# B&R Automation Studio project A2019059_Linka_Power_CP (part 2)

### Cpu.per - 5PC900_TS17_00/Cpu.per
```iecst
VAR_CONFIG
	Paletka AT %M0; (* *)
	P1_Skrutk_4F_DPS_M4_Vysunutie AT %MD5944; (* *)
	P1_Skrutk_4F_LavaK30_Vysunutie AT %MD5948; (* *)
	P1_Skrutk_4F_PravaK30_Vysunutie AT %MD5952; (* *)
	P1_Skrutk_4F_PrednaM4_Vysunutie AT %MD5956; (* *)
	P1_Skrutk_4F_ZadnaM4_Vysunutie AT %MD5960; (* *)
	P1_Skrutk_5F_DPS_M4_Vysunutie AT %MD5964; (* *)
	P1_Skrutk_5F_LavaK30_Vysunutie AT %MD5968; (* *)
	P1_Skrutk_5F_PravaK30_Vysunutie AT %MD5972; (* *)
	P1_Skrutk_5F_PrednaM4_Vysunutie AT %MD5976; (* *)
	P1_Skrutk_5F_ZadnaM4_Vysunutie AT %MD5980; (* *)
	P1_Skrutk_5H_LavaK30_Vysunutie AT %MD5984; (* *)
	P1_Skrutk_5H_LavaM5_Vysunutie AT %MD5988; (* *)
	P1_Skrutk_5H_PravaK30_Vysunutie AT %MD5992; (* *)
	P1_Skrutk_5H_PravaM5_Vysunutie AT %MD5996; (* *)
	P1_Skrutk_5H_StrednaM5_Vysunutie AT %MD6000; (* *)
	P2_Maticovacka_5H_Vysunutie AT %MD6004; (* *)
	P2_Skrutk_4F_LavaM4_Vysunutie AT %MD6008; (* *)
	P2_Skrutk_4F_LavaM6_Vysunutie AT %MD6012; (* *)
	P2_Skrutk_4F_PravaM4_Vysunutie AT %MD6016; (* *)
	P2_Skrutk_4F_PravaM6_Vysunutie AT %MD6020; (* *)
	P2_Skrutk_5F_LavaM4_Vysunutie AT %MD6024; (* *)
	P2_Skrutk_5F_LavaM6_Vysunutie AT %MD6028; (* *)
	P2_Skrutk_5F_PravaM4_Vysunutie AT %MD6032; (* *)
	P2_Skrutk_5F_PravaM6_Vysunutie AT %MD6036; (* *)
	P2_Skrutk_5H_LavaM5_Vysunutie AT %MD6040; (* *)
	P2_Skrutk_5H_PravaM5_Vysunutie AT %MD6044; (* *)
	P2_Skrutk_5H_StrednaM4_Vysunutie AT %MD6048; (* *)
	P3_Skrutk_4F_StredK40_Vysunutie AT %MD6052; (* *)
	P3_Skrutk_4F_StredM5_Vysunutie AT %MD6056; (* *)
	P3_Skrutk_5F_StredK40_Vysunutie AT %MD6060; (* *)
	P3_Skrutk_5F_StredM5_Vysunutie AT %MD6064; (* *)
	P3_Skrutk_5H_StredM5_Vysunutie AT %MD6068; (* *)
	Buffer_1 AT %M6072; (* *)
	Buffer_2 AT %M6280; (* *)
	Buffer_3 AT %M6488; (* *)
	Buffer_4 AT %M6696; (* *)
	Buffer_5 AT %M6904; (* *)
	Buffer_6 AT %M7112; (* *)
	Buffer_7 AT %M7320; (* *)
	Buffer_8 AT %M7528; (* *)
	Buffer_9 AT %M7736; (* *)
	Buffer_10 AT %M7944; (* *)
	Buffer_11 AT %M8152; (* *)
	Buffer_12 AT %M8360; (* *)
	Buffer_13 AT %M8568; (* *)
	Buffer_14 AT %M8776; (* *)
	Buffer_15 AT %M8984; (* *)
	Buffer_16 AT %M9192; (* *)
	Buffer_17 AT %M9400; (* *)
	Buffer_18 AT %M9608; (* *)
	Buffer_19 AT %M9816; (* *)
	Buffer_20 AT %M10024; (* *)
END_VAR
```

### IoMap.iom - 5PC900_TS17_00/IoMap.iom
```iecst
VAR_CONFIG
	Cyclic#1.Safety.IN.P2_Robot_TlacitkoCS_CH1_CS4 AT %IX."AB2.4_20xSI".SafeDigitalInput01;
	Cyclic#1.Safety.IN.P2_Robot_TlacitkoCS_CH2_CS4 AT %IX."AB2.4_20xSI".SafeDigitalInput02;
	Cyclic#1.Safety.IN.P2_Panel_TlacitkoCS_CH1_CS2 AT %IX."AB2.4_20xSI".SafeDigitalInput03;
	Cyclic#1.Safety.IN.P2_Panel_TlacitkoCS_CH2_CS2 AT %IX."AB2.4_20xSI".SafeDigitalInput04;
	Cyclic#1.Safety.IN.P2_VyblokovanieSafety_CH1_SA1 AT %IX."AB2.4_20xSI".SafeDigitalInput05;
	Cyclic#1.Safety.IN.P2_VyblokovanieSafety_CH2_SA1 AT %IX."AB2.4_20xSI".SafeDigitalInput06;
	Cyclic#1.Safety.IN.P2_Skrina_TlacitkoCS_CH1_CS3 AT %IX."AB2.4_20xSI".SafeDigitalInput07;
	Cyclic#1.Safety.IN.P2_Skrina_TlacitkoCS_CH2_CS3 AT %IX."AB2.4_20xSI".SafeDigitalInput08;
	Cyclic#1.Safety.IN.P2_ZaklTesn_PojazdSnim_CH1_B2 AT %IX."AB2.4_20xSI".SafeDigitalInput09;
	Cyclic#1.Safety.IN.P2_ZaklTesn_PojazdSnim_CH2_B2 AT %IX."AB2.4_20xSI".SafeDigitalInput10;
	Cyclic#1.P2_Dopravniky.IN.HornyDoprav_TeplotaMotora_OK AT %IX."AB2.4_20xSI".SafeDigitalInput11;
	Cyclic#1.P2_Dopravniky.IN.SpodnyDoprav_TeplotaMotora_OK AT %IX."AB2.4_20xSI".SafeDigitalInput12;
	Cyclic#1.Safety.IN.P2_ZaklTesn_Bumper_CH1_B1 AT %IX."AB2.4_20xSI".SafeDigitalInput13;
	Cyclic#1.Safety.IN.P2_ZaklTesn_Bumper_CH2_B1 AT %IX."AB2.4_20xSI".SafeDigitalInput14;
	Cyclic#1.P2_Pracovisko.IN.PrepatovaOchrana_OK AT %IX."AB2.7_16xDI".DigitalInput01;
	Cyclic#1.P2_Pracovisko.IN.NapajaniaRobota_OK AT %IX."AB2.7_16xDI".DigitalInput02;
	Cyclic#1.P2_SkrutkovacMatic.IN.NapajanieSkrutkovackyMatic_OK AT %IX."AB2.7_16xDI".DigitalInput03;
	Cyclic#1.P2_Srobovanie.IN.NapajanieSkrutkovackyM6_OK AT %IX."AB2.7_16xDI".DigitalInput04;
	Cyclic#1.P2_Srobovanie.IN.NapajanieSkrutkovackyM4_OK AT %IX."AB2.7_16xDI".DigitalInput05;
	Cyclic#1.P2_Srobovanie.IN.NapajanieSkrutkovackyM5_OK AT %IX."AB2.7_16xDI".DigitalInput06;
	Cyclic#1.P2_Srobovanie.IN.NapajanieVibroZasobnikaM5_OK AT %IX."AB2.7_16xDI".DigitalInput07;
	Cyclic#1.P2_Srobovanie.IN.NapajanieVibroZasobnikaM4_OK AT %IX."AB2.7_16xDI".DigitalInput08;
	Cyclic#1.P2_Srobovanie.IN.NapajanieVibroZasobnikaM6_OK AT %IX."AB2.7_16xDI".DigitalInput09;
	Cyclic#1.P2_SkrutkovacMatic.IN.NapajanieVibroZasobnikaMatic_OK AT %IX."AB2.7_16xDI".DigitalInput10;
	Cyclic#1.P2_Dopravniky.IN.HornyDoprav_READY AT %IX."AB2.7_16xDI".DigitalInput11;
	Cyclic#1.P2_Dopravniky.IN.SpodnyDoprav_READY AT %IX."AB2.7_16xDI".DigitalInput12;
	Cyclic#1.P2_Zvaranie.IN.NapajanieZvaracky_OK AT %IX."AB2.7_16xDI".DigitalInput13;
	Cyclic#1.P2_Cistenie.IN.Ionizator_Alarm1 AT %IX."AB2.7_16xDI".DigitalInput14;
	Cyclic#1.P2_Cistenie.IN.Ionizator_Alarm2 AT %IX."AB2.7_16xDI".DigitalInput15;
	Cyclic#1.P2_Cistenie.IN.Ionizator_Alarm3 AT %IX."AB2.7_16xDI".DigitalInput16;
	Cyclic#1.P2_Pracovisko.STAV.KartaAB24_OK AT %IX."AB2.4_20xSI".ModuleOk;
	Cyclic#1.P2_Pracovisko.STAV.KartaAB25_OK AT %IX."AB2.5_4xSO".ModuleOk;
	Cyclic#1.P2_Pracovisko.STAV.KartaAB26_OK AT %IX."AB2.6_4xSO".ModuleOk;
	Cyclic#1.P2_Pracovisko.STAV.KartaAB27_OK AT %IX."AB2.7_16xDI".ModuleOk;
	Cyclic#1.P2_Pracovisko.STAV.KartaAB28_OK AT %IX."AB2.8_16xDI".ModuleOk;
	Cyclic#1.P2_Pracovisko.STAV.KartaAB29_OK AT %IX."AB2.9_16xDO".ModuleOk;
	Cyclic#1.P2_Pracovisko.STAV.KartaAB210_OK AT %IX."AB2.10_16xDO".ModuleOk;
	Cyclic#1.P2_Pracovisko.STAV.KartaAB211_OK AT %IX."AB2.11_X2X".ModuleOk;
	Cyclic#1.P2_Pracovisko.STAV.ModulDM21_OK AT %IX."DM2.1_16DI/DO".ModuleOk;
	Cyclic#1.P2_Pracovisko.STAV.ModulDI21_OK AT %IX."DI2.1_8DI".ModuleOk;
	Cyclic#1.P2_Pracovisko.STAV.ModulDI22_OK AT %IX."DI2.2_16DI".ModuleOk;
	Cyclic#1.P2_Pracovisko.STAV.ModulDI23_OK AT %IX."DI2.3_16DI".ModuleOk;
	Cyclic#1.P2_Pracovisko.STAV.ModulDI24_OK AT %IX."DI2.4_16DI".ModuleOk;
	Cyclic#1.P2_Pracovisko.STAV.ModulDI25_OK AT %IX."DI2.5_16DI".ModuleOk;
	Cyclic#1.P2_Pracovisko.STAV.ModulSI21_OK AT %IX."SI2.1".ModuleOk;
	Cyclic#1.P2_Pracovisko.STAV.ModulSI22_OK AT %IX."SI2.2".ModuleOk;
	Cyclic#1.P2_Zvaranie.IN.ZvarackaStav_RUN AT %IX."AB2.8_16xDI".DigitalInput01;
	Cyclic#1.P2_Zvaranie.IN.ZvarackaStav_READY AT %IX."AB2.8_16xDI".DigitalInput02;
	Cyclic#1.Safety.IN.P2_SV_Ventil1_ZonaBunka AT %IX."AB2.8_16xDI".DigitalInput04;
	Cyclic#1.Safety.IN.P2_SV_Ventil2_ZonaBunka AT %IX."AB2.8_16xDI".DigitalInput05;
	Cyclic#1.Safety.IN.P2_SV_Ventil_ZonaMaticov AT %IX."AB2.8_16xDI".DigitalInput06;
	Cyclic#1.Safety.IN.P2_SV_ZonaCS AT %IX."AB2.8_16xDI".DigitalInput07;
	Cyclic#1.Safety.IN.P2_SV_ZonaBunka AT %IX."AB2.8_16xDI".DigitalInput08;
	Cyclic#1.Safety.IN.P2_SV_ZonaZaklTesneniaPojazd AT %IX."AB2.8_16xDI".DigitalInput09;
	Cyclic#1.Safety.IN.P2_SV_ZonaZaklTesneniaZdvih AT %IX."AB2.8_16xDI".DigitalInput10;
	Cyclic#1.P2_Pracovisko.OUT.Majak_ZeleneSvetlo AT %QX."AB2.9_16xDO".DigitalOutput01;
	Cyclic#1.P2_Pracovisko.OUT.Majak_ZlteSvetlo AT %QX."AB2.9_16xDO".DigitalOutput02;
	Cyclic#1.P2_Pracovisko.OUT.Majak_CerveneSvetlo AT %QX."AB2.9_16xDO".DigitalOutput03;
	Cyclic#1.P2_Pracovisko.OUT.Majak_Hukacka AT %QX."AB2.9_16xDO".DigitalOutput04;
	Cyclic#1.P2_Cistenie.OUT.Ionizator_RUN_ZX2 AT %QX."AB2.9_16xDO".DigitalOutput09;
	Cyclic#1.P2_Zvaranie.OUT.Zvaracka_START AT %QX."AB2.9_16xDO".DigitalOutput10;
	Cyclic#1.P2_Zvaranie.OUT.Zvaracka_RESET AT %QX."AB2.9_16xDO".DigitalOutput11;
	Cyclic#1.P2_SkrutkovacMatic.OUT.SkrutkMatic_VYSUN_YV62 AT %QX."AB2.10_16xDO".DigitalOutput01;
	Cyclic#1.P2_SkrutkovacMatic.OUT.SkrutkMatic_ZASUN_YV75 AT %QX."AB2.10_16xDO".DigitalOutput02;
	Cyclic#1.P2_Pracovisko.OUT.OsvetlenieBunky AT %QX."AB2.10_16xDO".DigitalOutput03;
	Cyclic#1.P2_Srobovanie.OUT.ZasobSrobM6_Banner_CervenaLED AT %QX."DM2.1_16DI/DO".DigitalOutput09;
	Cyclic#1.P2_Srobovanie.IN.ZasobSrobM6_Banner_SB3 AT %IX."DM2.1_16DI/DO".DigitalInput10;
	Cyclic#1.P2_SkrutkovacMatic.IN.ZasobMatic_Banner_SB4 AT %IX."DM2.1_16DI/DO".DigitalInput12;
	Cyclic#1.P2_Srobovanie.OUT.ZasobSrobM4_Banner_CervenaLED AT %QX."DM2.1_16DI/DO".DigitalOutput13;
	Cyclic#1.P2_Srobovanie.IN.ZasobSrobM4_Banner_SB5 AT %IX."DM2.1_16DI/DO".DigitalInput14;
	Cyclic#1.P2_Srobovanie.OUT.ZasobSrobM5_Banner_CervenaLED AT %QX."DM2.1_16DI/DO".DigitalOutput15;
	Cyclic#1.P2_Srobovanie.IN.ZasobSrobM5_Banner_SB6 AT %IX."DM2.1_16DI/DO".DigitalInput16;
	Cyclic#1.P2_SkrutkovacMatic.OUT.ZasobMatic_Banner_CervenaLED AT %QX."DM2.1_16DI/DO".DigitalOutput11;
	Cyclic#1.P2_Srobovanie.IN.ManipulOsY_LimSnimacPOS_IS19 AT %IX."DI2.1_8DI".DigitalInput01;
	Cyclic#1.P2_Srobovanie.IN.ManipulOsY_LimSnimacNEG_IS20 AT %IX."DI2.1_8DI".DigitalInput02;
	Cyclic#1.P2_Srobovanie.IN.ManipulOsX_LimSnimacPOS_IS21 AT %IX."DI2.1_8DI".DigitalInput03;
	Cyclic#1.P2_Srobovanie.IN.ManipulOsX_LimSnimacNEG_IS22 AT %IX."DI2.1_8DI".DigitalInput04;
	Cyclic#1.P2_Zvaranie.IN.ZdvihZvarania_RefSnimac_IS9 AT %IX."DI2.2_16DI".DigitalInput01;
	Cyclic#1.P2_Zvaranie.IN.PojazdZvarania_PozVPRAVO_IS10 AT %IX."DI2.2_16DI".DigitalInput02;
	Cyclic#1.P2_Zvaranie.IN.PojazdZvarania_PozVLAVO_IS11 AT %IX."DI2.2_16DI".DigitalInput03;
	Cyclic#1.P2_Cistenie.IN.Dvere_OTVORENE_MS7 AT %IX."DI2.2_16DI".DigitalInput09;
	Cyclic#1.P2_Cistenie.IN.Dvere_ZATVORENE_MS8 AT %IX."DI2.2_16DI".DigitalInput10;
	Cyclic#1.P2_Cistenie.IN.VakumDosiahnute_S5 AT %IX."DI2.2_16DI".DigitalInput11;
	Cyclic#1.P2_Robot.IN.DokStanPritGripra_MVcase_IS1 AT %IX."DI2.2_16DI".DigitalInput12;
	Cyclic#1.P2_Robot.IN.DokStanPritGripra_BusBary45F_IS2 AT %IX."DI2.2_16DI".DigitalInput13;
	Cyclic#1.P2_Robot.IN.DokStanPritGripra_BusBary5H_IS3 AT %IX."DI2.2_16DI".DigitalInput14;
	Cyclic#1.P2_Robot.IN.SnimacVakua_45F_S1 AT %IX."DI2.2_16DI".DigitalInput15;
	Cyclic#1.P2_Robot.IN.SnimacVakua_5H_S2 AT %IX."DI2.2_16DI".DigitalInput16;
	Cyclic#1.P2_StoperMaticovacky.IN.Centrovanie_VYSUNUTE_IS12 AT %IX."DI2.3_16DI".DigitalInput01;
	Cyclic#1.P2_StoperMaticovacky.IN.Centrovanie_ZASUNUTE_IS13 AT %IX."DI2.3_16DI".DigitalInput02;
	Cyclic#1.P2_StoperSrobovania.IN.Centrovanie_VYSUNUTE_IS14 AT %IX."DI2.3_16DI".DigitalInput03;
	Cyclic#1.P2_StoperSrobovania.IN.Centrovanie_ZASUNUTE_IS15 AT %IX."DI2.3_16DI".DigitalInput04;
	Cyclic#1.P2_StoperZvarania.IN.Centrovanie_VYSUNUTE_IS16 AT %IX."DI2.3_16DI".DigitalInput05;
	Cyclic#1.P2_StoperZvarania.IN.Centrovanie_ZASUNUTE_IS17 AT %IX."DI2.3_16DI".DigitalInput06;
	Cyclic#1.P2_Dopravniky.IN.SpodnyDoprav_Zaplnenie_IS18 AT %IX."DI2.3_16DI".DigitalInput07;
	Cyclic#1.P2_Srobovanie.IN.SkrutkM5_SrobaPresla_IS32 AT %IX."DI2.3_16DI".DigitalInput15;
	Cyclic#1.P2_Srobovanie.IN.SkrutkM5_Cist_SrobaPresla_IS31 AT %IX."DI2.3_16DI".DigitalInput14;
	Cyclic#1.P2_Srobovanie.IN.SkrutkM5_Cist_BrzdaZatvorena_MS2 AT %IX."DI2.3_16DI".DigitalInput13;
	Cyclic#1.P2_Srobovanie.IN.SkrutkM5_Cist_BrzdaOtvorena_MS1 AT %IX."DI2.3_16DI".DigitalInput12;
	Cyclic#1.P2_Srobovanie.IN.NastrelSrobM5_SrobaPresla_IS29 AT %IX."DI2.3_16DI".DigitalInput11;
	Cyclic#1.P2_Srobovanie.IN.ZasobSrobM5_ListaPLNA_OS3 AT %IX."DI2.3_16DI".DigitalInput10;
	Cyclic#1.P2_Srobovanie.IN.ZasobSrobM5_PRAZDNY_IS28 AT %IX."DI2.3_16DI".DigitalInput09;
	Cyclic#1.P2_SkrutkovacMatic.IN.ZasobMatic_PRAZDNY_IS23 AT %IX."DI2.4_16DI".DigitalInput01;
	Cyclic#1.P2_SkrutkovacMatic.IN.ZasobMatic_ListaPLNA_OS1 AT %IX."DI2.4_16DI".DigitalInput02;
	Cyclic#1.P2_SkrutkovacMatic.IN.OddelMatic_MaticaPresla_IS24 AT %IX."DI2.4_16DI".DigitalInput03;
	Cyclic#1.P2_SkrutkovacMatic.IN.DavkMatic_PritomnostMatice_OS2 AT %IX."DI2.4_16DI".DigitalInput04;
	Cyclic#1.P2_SkrutkovacMatic.IN.DavkMatic_ZASUNUTY_IS25 AT %IX."DI2.4_16DI".DigitalInput05;
	Cyclic#1.P2_SkrutkovacMatic.IN.DavkMatic_VYSUNUTY_IS26 AT %IX."DI2.4_16DI".DigitalInput06;
	Cyclic#1.P2_SkrutkovacMatic.IN.DavkMatic_MaticaPresla_IS27 AT %IX."DI2.4_16DI".DigitalInput07;
	Cyclic#1.P2_SkrutkovacMatic.IN.SkrutkMatic_ZASUNUTY_MS9 AT %IX."DI2.4_16DI".DigitalInput08;
	Cyclic#1.P2_Srobovanie.IN.ZasobSrobM4_PRAZDNY_IS33 AT %IX."DI2.4_16DI".DigitalInput09;
	Cyclic#1.P2_Srobovanie.IN.ZasobSrobM4_ListaPLNA_OS4 AT %IX."DI2.4_16DI".DigitalInput10;
	Cyclic#1.P2_Srobovanie.IN.NastrelSrobM4_SrobaPresla_IS34 AT %IX."DI2.4_16DI".DigitalInput11;
	Cyclic#1.P2_Srobovanie.IN.SkrutkM4_Cist_BrzdaOtvorena_MS12 AT %IX."DI2.4_16DI".DigitalInput12;
	Cyclic#1.P2_Srobovanie.IN.SkrutkM4_Cist_BrzdaZatvoren_MS13 AT %IX."DI2.4_16DI".DigitalInput13;
	Cyclic#1.P2_Srobovanie.IN.SkrutkM4_Cist_SrobaPresla_IS35 AT %IX."DI2.4_16DI".DigitalInput14;
	Cyclic#1.P2_Srobovanie.IN.SkrutkM4_SrobaPresla_IS30 AT %IX."DI2.4_16DI".DigitalInput15;
	Cyclic#1.P2_Srobovanie.IN.ZasobSrobM6_PRAZDNY_IS36 AT %IX."DI2.5_16DI".DigitalInput01;
	Cyclic#1.P2_Srobovanie.IN.ZasobSrobM6_ListaPLNA_OS5 AT %IX."DI2.5_16DI".DigitalInput02;
	Cyclic#1.P2_Srobovanie.IN.NastrelSrobM6_SrobaPresla_IS37 AT %IX."DI2.5_16DI".DigitalInput03;
	Cyclic#1.P2_Srobovanie.IN.SkrutkM6_Cist_BrzdaOtvorena_MS15 AT %IX."DI2.5_16DI".DigitalInput04;
	Cyclic#1.P2_Srobovanie.IN.SkrutkM6_Cist_BrzdaZatvoren_MS16 AT %IX."DI2.5_16DI".DigitalInput05;
	Cyclic#1.P2_Srobovanie.IN.SkrutkM6_Cist_SrobaPresla_IS39 AT %IX."DI2.5_16DI".DigitalInput06;
	Cyclic#1.P2_Srobovanie.IN.SkrutkM6_SrobaPresla_IS38 AT %IX."DI2.5_16DI".DigitalInput07;
	Cyclic#1.P2_ZakladacTesnenia.IN.ZdvihZaklad_RefSnimac_IS8 AT %IX."DI2.5_16DI".DigitalInput09;
	Cyclic#1.P2_ZakladacTesnenia.IN.Vozik_Zaklad_PritomPowerCP_IOS6 AT %IX."DI2.5_16DI".DigitalInput14;
	Cyclic#1.P2_ZakladacTesnenia.IN.Kopito_ZakladPoloha_IS7 AT %IX."DI2.5_16DI".DigitalInput15;
	Cyclic#1.P2_Pracovisko.IN.PrivodVzduchu_SnimacTlaku_S3 AT %IX."DI2.5_16DI".DigitalInput16;
	Cyclic#1.Safety.IN.P2_ZamkyBunky_CH1 AT %IX."SI2.1".SafeDigitalInput01;
	Cyclic#1.Safety.IN.P2_ZamkyBunky_CH2 AT %IX."SI2.1".SafeDigitalInput02;
	Cyclic#1.Safety.OUT.P2_ZamkniZamok_PredneDvereLS AT %QX."DM2.1_16DI/DO".DigitalOutput01;
	Cyclic#1.Safety.IN.P2_PredneDvereLS_PritomPetlice AT %IX."DM2.1_16DI/DO".DigitalInput02;
	Cyclic#1.Safety.OUT.P2_ZamkniZamok_PredneDverePS AT %QX."DM2.1_16DI/DO".DigitalOutput03;
	Cyclic#1.Safety.IN.P2_PredneDverePS_PritomPetlice AT %IX."DM2.1_16DI/DO".DigitalInput04;
	Cyclic#1.Safety.IN.P2_ZaklTesn_Bariera_CH1_BC1 AT %IX."SI2.1".SafeDigitalInput03;
	Cyclic#1.Safety.IN.P2_ZaklTesn_Bariera_CH2_BC1 AT %IX."SI2.1".SafeDigitalInput04;
	Cyclic#1.Safety.IN.P2_TlacitkoCS_CH1_CS1 AT %IX."SI2.1".SafeDigitalInput05;
	Cyclic#1.Safety.IN.P2_TlacitkoCS_CH2_CS1 AT %IX."SI2.1".SafeDigitalInput06;
	Cyclic#1.Safety.IN.P2_VstupBunky_Bariera_CH1_BC2 AT %IX."SI2.2".SafeDigitalInput01;
	Cyclic#1.Safety.IN.P2_VstupBunky_Bariera_CH2_BC2 AT %IX."SI2.2".SafeDigitalInput02;
	Cyclic#1.Safety.IN.P2_ZaklTesn_DvojrOvladLS_CH1_SB1 AT %IX."SI2.2".SafeDigitalInput05;
	Cyclic#1.Safety.IN.P2_ZaklTesn_DvojrOvladLS_CH2_SB1 AT %IX."SI2.2".SafeDigitalInput06;
	Cyclic#1.Safety.IN.P2_ZaklTesn_DvojrOvladPS_CH1_SB2 AT %IX."SI2.2".SafeDigitalInput07;
	Cyclic#1.Safety.IN.P2_ZaklTesn_DvojrOvladPS_CH2_SB2 AT %IX."SI2.2".SafeDigitalInput08;
	Cyclic#1.P2_Pracovisko.OUT.VT1_OUT1 AT %QB."VentilovyTerminal_VT1".OUT1_I2200_S01Out;
	Cyclic#1.P2_Pracovisko.OUT.VT1_OUT2 AT %QB."VentilovyTerminal_VT1".OUT2_I2200_S02Out;
	Cyclic#1.P2_Pracovisko.OUT.VT1_OUT3 AT %QB."VentilovyTerminal_VT1".OUT3_I2200_S03Out;
	Cyclic#1.P2_Pracovisko.OUT.VT1_OUT4 AT %QB."VentilovyTerminal_VT1".OUT4_I2200_S04Out;
	Cyclic#1.P2_Pracovisko.OUT.VT2_OUT1 AT %QB."VentilovyTerminal_VT2".OUT1_I2200_S01Out;
	Cyclic#1.P2_Pracovisko.OUT.VT2_OUT2 AT %QB."VentilovyTerminal_VT2".OUT2_I2200_S02Out;
	Cyclic#1.P2_Pracovisko.OUT.VT2_OUT3 AT %QB."VentilovyTerminal_VT2".OUT3_I2200_S03Out;
	Cyclic#1.P2_Pracovisko.OUT.VT2_OUT4 AT %QB."VentilovyTerminal_VT2".OUT4_I2200_S04Out;
	Cyclic#1.P2_Pracovisko.OUT.VT3_OUT1 AT %QB."VentilovyTerminal_VT3".OUT1_I2200_S01Out;
	Cyclic#1.P2_Pracovisko.OUT.VT3_OUT2 AT %QB."VentilovyTerminal_VT3".OUT2_I2200_S02Out;
	Cyclic#1.P2_Pracovisko.OUT.VT3_OUT3 AT %QB."VentilovyTerminal_VT3".OUT3_I2200_S03Out;
	Cyclic#1.P2_Pracovisko.OUT.VT3_OUT4 AT %QB."VentilovyTerminal_VT3".OUT4_I2200_S04Out;
	Cyclic#1.Safety.IN.ZonaCS_RESET AT %QX."SL1_SafetyMaster".BOOL101;
	Cyclic#1.Safety.IN.P2_ZonaZaklTesneniaPojazd_RESET AT %QX."SL1_SafetyMaster".BOOL102;
	Cyclic#1.Safety.IN.P2_ZonaZaklTesneniaZdvih_RESET AT %QX."SL1_SafetyMaster".BOOL103;
	Cyclic#1.Safety.IN.P2_ZonaMaticovacky_RESET AT %QX."SL1_SafetyMaster".BOOL104;
	Cyclic#1.Safety.IN.P2_ZonaBunky_RESET AT %QX."SL1_SafetyMaster".BOOL105;
	Cyclic#1.P2_Pracovisko.IN.PrivodVzduchu_SnimacTlaku_S3 AT %QX."SL1_SafetyMaster".BOOL106;
	Cyclic#1.Safety.IN.P2_SV_Ventil_ZonaMaticov AT %QX."SL1_SafetyMaster".BOOL107;
	Cyclic#1.Safety.IN.P2_SV_Ventil1_ZonaBunka AT %QX."SL1_SafetyMaster".BOOL108;
	Cyclic#1.Safety.IN.P2_SV_Ventil2_ZonaBunka AT %QX."SL1_SafetyMaster".BOOL109;
	Cyclic#1.Safety.IN.P2_SV_ZonaBunka AT %QX."SL1_SafetyMaster".BOOL110;
	Cyclic#1.Safety.IN.P2_SV_ZonaCS AT %QX."SL1_SafetyMaster".BOOL111;
	Cyclic#1.Safety.IN.P2_SV_ZonaZaklTesneniaPojazd AT %QX."SL1_SafetyMaster".BOOL112;
	Cyclic#1.Safety.IN.P2_SV_ZonaZaklTesneniaZdvih AT %QX."SL1_SafetyMaster".BOOL113;
	Cyclic#1.Safety.STAV.SafetyPLC_Nabehlo AT %IX."SL1_SafetyMaster".BOOL001;
	Cyclic#1.Safety.STAV.P2_TlacitkoCS_AKTIVNE AT %IX."SL1_SafetyMaster".BOOL002;
	Cyclic#1.Safety.STAV.P2_Panel_TlacitkoCS_AKTIVNE AT %IX."SL1_SafetyMaster".BOOL003;
	Cyclic#1.Safety.STAV.P2_Robot_TlacitkoCS_AKTIVNE AT %IX."SL1_SafetyMaster".BOOL004;
	Cyclic#1.Safety.STAV.P2_Skrina_TlacitkoCS_AKTIVNE AT %IX."SL1_SafetyMaster".BOOL005;
	Cyclic#1.Safety.STAV.P2_VstupBunky_Bariera_AKTIVNA AT %IX."SL1_SafetyMaster".BOOL006;
	Cyclic#1.Safety.STAV.P2_ZaklTesnenia_Bariera_AKTIVNA AT %IX."SL1_SafetyMaster".BOOL007;
	Cyclic#1.Safety.STAV.P2_ZaklTesnenia_Bumper_AKTIVNY AT %IX."SL1_SafetyMaster".BOOL008;
	Cyclic#1.Safety.STAV.P2_DvojrucneOvladanie_AKTIVNE AT %IX."SL1_SafetyMaster".BOOL009;
	Cyclic#1.Safety.STAV.P2_ZamkyBunky_AKTIVNE AT %IX."SL1_SafetyMaster".BOOL010;
	Cyclic#1.Safety.STAV.P2_ZonaMaticovacky_AKTIVNA AT %IX."SL1_SafetyMaster".BOOL011;
	Cyclic#1.Safety.STAV.P2_ZonaZaklTesnenPojazd_AKTIVNA AT %IX."SL1_SafetyMaster".BOOL012;
	Cyclic#1.Safety.STAV.P2_ZonaZaklTesnenZdvih_AKTIVNA AT %IX."SL1_SafetyMaster".BOOL013;
	Cyclic#1.Safety.STAV.ZonaCS_AKTIVNA AT %IX."SL1_SafetyMaster".BOOL014;
	Cyclic#1.Safety.STAV.P2_ZonaBunky_AKTIVNA AT %IX."SL1_SafetyMaster".BOOL015;
	Cyclic#1.Safety.STAV.P2_VyblokovanieSafety_AKTIVNE AT %IX."SL1_SafetyMaster".BOOL016;
	Cyclic#1.Safety.STAV.P2_ZaklTesnenia_Pojazd_ZASUNUTY AT %IX."SL1_SafetyMaster".BOOL017;
	Cyclic#1.Safety.IN.P2_StavKartySO_AB25 AT %QD."SL1_SafetyMaster".UDINT101;
	Cyclic#1.Safety.IN.P2_StavKartySO_AB26 AT %QD."SL1_SafetyMaster".UDINT102;
	Cyclic#1.Safety.IN.P2_ReleaseKartySO_AB25 AT %QX."SL1_SafetyMaster".BOOL114;
	Cyclic#1.Safety.IN.P2_ReleaseKartySO_AB26 AT %QX."SL1_SafetyMaster".BOOL115;
	Cyclic#1.P2_ZakladacTesnenia.OUT.LED_DvojrucneOvladanie_H1 AT %QX."AB2.10_16xDO".DigitalOutput10;
	Cyclic#1.P2_StoperZaklTesnenia.PAR.SnimacPaletky_IOLinkInputs AT %IO."DS2_2".InputData01;
	Cyclic#1.P2_StoperMaticovacky.PAR.SnimacPaletky_IOLinkInputs AT %IO."DS2_2".InputData02;
	Cyclic#1.P2_StoperSrobovania.PAR.SnimacPaletky_IOLinkInputs AT %IO."DS2_2".InputData03;
	Cyclic#1.P2_StoperZvarania.PAR.SnimacPaletky_IOLinkInputs AT %IO."DS2_2".InputData04;
	Cyclic#1.P2_Robot.PAR.Modul_IOLink_Inputs AT %IB."DS2_1".InputData01_1;
	Cyclic#1.P2_StoperZaklTesnenia.PAR.Banner_IOLinkInputs AT %IB."DS2_1".InputData02_1;
	Cyclic#1.P2_StoperZaklTesnenia.PAR.Banner_IOLinkOutputs AT %QB."DS2_1".OutputData02_1;
	Cyclic#1.P2_Robot.PAR.Griper_4F_5F_5H_IOLink_Inputs AT %IW."DS2_1".InputData04_1;
	Cyclic#1.P2_StoperZaklTesnenia.PAR.Banner_IOLinkInputs AT %IO."DS2_1".InputData02;
	Cyclic#1.P2_StoperZaklTesnenia.PAR.Banner_IOLinkOutputs AT %QO."DS2_1".OutputData02;
	Cyclic#1.P2_Pracovisko.OUT.Osvetlenie_CAM7_CAM17 AT %QX."AB2.10_16xDO".DigitalOutput06;
	Cyclic#1.P2_Pracovisko.OUT.Osvetlenie_CAM1 AT %QX."AB2.10_16xDO".DigitalOutput07;
	Cyclic#1.P2_Pracovisko.OUT.Osvetlenie_CAM10 AT %QX."AB2.10_16xDO".DigitalOutput08;
	Cyclic#1.P2_Pracovisko.OUT.Osvetlenie_CAM11 AT %QX."AB2.10_16xDO".DigitalOutput09;
	Cyclic#1.P2_Srobovanie.IN.SkrutkM6_ZASUNUTY_MS14 AT %IX."DI2.1_8DI".DigitalInput05;
	Cyclic#1.P2_Srobovanie.IN.SkrutkM4_ZASUNUTY_MS10 AT %IX."DI2.1_8DI".DigitalInput06;
	Cyclic#1.P2_Srobovanie.IN.SkrutkM5_ZASUNUTY_MS11 AT %IX."DI2.1_8DI".DigitalInput07;
	Cyclic#1.P2_SkrutkovacMatic.IN.OddelMatic_Otoceny_VZAD_MS58 AT %IX."DI2.2_16DI".DigitalInput04;
	Cyclic#1.P2_SkrutkovacMatic.IN.OddelMatic_Otoceny_VPRED_MS59 AT %IX."DI2.2_16DI".DigitalInput05;
	Cyclic#1.P2_SkrutkovacMatic.OUT.ZasobMatic_Vibrovanie_RUN_FM1 AT %QX."AB2.9_16xDO".DigitalOutput05;
	Cyclic#1.P2_Srobovanie.OUT.ZasobSrobM6_Vibrovanie_RUN_FM2 AT %QX."AB2.9_16xDO".DigitalOutput06;
	Cyclic#1.P2_Srobovanie.OUT.ZasobSrobM4_Vibrovanie_RUN_FM3 AT %QX."AB2.9_16xDO".DigitalOutput07;
	Cyclic#1.P2_Srobovanie.OUT.ZasobSrobM5_Vibrovanie_RUN_FM4 AT %QX."AB2.9_16xDO".DigitalOutput08;
	Cyclic#1.Safety.IN.P1_Robot_TlacitkoCS_CH1_CS10 AT %IX."AB1.4_20xSI".SafeDigitalInput01;
	Cyclic#1.Safety.IN.P1_Robot_TlacitkoCS_CH2_CS10 AT %IX."AB1.4_20xSI".SafeDigitalInput02;
	Cyclic#1.Safety.IN.P1_Panel_TlacitkoCS_CH1_CS8 AT %IX."AB1.4_20xSI".SafeDigitalInput03;
	Cyclic#1.Safety.IN.P1_Panel_TlacitkoCS_CH2_CS8 AT %IX."AB1.4_20xSI".SafeDigitalInput04;
	Cyclic#1.Safety.IN.P1_VyblokovanieSafety_CH1_SA1 AT %IX."AB1.4_20xSI".SafeDigitalInput05;
	Cyclic#1.Safety.IN.P1_VyblokovanieSafety_CH2_SA1 AT %IX."AB1.4_20xSI".SafeDigitalInput06;
	Cyclic#1.Safety.IN.P1_Skrina_TlacitkoCS_CH1_CS5 AT %IX."AB1.4_20xSI".SafeDigitalInput07;
	Cyclic#1.Safety.IN.P1_Skrina_TlacitkoCS_CH2_CS5 AT %IX."AB1.4_20xSI".SafeDigitalInput08;
	Cyclic#1.Safety.IN.P1_Vytah_SnimHornaPoz_CH1_B8 AT %IX."AB1.4_20xSI".SafeDigitalInput09;
	Cyclic#1.Safety.IN.P1_Vytah_SnimHornaPoz_CH2_B8 AT %IX."AB1.4_20xSI".SafeDigitalInput10;
	Cyclic#1.P1_Dopravniky.IN.HornyDoprav_TeplotaMotora_OK AT %IX."AB1.4_20xSI".SafeDigitalInput12;
	Cyclic#1.P1_Dopravniky.IN.SpodnyDoprav_TeplotaMotora_OK AT %IX."AB1.4_20xSI".SafeDigitalInput13;
	Cyclic#1.P1_Vytah.IN.Dopravnik_TeplotaMotora_OK AT %IX."AB1.4_20xSI".SafeDigitalInput11;
	Cyclic#1.P1_Pracovisko.STAV.KartaAB14_OK AT %IX."AB1.4_20xSI".ModuleOk;
	Cyclic#1.P1_Pracovisko.STAV.KartaAB15_OK AT %IX."AB1.5_4xSO".ModuleOk;
	Cyclic#1.P1_Pracovisko.STAV.KartaAB16_OK AT %IX."AB1.6_16xDI".ModuleOk;
	Cyclic#1.P1_Pracovisko.IN.PrepatovaOchrana_OK AT %IX."AB1.6_16xDI".DigitalInput01;
	Cyclic#1.P1_Pracovisko.IN.NapajaniaRobota_OK AT %IX."AB1.6_16xDI".DigitalInput02;
	Cyclic#1.P1_Srobovanie.IN.NapajanieSkrutkovackyK30_OK AT %IX."AB1.6_16xDI".DigitalInput03;
	Cyclic#1.P1_Srobovanie.IN.NapajanieSkrutkovackyM5_OK AT %IX."AB1.6_16xDI".DigitalInput04;
	Cyclic#1.P1_Srobovanie.IN.NapajanieSkrutkovackyM4_OK AT %IX."AB1.6_16xDI".DigitalInput05;
	Cyclic#1.P1_Srobovanie.IN.NapajanieVibroZasobnikaK30_OK AT %IX."AB1.6_16xDI".DigitalInput06;
	Cyclic#1.P1_Srobovanie.IN.NapajanieVibroZasobnikaM4_OK AT %IX."AB1.6_16xDI".DigitalInput07;
	Cyclic#1.P1_Pracovisko.STAV.ModulSI11_OK AT %IX."SI1.1".ModuleOk;
	Cyclic#1.Safety.IN.P1_ZamkyBunky_CH1 AT %IX."SI1.1".SafeDigitalInput01;
	Cyclic#1.Safety.IN.P1_ZamkyBunky_CH2 AT %IX."SI1.1".SafeDigitalInput02;
	Cyclic#1.Safety.IN.P1_Vytah_Bariera_CH1_BC6 AT %IX."SI1.1".SafeDigitalInput03;
	Cyclic#1.Safety.IN.P1_Vytah_Bariera_CH2_BC6 AT %IX."SI1.1".SafeDigitalInput04;
	Cyclic#1.P1_Pracovisko.STAV.ModulSI12_OK AT %IX."SI1.2".ModuleOk;
	Cyclic#1.Safety.IN.P1_VstupBunky_Bariera_CH1_BC7 AT %IX."SI1.2".SafeDigitalInput01;
	Cyclic#1.Safety.IN.P1_VstupBunky_Bariera_CH2_BC7 AT %IX."SI1.2".SafeDigitalInput02;
	Cyclic#1.Safety.IN.P1_VystupTunela_Bariera_CH1_BC8 AT %IX."SI1.2".SafeDigitalInput03;
	Cyclic#1.Safety.IN.P1_VystupTunela_Bariera_CH2_BC8 AT %IX."SI1.2".SafeDigitalInput04;
	Cyclic#1.P1_Srobovanie.IN.NapajanieVibroZasobnikaM5_OK AT %IX."AB1.6_16xDI".DigitalInput08;
	Cyclic#1.P1_Srobovanie.IN.NapajanieVibroListyM5_OK AT %IX."AB1.6_16xDI".DigitalInput09;
	Cyclic#1.P1_Vytah.IN.Dopravnik_READY AT %IX."AB1.6_16xDI".DigitalInput10;
	Cyclic#1.P1_Dopravniky.IN.HornyDoprav_READY AT %IX."AB1.6_16xDI".DigitalInput11;
	Cyclic#1.P1_Dopravniky.IN.SpodnyDoprav_READY AT %IX."AB1.6_16xDI".DigitalInput12;
	Cyclic#1.Safety.IN.P1_SV_Ventil1_ZonaBunka_B9 AT %IX."AB1.6_16xDI".DigitalInput13;
	Cyclic#1.Safety.IN.P1_SV_Ventil2_ZonaBunka_B10 AT %IX."AB1.6_16xDI".DigitalInput14;
	Cyclic#1.P1_Pracovisko.STAV.KartaAB17_OK AT %IX."AB1.7_16xDI".ModuleOk;
	Cyclic#1.Safety.IN.P1_SV_ZonaCS AT %IX."AB1.7_16xDI".DigitalInput09;
	Cyclic#1.Safety.IN.P1_SV_ZonaBunka AT %IX."AB1.7_16xDI".DigitalInput10;
	Cyclic#1.Safety.IN.P1_SV_ZonaVytah AT %IX."AB1.7_16xDI".DigitalInput11;
	Cyclic#1.P1_Pracovisko.STAV.KartaAB18_OK AT %IX."AB1.8_16xDO".ModuleOk;
	Cyclic#1.P1_Pracovisko.OUT.Majak_ZeleneSvetlo AT %QX."AB1.8_16xDO".DigitalOutput01;
	Cyclic#1.P1_Pracovisko.OUT.Majak_ZlteSvetlo AT %QX."AB1.8_16xDO".DigitalOutput02;
	Cyclic#1.P1_Pracovisko.OUT.Majak_CerveneSvetlo AT %QX."AB1.8_16xDO".DigitalOutput03;
	Cyclic#1.P1_Pracovisko.OUT.Majak_Hukacka AT %QX."AB1.8_16xDO".DigitalOutput04;
	Cyclic#1.P1_Srobovanie.OUT.ZasobSrobK30_Vibrovanie_RUN_FM8 AT %QX."AB1.8_16xDO".DigitalOutput05;
	Cyclic#1.P1_Srobovanie.OUT.ZasobSrobM4_Vibrovanie_RUN_FM9 AT %QX."AB1.8_16xDO".DigitalOutput06;
	Cyclic#1.P1_Srobovanie.OUT.ZasobSrobM5_Vibrov_RUN_FM10 AT %QX."AB1.8_16xDO".DigitalOutput07;
	Cyclic#1.P1_Srobovanie.OUT.VibrolistaSrobM5_Vibrov_RUN_FM11 AT %QX."AB1.8_16xDO".DigitalOutput08;
	Cyclic#1.P1_Pracovisko.OUT.OsvetlenieBunky AT %QX."AB1.8_16xDO".DigitalOutput09;
	Cyclic#1.P1_Dopravniky.OUT.HornyDoprav_ChodVPRED_M32 AT %QX."AB1.8_16xDO".DigitalOutput11;
	Cyclic#1.P1_Dopravniky.OUT.SpodnyDoprav_ChodVPRED_M29 AT %QX."AB1.8_16xDO".DigitalOutput12;
	Cyclic#1.P1_Pracovisko.STAV.KartaAB19_OK AT %IX."AB1.9_16xDO".ModuleOk;
	Cyclic#1.P1_Pracovisko.OUT.Osvetlenie_CAM2 AT %QX."AB1.9_16xDO".DigitalOutput05;
	Cyclic#1.P1_Pracovisko.OUT.Osvetlenie_CAM4 AT %QX."AB1.9_16xDO".DigitalOutput06;
	Cyclic#1.P1_Pracovisko.OUT.Osvetlenie_CAM6 AT %QX."AB1.9_16xDO".DigitalOutput07;
	Cyclic#1.P1_Pracovisko.STAV.ModulDI13_OK AT %IX."DI1.3_8DI".ModuleOk;
	Cyclic#1.P1_Pracovisko.STAV.ModulDM11_OK AT %IX."DM1.1_16DI/DO".ModuleOk;
	Cyclic#1.P1_Pracovisko.STAV.ModulDI12_OK AT %IX."DI1.2_16DI".ModuleOk;
	Cyclic#1.P1_Pracovisko.STAV.ModulDS11_OK AT %IX."DS1_1".ModuleOk;
	Cyclic#1.P1_Pracovisko.STAV.ModulDI11_OK AT %IX."DI1.1_16DI".ModuleOk;
	Cyclic#1.P1_Pracovisko.STAV.ModulDI14_OK AT %IX."DI1.4_8DI".ModuleOk;
	Cyclic#1.P1_Pracovisko.STAV.ModulDS12_OK AT %IX."DS1_2".ModuleOk;
	Cyclic#1.P1_Robot.OUT.OtvorGriper_YV97 AT %QX."DM1.1_16DI/DO".DigitalOutput07;
	Cyclic#1.P1_Robot.OUT.ZatvorGriper_YV98 AT %QX."DM1.1_16DI/DO".DigitalOutput08;
	Cyclic#1.P1_Srobovanie.OUT.ZasobSrobK30_Banner_CervenaLED AT %QX."DM1.1_16DI/DO".DigitalOutput09;
	Cyclic#1.P1_Srobovanie.IN.ZasobSrobK30_Banner_SB9 AT %IX."DM1.1_16DI/DO".DigitalInput10;
	Cyclic#1.P1_Srobovanie.OUT.ZasobSrobM5_Banner_CervenaLED AT %QX."DM1.1_16DI/DO".DigitalOutput11;
	Cyclic#1.P1_Srobovanie.IN.ZasobSrobM5_Banner_SB10 AT %IX."DM1.1_16DI/DO".DigitalInput12;
	Cyclic#1.P1_Srobovanie.OUT.ZasobSrobM4_Banner_CervenaLED AT %QX."DM1.1_16DI/DO".DigitalOutput13;
	Cyclic#1.P1_Srobovanie.IN.ZasobSrobM4_Banner_SB8 AT %IX."DM1.1_16DI/DO".DigitalInput14;
	Cyclic#1.P1_StoperSrobovania.IN.Centrovanie_VYSUNUTE_IS62 AT %IX."DI1.1_16DI".DigitalInput01;
	Cyclic#1.P1_StoperSrobovania.IN.Centrovanie_ZASUNUTE_IS63 AT %IX."DI1.1_16DI".DigitalInput02;
	Cyclic#1.P1_AkumulacnyStoper.IN.PritomnPaletky_IS45 AT %IX."DI1.1_16DI".DigitalInput03;
	Cyclic#1.P1_SpodnyStoper.IN.PritomnPaletky_IS64 AT %IX."DI1.1_16DI".DigitalInput04;
	Cyclic#1.P1_Robot.IN.SnimacVakua_S20 AT %IX."DI1.1_16DI".DigitalInput05;
	Cyclic#1.P1_Robot.IN.DokStanPritGrip_BusBary5H_IS77 AT %IX."DI1.1_16DI".DigitalInput06;
	Cyclic#1.P1_Robot.IN.DokStanPritGrip_BusBary45F_IS78 AT %IX."DI1.1_16DI".DigitalInput07;
	Cyclic#1.P1_Srobovanie.IN.SkrutkM4_Cist_BrzdaZatvoren_MS19 AT %IX."DI1.1_16DI".DigitalInput14;
	Cyclic#1.P1_Srobovanie.IN.SkrutkM4_Cist_BrzdaOtvorena_MS18 AT %IX."DI1.1_16DI".DigitalInput13;
	Cyclic#1.P1_Srobovanie.IN.SkrutkM4_Cist_SrobaPresla_IS48 AT %IX."DI1.1_16DI".DigitalInput12;
	Cyclic#1.P1_Srobovanie.IN.NastrelSrobM4_SrobaPresla_IS46 AT %IX."DI1.1_16DI".DigitalInput11;
	Cyclic#1.P1_Srobovanie.IN.ZasobSrobM4_ListaPLNA_OS6 AT %IX."DI1.1_16DI".DigitalInput10;
	Cyclic#1.P1_Srobovanie.IN.ZasobSrobM4_PRAZDNY_IS44 AT %IX."DI1.1_16DI".DigitalInput09;
	Cyclic#1.P1_Srobovanie.IN.SkrutkM4_SrobaPresla_IS47 AT %IX."DI1.1_16DI".DigitalInput15;
	Cyclic#1.P1_Srobovanie.IN.ZasobSrobK30_PRAZDNY_IS49 AT %IX."DI1.2_16DI".DigitalInput01;
	Cyclic#1.P1_Srobovanie.IN.ZasobSrobK30_ListaPLNA_OS7 AT %IX."DI1.2_16DI".DigitalInput02;
	Cyclic#1.P1_Srobovanie.IN.NastrelSrobK30_SrobaPresla_IS50 AT %IX."DI1.2_16DI".DigitalInput03;
	Cyclic#1.P1_Srobovanie.IN.SkrutkK30_Cist_SrobaPresla_IS52 AT %IX."DI1.2_16DI".DigitalInput04;
	Cyclic#1.P1_Srobovanie.IN.SkrutkK30_Cist_BrzdaOtvoren_MS21 AT %IX."DI1.2_16DI".DigitalInput05;
	Cyclic#1.P1_Srobovanie.IN.SkrutkK30_Cist_BrzdaZatvor_MS22 AT %IX."DI1.2_16DI".DigitalInput06;
	Cyclic#1.P1_Srobovanie.IN.SkrutkK30_SrobaPresla_IS51 AT %IX."DI1.2_16DI".DigitalInput07;
	Cyclic#1.P1_Srobovanie.IN.ZasobSrobM5_PRAZDNY_IS53 AT %IX."DI1.2_16DI".DigitalInput09;
	Cyclic#1.P1_Srobovanie.IN.ZasobSrobM5_ListaPLNA_OS8 AT %IX."DI1.2_16DI".DigitalInput10;
	Cyclic#1.P1_Srobovanie.IN.VibrolistaSrobM5_KONIEC_OS9 AT %IX."DI1.2_16DI".DigitalInput11;
	Cyclic#1.P1_Srobovanie.IN.VibrolistaSrobM5_ZACIATOK_OS10 AT %IX."DI1.2_16DI".DigitalInput12;
	Cyclic#1.P1_Srobovanie.IN.OddelSrobM5_SrobaNaVstupe_OS13 AT %IX."DI1.2_16DI".DigitalInput13;
	Cyclic#1.P1_Srobovanie.IN.OddelSrobM5_SrobaNaVystupe_OS14 AT %IX."DI1.2_16DI".DigitalInput14;
	Cyclic#1.P1_Srobovanie.IN.OddelSrobM5_OtocenyVPRED_MS37 AT %IX."DI1.2_16DI".DigitalInput15;
	Cyclic#1.P1_Srobovanie.IN.OddelSrobM5_OtocenyVZAD_MS38 AT %IX."DI1.2_16DI".DigitalInput16;
	Cyclic#1.P1_Srobovanie.IN.ManipulOsY_LimSnimacNEG_IS40 AT %IX."DI1.4_8DI".DigitalInput01;
	Cyclic#1.P1_Srobovanie.IN.ManipulOsY_LimSnimacPOS_IS41 AT %IX."DI1.4_8DI".DigitalInput02;
	Cyclic#1.P1_Srobovanie.IN.ManipulOsX_LimSnimacNEG_IS42 AT %IX."DI1.4_8DI".DigitalInput03;
	Cyclic#1.P1_Srobovanie.IN.ManipulOsX_LimSnimacPOS_IS43 AT %IX."DI1.4_8DI".DigitalInput04;
	Cyclic#1.P1_Srobovanie.IN.SkrutkK30_ZASUNUTY_MS20 AT %IX."DI1.4_8DI".DigitalInput05;
	Cyclic#1.P1_Srobovanie.IN.SkrutkM5_ZASUNUTY_MS39 AT %IX."DI1.4_8DI".DigitalInput06;
	Cyclic#1.P1_Srobovanie.IN.SkrutkM4_ZASUNUTY_MS17 AT %IX."DI1.4_8DI".DigitalInput07;
	Cyclic#1.Safety.OUT.P1_ZamkniZamok_PredneDvere AT %QX."DM1.1_16DI/DO".DigitalOutput01;
	Cyclic#1.Safety.IN.P1_PredneDvere_PritomPetlice AT %IX."DM1.1_16DI/DO".DigitalInput02;
	Cyclic#1.Safety.OUT.P1_ZamkniZamok_ZadneDverePS AT %QX."DM1.1_16DI/DO".DigitalOutput03;
	Cyclic#1.Safety.IN.P1_ZadneDverePS_PritomPetlice AT %IX."DM1.1_16DI/DO".DigitalInput04;
	Cyclic#1.Safety.OUT.P1_ZamkniZamok_ZadneDvereLS AT %QX."DM1.1_16DI/DO".DigitalOutput05;
	Cyclic#1.Safety.IN.P1_ZadneDvereLS_PritomPetlice AT %IX."DM1.1_16DI/DO".DigitalInput06;
	Cyclic#1.P2_Pracovisko.STAV.ModulDS22_OK AT %IX."DS2_2".ModuleOk;
	Cyclic#1.P2_Pracovisko.STAV.ModulDS21_OK AT %IX."DS2_1".ModuleOk;
	Cyclic#1.P1_Pracovisko.IN.PrivodVzduchu_SnimacTlaku_S18 AT %QX."SL1_SafetyMaster".BOOL116;
	Cyclic#1.Safety.IN.P1_ZonaBunky_RESET AT %QX."SL1_SafetyMaster".BOOL117;
	Cyclic#1.Safety.IN.P1_ZonaVytahu_RESET AT %QX."SL1_SafetyMaster".BOOL118;
	Cyclic#1.Safety.IN.P1_SV_Ventil1_ZonaBunka_B9 AT %QX."SL1_SafetyMaster".BOOL119;
	Cyclic#1.Safety.IN.P1_SV_Ventil2_ZonaBunka_B10 AT %QX."SL1_SafetyMaster".BOOL120;
	Cyclic#1.Safety.IN.P1_SV_ZonaBunka AT %QX."SL1_SafetyMaster".BOOL121;
	Cyclic#1.Safety.IN.P1_SV_ZonaCS AT %QX."SL1_SafetyMaster".BOOL122;
	Cyclic#1.Safety.IN.P1_SV_ZonaVytah AT %QX."SL1_SafetyMaster".BOOL123;
	Cyclic#1.Safety.IN.P1_ReleaseKartySO_AB15 AT %QX."SL1_SafetyMaster".BOOL124;
	Cyclic#1.Safety.STAV.P1_Panel_TlacitkoCS_AKTIVNE AT %IX."SL1_SafetyMaster".BOOL018;
	Cyclic#1.Safety.STAV.P1_Robot_TlacitkoCS_AKTIVNE AT %IX."SL1_SafetyMaster".BOOL019;
	Cyclic#1.Safety.STAV.P1_Skrina_TlacitkoCS_AKTIVNE AT %IX."SL1_SafetyMaster".BOOL020;
	Cyclic#1.Safety.STAV.P1_VstupBunky_Bariera_AKTIVNA AT %IX."SL1_SafetyMaster".BOOL021;
	Cyclic#1.Safety.STAV.P1_VystupTunela_Bariera_AKTIVNA AT %IX."SL1_SafetyMaster".BOOL022;
	Cyclic#1.Safety.STAV.P1_Vytah_Bariera_AKTIVNA AT %IX."SL1_SafetyMaster".BOOL023;
	Cyclic#1.Safety.STAV.P1_VyblokovanieSafety_AKTIVNE AT %IX."SL1_SafetyMaster".BOOL024;
	Cyclic#1.Safety.STAV.P1_ZamkyBunky_AKTIVNE AT %IX."SL1_SafetyMaster".BOOL025;
	Cyclic#1.Safety.STAV.P1_ZonaBunky_AKTIVNA AT %IX."SL1_SafetyMaster".BOOL026;
	Cyclic#1.Safety.STAV.P1_ZonaVytahu_AKTIVNA AT %IX."SL1_SafetyMaster".BOOL027;
	Cyclic#1.Safety.STAV.P1_SnimacVytahu_AKTIVNY AT %IX."SL1_SafetyMaster".BOOL028;
	Cyclic#1.P1_Pracovisko.OUT.VT4_OUT1 AT %QB."VentilovyTerminal_VT4".OUT1_I2200_S01Out;
	Cyclic#1.P1_Pracovisko.OUT.VT4_OUT2 AT %QB."VentilovyTerminal_VT4".OUT2_I2200_S02Out;
	Cyclic#1.P1_Pracovisko.OUT.VT4_OUT3 AT %QB."VentilovyTerminal_VT4".OUT3_I2200_S03Out;
	Cyclic#1.P1_Pracovisko.OUT.VT4_OUT4 AT %QB."VentilovyTerminal_VT4".OUT4_I2200_S04Out;
	Cyclic#1.P1_Pracovisko.OUT.VT5_OUT1 AT %QB."VentilovyTerminal_VT5".OUT1_I2200_S01Out;
	Cyclic#1.P1_Pracovisko.OUT.VT5_OUT2 AT %QB."VentilovyTerminal_VT5".OUT2_I2200_S02Out;
	Cyclic#1.P1_Pracovisko.OUT.VT5_OUT3 AT %QB."VentilovyTerminal_VT5".OUT3_I2200_S03Out;
	Cyclic#1.P1_Pracovisko.OUT.VT5_OUT4 AT %QB."VentilovyTerminal_VT5".OUT4_I2200_S04Out;
	Cyclic#1.Safety.IN.P1_Vytah_Zdvih_BUSY AT %QX."SL1_SafetyMaster".BOOL125;
	Cyclic#1.Safety.IN.P2_ZaklTesnenia_Vysuvanie_BUSY AT %QX."SL1_SafetyMaster".BOOL126;
	Cyclic#1.Safety.IN.P2_ZaklTesnenia_Zasuvanie_BUSY AT %QX."SL1_SafetyMaster".BOOL127;
	Cyclic#1.Safety.IN.P2_ZaklTesnenia_Zdvih_BUSY AT %QX."SL1_SafetyMaster".BOOL128;
	Cyclic#1.::P2_Pracovisko.STAV.ModulDS23_OK AT %IX."DS2_3".ModuleOk;
	Cyclic#1.P1_Srobovanie.IN.SkrutkK30_VysunutieHrotu_IOlink AT %IW."DS1_2".InputData01_1;
	Cyclic#1.P1_Srobovanie.IN.SkrutkM4_VysunutieHrotu_IOlink AT %IW."DS1_2".InputData02_1;
	Cyclic#1.P1_Pracovisko.STAV.KOM_Robot_OK AT %IX."R1_IRB120".ModuleOk;
	Cyclic#1.P1_Robot.KOM_IN.Profinet_PLC_INPUTS[0] AT %IB."R1_IRB120".Module001_Input_0;
	Cyclic#1.P1_Robot.KOM_IN.Profinet_PLC_INPUTS[1] AT %IB."R1_IRB120".Module001_Input_1;
	Cyclic#1.P1_Robot.KOM_IN.Profinet_PLC_INPUTS[2] AT %IB."R1_IRB120".Module001_Input_2;
	Cyclic#1.P1_Robot.KOM_IN.Profinet_PLC_INPUTS[3] AT %IB."R1_IRB120".Module001_Input_3;
	Cyclic#1.P1_Robot.KOM_IN.Profinet_PLC_INPUTS[4] AT %IB."R1_IRB120".Module001_Input_4;
	Cyclic#1.P1_Robot.KOM_IN.Profinet_PLC_INPUTS[5] AT %IB."R1_IRB120".Module001_Input_5;
	Cyclic#1.P1_Robot.KOM_IN.Profinet_PLC_INPUTS[6] AT %IB."R1_IRB120".Module001_Input_6;
	Cyclic#1.P1_Robot.KOM_IN.Profinet_PLC_INPUTS[7] AT %IB."R1_IRB120".Module001_Input_7;
	Cyclic#1.P1_Robot.KOM_IN.Profinet_PLC_INPUTS[8] AT %IB."R1_IRB120".Module001_Input_8;
	Cyclic#1.P1_Robot.KOM_IN.Profinet_PLC_INPUTS[9] AT %IB."R1_IRB120".Module001_Input_9;
	Cyclic#1.P1_Robot.KOM_IN.Profinet_PLC_INPUTS[10] AT %IB."R1_IRB120".Module001_Input_10;
	Cyclic#1.P1_Robot.KOM_IN.Profinet_PLC_INPUTS[11] AT %IB."R1_IRB120".Module001_Input_11;
	Cyclic#1.P1_Robot.KOM_IN.Profinet_PLC_INPUTS[12] AT %IB."R1_IRB120".Module001_Input_12;
	Cyclic#1.P1_Robot.KOM_IN.Profinet_PLC_INPUTS[13] AT %IB."R1_IRB120".Module001_Input_13;
	Cyclic#1.P1_Robot.KOM_IN.Profinet_PLC_INPUTS[14] AT %IB."R1_IRB120".Module001_Input_14;
	Cyclic#1.P1_Robot.KOM_IN.Profinet_PLC_INPUTS[15] AT %IB."R1_IRB120".Module001_Input_15;
	Cyclic#1.P1_Robot.KOM_IN.Profinet_PLC_INPUTS[16] AT %IB."R1_IRB120".Module001_Input_16;
	Cyclic#1.P1_Robot.KOM_IN.Profinet_PLC_INPUTS[17] AT %IB."R1_IRB120".Module001_Input_17;
	Cyclic#1.P1_Robot.KOM_IN.Profinet_PLC_INPUTS[18] AT %IB."R1_IRB120".Module001_Input_18;
	Cyclic#1.P1_Robot.KOM_IN.Profinet_PLC_INPUTS[19] AT %IB."R1_IRB120".Module001_Input_19;
	Cyclic#1.P1_Robot.KOM_IN.Profinet_PLC_INPUTS[20] AT %IB."R1_IRB120".Module001_Input_20;
	Cyclic#1.P1_Robot.KOM_IN.Profinet_PLC_INPUTS[21] AT %IB."R1_IRB120".Module001_Input_21;
	Cyclic#1.P1_Robot.KOM_IN.Profinet_PLC_INPUTS[22] AT %IB."R1_IRB120".Module001_Input_22;
	Cyclic#1.P1_Robot.KOM_IN.Profinet_PLC_INPUTS[23] AT %IB."R1_IRB120".Module001_Input_23;
	Cyclic#1.P1_Robot.KOM_IN.Profinet_PLC_INPUTS[24] AT %IB."R1_IRB120".Module001_Input_24;
	Cyclic#1.P1_Robot.KOM_IN.Profinet_PLC_INPUTS[25] AT %IB."R1_IRB120".Module001_Input_25;
	Cyclic#1.P1_Robot.KOM_IN.Profinet_PLC_INPUTS[63] AT %IB."R1_IRB120".Module001_Input_63;
	Cyclic#1.P1_Robot.KOM_IN.Profinet_PLC_INPUTS[62] AT %IB."R1_IRB120".Module001_Input_62;
	Cyclic#1.P1_Robot.KOM_IN.Profinet_PLC_INPUTS[61] AT %IB."R1_IRB120".Module001_Input_61;
	Cyclic#1.P1_Robot.KOM_IN.Profinet_PLC_INPUTS[60] AT %IB."R1_IRB120".Module001_Input_60;
	Cyclic#1.P1_Robot.KOM_IN.Profinet_PLC_INPUTS[59] AT %IB."R1_IRB120".Module001_Input_59;
	Cyclic#1.P1_Robot.KOM_IN.Profinet_PLC_INPUTS[58] AT %IB."R1_IRB120".Module001_Input_58;
	Cyclic#1.P1_Robot.KOM_IN.Profinet_PLC_INPUTS[57] AT %IB."R1_IRB120".Module001_Input_57;
	Cyclic#1.P1_Robot.KOM_IN.Profinet_PLC_INPUTS[56] AT %IB."R1_IRB120".Module001_Input_56;
	Cyclic#1.P1_Robot.KOM_IN.Profinet_PLC_INPUTS[55] AT %IB."R1_IRB120".Module001_Input_55;
	Cyclic#1.P1_Robot.KOM_IN.Profinet_PLC_INPUTS[54] AT %IB."R1_IRB120".Module001_Input_54;
	Cyclic#1.P1_Robot.KOM_IN.Profinet_PLC_INPUTS[53] AT %IB."R1_IRB120".Module001_Input_53;
	Cyclic#1.P1_Robot.KOM_IN.Profinet_PLC_INPUTS[52] AT %IB."R1_IRB120".Module001_Input_52;
	Cyclic#1.P1_Robot.KOM_IN.Profinet_PLC_INPUTS[51] AT %IB."R1_IRB120".Module001_Input_51;
	Cyclic#1.P1_Robot.KOM_IN.Profinet_PLC_INPUTS[50] AT %IB."R1_IRB120".Module001_Input_50;
	Cyclic#1.P1_Robot.KOM_IN.Profinet_PLC_INPUTS[49] AT %IB."R1_IRB120".Module001_Input_49;
	Cyclic#1.P1_Robot.KOM_IN.Profinet_PLC_INPUTS[48] AT %IB."R1_IRB120".Module001_Input_48;
	Cyclic#1.P1_Robot.KOM_IN.Profinet_PLC_INPUTS[47] AT %IB."R1_IRB120".Module001_Input_47;
	Cyclic#1.P1_Robot.KOM_IN.Profinet_PLC_INPUTS[46] AT %IB."R1_IRB120".Module001_Input_46;
	Cyclic#1.P1_Robot.KOM_IN.Profinet_PLC_INPUTS[45] AT %IB."R1_IRB120".Module001_Input_45;
	Cyclic#1.P1_Robot.KOM_IN.Profinet_PLC_INPUTS[44] AT %IB."R1_IRB120".Module001_Input_44;
	Cyclic#1.P1_Robot.KOM_IN.Profinet_PLC_INPUTS[43] AT %IB."R1_IRB120".Module001_Input_43;
	Cyclic#1.P1_Robot.KOM_IN.Profinet_PLC_INPUTS[42] AT %IB."R1_IRB120".Module001_Input_42;
	Cyclic#1.P1_Robot.KOM_IN.Profinet_PLC_INPUTS[41] AT %IB."R1_IRB120".Module001_Input_41;
	Cyclic#1.P1_Robot.KOM_IN.Profinet_PLC_INPUTS[40] AT %IB."R1_IRB120".Module001_Input_40;
	Cyclic#1.P1_Robot.KOM_IN.Profinet_PLC_INPUTS[39] AT %IB."R1_IRB120".Module001_Input_39;
	Cyclic#1.P1_Robot.KOM_IN.Profinet_PLC_INPUTS[38] AT %IB."R1_IRB120".Module001_Input_38;
	Cyclic#1.P1_Robot.KOM_IN.Profinet_PLC_INPUTS[37] AT %IB."R1_IRB120".Module001_Input_37;
	Cyclic#1.P1_Robot.KOM_IN.Profinet_PLC_INPUTS[36] AT %IB."R1_IRB120".Module001_Input_36;
	Cyclic#1.P1_Robot.KOM_IN.Profinet_PLC_INPUTS[35] AT %IB."R1_IRB120".Module001_Input_35;
	Cyclic#1.P1_Robot.KOM_IN.Profinet_PLC_INPUTS[34] AT %IB."R1_IRB120".Module001_Input_34;
	Cyclic#1.P1_Robot.KOM_IN.Profinet_PLC_INPUTS[33] AT %IB."R1_IRB120".Module001_Input_33;
	Cyclic#1.P1_Robot.KOM_IN.Profinet_PLC_INPUTS[32] AT %IB."R1_IRB120".Module001_Input_32;
	Cyclic#1.P1_Robot.KOM_IN.Profinet_PLC_INPUTS[31] AT %IB."R1_IRB120".Module001_Input_31;
	Cyclic#1.P1_Robot.KOM_IN.Profinet_PLC_INPUTS[30] AT %IB."R1_IRB120".Module001_Input_30;
	Cyclic#1.P1_Robot.KOM_IN.Profinet_PLC_INPUTS[29] AT %IB."R1_IRB120".Module001_Input_29;
	Cyclic#1.P1_Robot.KOM_IN.Profinet_PLC_INPUTS[28] AT %IB."R1_IRB120".Module001_Input_28;
	Cyclic#1.P1_Robot.KOM_IN.Profinet_PLC_INPUTS[27] AT %IB."R1_IRB120".Module001_Input_27;
	Cyclic#1.P1_Robot.KOM_IN.Profinet_PLC_INPUTS[26] AT %IB."R1_IRB120".Module001_Input_26;
	Cyclic#1.P1_Robot.KOM_OUT.Profinet_PLC_OUTPUTS[0] AT %QB."R1_IRB120".Module002_Output_0;
	Cyclic#1.P1_Robot.KOM_OUT.Profinet_PLC_OUTPUTS[1] AT %QB."R1_IRB120".Module002_Output_1;
	Cyclic#1.P1_Robot.KOM_OUT.Profinet_PLC_OUTPUTS[2] AT %QB."R1_IRB120".Module002_Output_2;
	Cyclic#1.P1_Robot.KOM_OUT.Profinet_PLC_OUTPUTS[3] AT %QB."R1_IRB120".Module002_Output_3;
	Cyclic#1.P1_Robot.KOM_OUT.Profinet_PLC_OUTPUTS[4] AT %QB."R1_IRB120".Module002_Output_4;
	Cyclic#1.P1_Robot.KOM_OUT.Profinet_PLC_OUTPUTS[5] AT %QB."R1_IRB120".Module002_Output_5;
	Cyclic#1.P1_Robot.KOM_OUT.Profinet_PLC_OUTPUTS[6] AT %QB."R1_IRB120".Module002_Output_6;
	Cyclic#1.P1_Robot.KOM_OUT.Profinet_PLC_OUTPUTS[7] AT %QB."R1_IRB120".Module002_Output_7;
	Cyclic#1.P1_Robot.KOM_OUT.Profinet_PLC_OUTPUTS[8] AT %QB."R1_IRB120".Module002_Output_8;
	Cyclic#1.P1_Robot.KOM_OUT.Profinet_PLC_OUTPUTS[9] AT %QB."R1_IRB120".Module002_Output_9;
	Cyclic#1.P1_Robot.KOM_OUT.Profinet_PLC_OUTPUTS[10] AT %QB."R1_IRB120".Module002_Output_10;
	Cyclic#1.P1_Robot.KOM_OUT.Profinet_PLC_OUTPUTS[11] AT %QB."R1_IRB120".Module002_Output_11;
	Cyclic#1.P1_Robot.KOM_OUT.Profinet_PLC_OUTPUTS[12] AT %QB."R1_IRB120".Module002_Output_12;
	Cyclic#1.P1_Robot.KOM_OUT.Profinet_PLC_OUTPUTS[13] AT %QB."R1_IRB120".Module002_Output_13;
	Cyclic#1.P1_Robot.KOM_OUT.Profinet_PLC_OUTPUTS[14] AT %QB."R1_IRB120".Module002_Output_14;
	Cyclic#1.P1_Robot.KOM_OUT.Profinet_PLC_OUTPUTS[15] AT %QB."R1_IRB120".Module002_Output_15;
	Cyclic#1.P1_Robot.KOM_OUT.Profinet_PLC_OUTPUTS[16] AT %QB."R1_IRB120".Module002_Output_16;
	Cyclic#1.P1_Robot.KOM_OUT.Profinet_PLC_OUTPUTS[17] AT %QB."R1_IRB120".Module002_Output_17;
	Cyclic#1.P1_Robot.KOM_OUT.Profinet_PLC_OUTPUTS[18] AT %QB."R1_IRB120".Module002_Output_18;
	Cyclic#1.P1_Robot.KOM_OUT.Profinet_PLC_OUTPUTS[19] AT %QB."R1_IRB120".Module002_Output_19;
	Cyclic#1.P1_Robot.KOM_OUT.Profinet_PLC_OUTPUTS[20] AT %QB."R1_IRB120".Module002_Output_20;
	Cyclic#1.P1_Robot.KOM_OUT.Profinet_PLC_OUTPUTS[21] AT %QB."R1_IRB120".Module002_Output_21;
	Cyclic#1.P1_Robot.KOM_OUT.Profinet_PLC_OUTPUTS[22] AT %QB."R1_IRB120".Module002_Output_22;
	Cyclic#1.P1_Robot.KOM_OUT.Profinet_PLC_OUTPUTS[23] AT %QB."R1_IRB120".Module002_Output_23;
	Cyclic#1.P1_Robot.KOM_OUT.Profinet_PLC_OUTPUTS[24] AT %QB."R1_IRB120".Module002_Output_24;
	Cyclic#1.P1_Robot.KOM_OUT.Profinet_PLC_OUTPUTS[25] AT %QB."R1_IRB120".Module002_Output_25;
	Cyclic#1.P1_Robot.KOM_OUT.Profinet_PLC_OUTPUTS[26] AT %QB."R1_IRB120".Module002_Output_26;
	Cyclic#1.P1_Robot.KOM_OUT.Profinet_PLC_OUTPUTS[27] AT %QB."R1_IRB120".Module002_Output_27;
	Cyclic#1.P1_Robot.KOM_OUT.Profinet_PLC_OUTPUTS[28] AT %QB."R1_IRB120".Module002_Output_28;
	Cyclic#1.P1_Robot.KOM_OUT.Profinet_PLC_OUTPUTS[29] AT %QB."R1_IRB120".Module002_Output_29;
	Cyclic#1.P1_Robot.KOM_OUT.Profinet_PLC_OUTPUTS[30] AT %QB."R1_IRB120".Module002_Output_30;
	Cyclic#1.P1_Robot.KOM_OUT.Profinet_PLC_OUTPUTS[31] AT %QB."R1_IRB120".Module002_Output_31;
	Cyclic#1.P1_Robot.KOM_OUT.Profinet_PLC_OUTPUTS[32] AT %QB."R1_IRB120".Module002_Output_32;
	Cyclic#1.P1_Robot.KOM_OUT.Profinet_PLC_OUTPUTS[33] AT %QB."R1_IRB120".Module002_Output_33;
	Cyclic#1.P1_Robot.KOM_OUT.Profinet_PLC_OUTPUTS[34] AT %QB."R1_IRB120".Module002_Output_34;
	Cyclic#1.P1_Robot.KOM_OUT.Profinet_PLC_OUTPUTS[35] AT %QB."R1_IRB120".Module002_Output_35;
	Cyclic#1.P1_Robot.KOM_OUT.Profinet_PLC_OUTPUTS[36] AT %QB."R1_IRB120".Module002_Output_36;
	Cyclic#1.P1_Robot.KOM_OUT.Profinet_PLC_OUTPUTS[37] AT %QB."R1_IRB120".Module002_Output_37;
	Cyclic#1.P1_Robot.KOM_OUT.Profinet_PLC_OUTPUTS[38] AT %QB."R1_IRB120".Module002_Output_38;
	Cyclic#1.P1_Robot.KOM_OUT.Profinet_PLC_OUTPUTS[39] AT %QB."R1_IRB120".Module002_Output_39;
	Cyclic#1.P1_Robot.KOM_OUT.Profinet_PLC_OUTPUTS[40] AT %QB."R1_IRB120".Module002_Output_40;
	Cyclic#1.P1_Robot.KOM_OUT.Profinet_PLC_OUTPUTS[41] AT %QB."R1_IRB120".Module002_Output_41;
	Cyclic#1.P1_Robot.KOM_OUT.Profinet_PLC_OUTPUTS[42] AT %QB."R1_IRB120".Module002_Output_42;
	Cyclic#1.P1_Robot.KOM_OUT.Profinet_PLC_OUTPUTS[43] AT %QB."R1_IRB120".Module002_Output_43;
	Cyclic#1.P1_Robot.KOM_OUT.Profinet_PLC_OUTPUTS[44] AT %QB."R1_IRB120".Module002_Output_44;
	Cyclic#1.P1_Robot.KOM_OUT.Profinet_PLC_OUTPUTS[45] AT %QB."R1_IRB120".Module002_Output_45;
	Cyclic#1.P1_Robot.KOM_OUT.Profinet_PLC_OUTPUTS[46] AT %QB."R1_IRB120".Module002_Output_46;
	Cyclic#1.P1_Robot.KOM_OUT.Profinet_PLC_OUTPUTS[47] AT %QB."R1_IRB120".Module002_Output_47;
	Cyclic#1.P1_Robot.KOM_OUT.Profinet_PLC_OUTPUTS[48] AT %QB."R1_IRB120".Module002_Output_48;
	Cyclic#1.P1_Robot.KOM_OUT.Profinet_PLC_OUTPUTS[49] AT %QB."R1_IRB120".Module002_Output_49;
	Cyclic#1.P1_Robot.KOM_OUT.Profinet_PLC_OUTPUTS[50] AT %QB."R1_IRB120".Module002_Output_50;
	Cyclic#1.P1_Robot.KOM_OUT.Profinet_PLC_OUTPUTS[51] AT %QB."R1_IRB120".Module002_Output_51;
	Cyclic#1.P1_Robot.KOM_OUT.Profinet_PLC_OUTPUTS[52] AT %QB."R1_IRB120".Module002_Output_52;
	Cyclic#1.P1_Robot.KOM_OUT.Profinet_PLC_OUTPUTS[53] AT %QB."R1_IRB120".Module002_Output_53;
	Cyclic#1.P1_Robot.KOM_OUT.Profinet_PLC_OUTPUTS[54] AT %QB."R1_IRB120".Module002_Output_54;
	Cyclic#1.P1_Robot.KOM_OUT.Profinet_PLC_OUTPUTS[55] AT %QB."R1_IRB120".Module002_Output_55;
	Cyclic#1.P1_Robot.KOM_OUT.Profinet_PLC_OUTPUTS[56] AT %QB."R1_IRB120".Module002_Output_56;
	Cyclic#1.P1_Robot.KOM_OUT.Profinet_PLC_OUTPUTS[57] AT %QB."R1_IRB120".Module002_Output_57;
	Cyclic#1.P1_Robot.KOM_OUT.Profinet_PLC_OUTPUTS[58] AT %QB."R1_IRB120".Module002_Output_58;
	Cyclic#1.P1_Robot.KOM_OUT.Profinet_PLC_OUTPUTS[59] AT %QB."R1_IRB120".Module002_Output_59;
	Cyclic#1.P1_Robot.KOM_OUT.Profinet_PLC_OUTPUTS[60] AT %QB."R1_IRB120".Module002_Output_60;
	Cyclic#1.P1_Robot.KOM_OUT.Profinet_PLC_OUTPUTS[61] AT %QB."R1_IRB120".Module002_Output_61;
	Cyclic#1.P1_Robot.KOM_OUT.Profinet_PLC_OUTPUTS[62] AT %QB."R1_IRB120".Module002_Output_62;
	Cyclic#1.P1_Robot.KOM_OUT.Profinet_PLC_OUTPUTS[63] AT %QB."R1_IRB120".Module002_Output_63;
	Cyclic#1.P2_Robot.KOM_IN.Profinet_PLC_INPUTS[0] AT %IB."R2_IRB1200".Module001_Input_0;
	Cyclic#1.P2_Robot.KOM_OUT.Profinet_PLC_OUTPUTS[0] AT %QB."R2_IRB1200".Module002_Output_0;
	Cyclic#1.P2_Robot.KOM_IN.Profinet_PLC_INPUTS[1] AT %IB."R2_IRB1200".Module001_Input_1;
	Cyclic#1.P2_Robot.KOM_IN.Profinet_PLC_INPUTS[2] AT %IB."R2_IRB1200".Module001_Input_2;
	Cyclic#1.P2_Robot.KOM_IN.Profinet_PLC_INPUTS[3] AT %IB."R2_IRB1200".Module001_Input_3;
	Cyclic#1.P2_Robot.KOM_IN.Profinet_PLC_INPUTS[4] AT %IB."R2_IRB1200".Module001_Input_4;
	Cyclic#1.P2_Robot.KOM_IN.Profinet_PLC_INPUTS[5] AT %IB."R2_IRB1200".Module001_Input_5;
	Cyclic#1.P2_Robot.KOM_IN.Profinet_PLC_INPUTS[6] AT %IB."R2_IRB1200".Module001_Input_6;
	Cyclic#1.P2_Robot.KOM_IN.Profinet_PLC_INPUTS[7] AT %IB."R2_IRB1200".Module001_Input_7;
	Cyclic#1.P2_Robot.KOM_IN.Profinet_PLC_INPUTS[8] AT %IB."R2_IRB1200".Module001_Input_8;
	Cyclic#1.P2_Robot.KOM_IN.Profinet_PLC_INPUTS[9] AT %IB."R2_IRB1200".Module001_Input_9;
	Cyclic#1.P2_Robot.KOM_IN.Profinet_PLC_INPUTS[10] AT %IB."R2_IRB1200".Module001_Input_10;
	Cyclic#1.P2_Robot.KOM_IN.Profinet_PLC_INPUTS[11] AT %IB."R2_IRB1200".Module001_Input_11;
	Cyclic#1.P2_Robot.KOM_IN.Profinet_PLC_INPUTS[12] AT %IB."R2_IRB1200".Module001_Input_12;
	Cyclic#1.P2_Robot.KOM_IN.Profinet_PLC_INPUTS[13] AT %IB."R2_IRB1200".Module001_Input_13;
	Cyclic#1.P2_Robot.KOM_IN.Profinet_PLC_INPUTS[14] AT %IB."R2_IRB1200".Module001_Input_14;
	Cyclic#1.P2_Robot.KOM_IN.Profinet_PLC_INPUTS[15] AT %IB."R2_IRB1200".Module001_Input_15;
	Cyclic#1.P2_Robot.KOM_IN.Profinet_PLC_INPUTS[16] AT %IB."R2_IRB1200".Module001_Input_16;
	Cyclic#1.P2_Robot.KOM_IN.Profinet_PLC_INPUTS[17] AT %IB."R2_IRB1200".Module001_Input_17;
	Cyclic#1.P2_Robot.KOM_IN.Profinet_PLC_INPUTS[18] AT %IB."R2_IRB1200".Module001_Input_18;
	Cyclic#1.P2_Robot.KOM_IN.Profinet_PLC_INPUTS[19] AT %IB."R2_IRB1200".Module001_Input_19;
	Cyclic#1.P2_Robot.KOM_IN.Profinet_PLC_INPUTS[20] AT %IB."R2_IRB1200".Module001_Input_20;
	Cyclic#1.P2_Robot.KOM_IN.Profinet_PLC_INPUTS[21] AT %IB."R2_IRB1200".Module001_Input_21;
	Cyclic#1.P2_Robot.KOM_IN.Profinet_PLC_INPUTS[22] AT %IB."R2_IRB1200".Module001_Input_22;
	Cyclic#1.P2_Robot.KOM_IN.Profinet_PLC_INPUTS[23] AT %IB."R2_IRB1200".Module001_Input_23;
	Cyclic#1.P2_Robot.KOM_IN.Profinet_PLC_INPUTS[24] AT %IB."R2_IRB1200".Module001_Input_24;
	Cyclic#1.P2_Robot.KOM_IN.Profinet_PLC_INPUTS[25] AT %IB."R2_IRB1200".Module001_Input_25;
	Cyclic#1.P2_Robot.KOM_IN.Profinet_PLC_INPUTS[26] AT %IB."R2_IRB1200".Module001_Input_26;
	Cyclic#1.P2_Robot.KOM_IN.Profinet_PLC_INPUTS[27] AT %IB."R2_IRB1200".Module001_Input_27;
	Cyclic#1.P2_Robot.KOM_IN.Profinet_PLC_INPUTS[28] AT %IB."R2_IRB1200".Module001_Input_28;
	Cyclic#1.P2_Robot.KOM_IN.Profinet_PLC_INPUTS[29] AT %IB."R2_IRB1200".Module001_Input_29;
	Cyclic#1.P2_Robot.KOM_IN.Profinet_PLC_INPUTS[30] AT %IB."R2_IRB1200".Module001_Input_30;
	Cyclic#1.P2_Robot.KOM_IN.Profinet_PLC_INPUTS[31] AT %IB."R2_IRB1200".Module001_Input_31;
	Cyclic#1.P2_Robot.KOM_IN.Profinet_PLC_INPUTS[32] AT %IB."R2_IRB1200".Module001_Input_32;
	Cyclic#1.P2_Robot.KOM_IN.Profinet_PLC_INPUTS[33] AT %IB."R2_IRB1200".Module001_Input_33;
	Cyclic#1.P2_Robot.KOM_IN.Profinet_PLC_INPUTS[34] AT %IB."R2_IRB1200".Module001_Input_34;
	Cyclic#1.P2_Robot.KOM_IN.Profinet_PLC_INPUTS[35] AT %IB."R2_IRB1200".Module001_Input_35;
	Cyclic#1.P2_Robot.KOM_IN.Profinet_PLC_INPUTS[36] AT %IB."R2_IRB1200".Module001_Input_36;
	Cyclic#1.P2_Robot.KOM_IN.Profinet_PLC_INPUTS[37] AT %IB."R2_IRB1200".Module001_Input_37;
	Cyclic#1.P2_Robot.KOM_IN.Profinet_PLC_INPUTS[38] AT %IB."R2_IRB1200".Module001_Input_38;
	Cyclic#1.P2_Robot.KOM_IN.Profinet_PLC_INPUTS[39] AT %IB."R2_IRB1200".Module001_Input_39;
	Cyclic#1.P2_Robot.KOM_IN.Profinet_PLC_INPUTS[40] AT %IB."R2_IRB1200".Module001_Input_40;
	Cyclic#1.P2_Robot.KOM_IN.Profinet_PLC_INPUTS[41] AT %IB."R2_IRB1200".Module001_Input_41;
	Cyclic#1.P2_Robot.KOM_IN.Profinet_PLC_INPUTS[42] AT %IB."R2_IRB1200".Module001_Input_42;
	Cyclic#1.P2_Robot.KOM_IN.Profinet_PLC_INPUTS[43] AT %IB."R2_IRB1200".Module001_Input_43;
	Cyclic#1.P2_Robot.KOM_IN.Profinet_PLC_INPUTS[44] AT %IB."R2_IRB1200".Module001_Input_44;
	Cyclic#1.P2_Robot.KOM_IN.Profinet_PLC_INPUTS[45] AT %IB."R2_IRB1200".Module001_Input_45;
	Cyclic#1.P2_Robot.KOM_IN.Profinet_PLC_INPUTS[46] AT %IB."R2_IRB1200".Module001_Input_46;
	Cyclic#1.P2_Robot.KOM_IN.Profinet_PLC_INPUTS[47] AT %IB."R2_IRB1200".Module001_Input_47;
	Cyclic#1.P2_Robot.KOM_IN.Profinet_PLC_INPUTS[48] AT %IB."R2_IRB1200".Module001_Input_48;
	Cyclic#1.P2_Robot.KOM_IN.Profinet_PLC_INPUTS[49] AT %IB."R2_IRB1200".Module001_Input_49;
	Cyclic#1.P2_Robot.KOM_IN.Profinet_PLC_INPUTS[50] AT %IB."R2_IRB1200".Module001_Input_50;
	Cyclic#1.P2_Robot.KOM_IN.Profinet_PLC_INPUTS[51] AT %IB."R2_IRB1200".Module001_Input_51;
	Cyclic#1.P2_Robot.KOM_IN.Profinet_PLC_INPUTS[52] AT %IB."R2_IRB1200".Module001_Input_52;
	Cyclic#1.P2_Robot.KOM_IN.Profinet_PLC_INPUTS[53] AT %IB."R2_IRB1200".Module001_Input_53;
	Cyclic#1.P2_Robot.KOM_IN.Profinet_PLC_INPUTS[54] AT %IB."R2_IRB1200".Module001_Input_54;
	Cyclic#1.P2_Robot.KOM_IN.Profinet_PLC_INPUTS[55] AT %IB."R2_IRB1200".Module001_Input_55;
	Cyclic#1.P2_Robot.KOM_IN.Profinet_PLC_INPUTS[56] AT %IB."R2_IRB1200".Module001_Input_56;
	Cyclic#1.P2_Robot.KOM_IN.Profinet_PLC_INPUTS[57] AT %IB."R2_IRB1200".Module001_Input_57;
	Cyclic#1.P2_Robot.KOM_IN.Profinet_PLC_INPUTS[58] AT %IB."R2_IRB1200".Module001_Input_58;
	Cyclic#1.P2_Robot.KOM_IN.Profinet_PLC_INPUTS[59] AT %IB."R2_IRB1200".Module001_Input_59;
	Cyclic#1.P2_Robot.KOM_IN.Profinet_PLC_INPUTS[60] AT %IB."R2_IRB1200".Module001_Input_60;
	Cyclic#1.P2_Robot.KOM_IN.Profinet_PLC_INPUTS[61] AT %IB."R2_IRB1200".Module001_Input_61;
	Cyclic#1.P2_Robot.KOM_IN.Profinet_PLC_INPUTS[62] AT %IB."R2_IRB1200".Module001_Input_62;
	Cyclic#1.P2_Robot.KOM_IN.Profinet_PLC_INPUTS[63] AT %IB."R2_IRB1200".Module001_Input_63;
	Cyclic#1.P2_Robot.KOM_OUT.Profinet_PLC_OUTPUTS[1] AT %QB."R2_IRB1200".Module002_Output_1;
	Cyclic#1.P2_Robot.KOM_OUT.Profinet_PLC_OUTPUTS[2] AT %QB."R2_IRB1200".Module002_Output_2;
	Cyclic#1.P2_Robot.KOM_OUT.Profinet_PLC_OUTPUTS[3] AT %QB."R2_IRB1200".Module002_Output_3;
	Cyclic#1.P2_Robot.KOM_OUT.Profinet_PLC_OUTPUTS[4] AT %QB."R2_IRB1200".Module002_Output_4;
	Cyclic#1.P2_Robot.KOM_OUT.Profinet_PLC_OUTPUTS[5] AT %QB."R2_IRB1200".Module002_Output_5;
	Cyclic#1.P2_Robot.KOM_OUT.Profinet_PLC_OUTPUTS[6] AT %QB."R2_IRB1200".Module002_Output_6;
	Cyclic#1.P2_Robot.KOM_OUT.Profinet_PLC_OUTPUTS[7] AT %QB."R2_IRB1200".Module002_Output_7;
	Cyclic#1.P2_Robot.KOM_OUT.Profinet_PLC_OUTPUTS[8] AT %QB."R2_IRB1200".Module002_Output_8;
	Cyclic#1.P2_Robot.KOM_OUT.Profinet_PLC_OUTPUTS[9] AT %QB."R2_IRB1200".Module002_Output_9;
	Cyclic#1.P2_Robot.KOM_OUT.Profinet_PLC_OUTPUTS[10] AT %QB."R2_IRB1200".Module002_Output_10;
	Cyclic#1.P2_Robot.KOM_OUT.Profinet_PLC_OUTPUTS[11] AT %QB."R2_IRB1200".Module002_Output_11;
	Cyclic#1.P2_Robot.KOM_OUT.Profinet_PLC_OUTPUTS[12] AT %QB."R2_IRB1200".Module002_Output_12;
	Cyclic#1.P2_Robot.KOM_OUT.Profinet_PLC_OUTPUTS[13] AT %QB."R2_IRB1200".Module002_Output_13;
	Cyclic#1.P2_Robot.KOM_OUT.Profinet_PLC_OUTPUTS[14] AT %QB."R2_IRB1200".Module002_Output_14;
	Cyclic#1.P2_Robot.KOM_OUT.Profinet_PLC_OUTPUTS[15] AT %QB."R2_IRB1200".Module002_Output_15;
	Cyclic#1.P2_Robot.KOM_OUT.Profinet_PLC_OUTPUTS[16] AT %QB."R2_IRB1200".Module002_Output_16;
	Cyclic#1.P2_Robot.KOM_OUT.Profinet_PLC_OUTPUTS[17] AT %QB."R2_IRB1200".Module002_Output_17;
	Cyclic#1.P2_Robot.KOM_OUT.Profinet_PLC_OUTPUTS[18] AT %QB."R2_IRB1200".Module002_Output_18;
	Cyclic#1.P2_Robot.KOM_OUT.Profinet_PLC_OUTPUTS[19] AT %QB."R2_IRB1200".Module002_Output_19;
	Cyclic#1.P2_Robot.KOM_OUT.Profinet_PLC_OUTPUTS[20] AT %QB."R2_IRB1200".Module002_Output_20;
	Cyclic#1.P2_Robot.KOM_OUT.Profinet_PLC_OUTPUTS[21] AT %QB."R2_IRB1200".Module002_Output_21;
	Cyclic#1.P2_Robot.KOM_OUT.Profinet_PLC_OUTPUTS[22] AT %QB."R2_IRB1200".Module002_Output_22;
	Cyclic#1.P2_Robot.KOM_OUT.Profinet_PLC_OUTPUTS[23] AT %QB."R2_IRB1200".Module002_Output_23;
	Cyclic#1.P2_Robot.KOM_OUT.Profinet_PLC_OUTPUTS[24] AT %QB."R2_IRB1200".Module002_Output_24;
	Cyclic#1.P2_Robot.KOM_OUT.Profinet_PLC_OUTPUTS[25] AT %QB."R2_IRB1200".Module002_Output_25;
	Cyclic#1.P2_Robot.KOM_OUT.Profinet_PLC_OUTPUTS[26] AT %QB."R2_IRB1200".Module002_Output_26;
	Cyclic#1.P2_Robot.KOM_OUT.Profinet_PLC_OUTPUTS[27] AT %QB."R2_IRB1200".Module002_Output_27;
	Cyclic#1.P2_Robot.KOM_OUT.Profinet_PLC_OUTPUTS[28] AT %QB."R2_IRB1200".Module002_Output_28;
	Cyclic#1.P2_Robot.KOM_OUT.Profinet_PLC_OUTPUTS[29] AT %QB."R2_IRB1200".Module002_Output_29;
	Cyclic#1.P2_Robot.KOM_OUT.Profinet_PLC_OUTPUTS[30] AT %QB."R2_IRB1200".Module002_Output_30;
	Cyclic#1.P2_Robot.KOM_OUT.Profinet_PLC_OUTPUTS[31] AT %QB."R2_IRB1200".Module002_Output_31;
	Cyclic#1.P2_Robot.KOM_OUT.Profinet_PLC_OUTPUTS[32] AT %QB."R2_IRB1200".Module002_Output_32;
	Cyclic#1.P2_Robot.KOM_OUT.Profinet_PLC_OUTPUTS[33] AT %QB."R2_IRB1200".Module002_Output_33;
	Cyclic#1.P2_Robot.KOM_OUT.Profinet_PLC_OUTPUTS[34] AT %QB."R2_IRB1200".Module002_Output_34;
	Cyclic#1.P2_Robot.KOM_OUT.Profinet_PLC_OUTPUTS[35] AT %QB."R2_IRB1200".Module002_Output_35;
	Cyclic#1.P2_Robot.KOM_OUT.Profinet_PLC_OUTPUTS[36] AT %QB."R2_IRB1200".Module002_Output_36;
	Cyclic#1.P2_Robot.KOM_OUT.Profinet_PLC_OUTPUTS[37] AT %QB."R2_IRB1200".Module002_Output_37;
	Cyclic#1.P2_Robot.KOM_OUT.Profinet_PLC_OUTPUTS[38] AT %QB."R2_IRB1200".Module002_Output_38;
	Cyclic#1.P2_Robot.KOM_OUT.Profinet_PLC_OUTPUTS[39] AT %QB."R2_IRB1200".Module002_Output_39;
	Cyclic#1.P2_Robot.KOM_OUT.Profinet_PLC_OUTPUTS[40] AT %QB."R2_IRB1200".Module002_Output_40;
	Cyclic#1.P2_Robot.KOM_OUT.Profinet_PLC_OUTPUTS[41] AT %QB."R2_IRB1200".Module002_Output_41;
	Cyclic#1.P2_Robot.KOM_OUT.Profinet_PLC_OUTPUTS[42] AT %QB."R2_IRB1200".Module002_Output_42;
	Cyclic#1.P2_Robot.KOM_OUT.Profinet_PLC_OUTPUTS[43] AT %QB."R2_IRB1200".Module002_Output_43;
	Cyclic#1.P2_Robot.KOM_OUT.Profinet_PLC_OUTPUTS[44] AT %QB."R2_IRB1200".Module002_Output_44;
	Cyclic#1.P2_Robot.KOM_OUT.Profinet_PLC_OUTPUTS[45] AT %QB."R2_IRB1200".Module002_Output_45;
	Cyclic#1.P2_Robot.KOM_OUT.Profinet_PLC_OUTPUTS[46] AT %QB."R2_IRB1200".Module002_Output_46;
	Cyclic#1.P2_Robot.KOM_OUT.Profinet_PLC_OUTPUTS[47] AT %QB."R2_IRB1200".Module002_Output_47;
	Cyclic#1.P2_Robot.KOM_OUT.Profinet_PLC_OUTPUTS[48] AT %QB."R2_IRB1200".Module002_Output_48;
	Cyclic#1.P2_Robot.KOM_OUT.Profinet_PLC_OUTPUTS[49] AT %QB."R2_IRB1200".Module002_Output_49;
	Cyclic#1.P2_Robot.KOM_OUT.Profinet_PLC_OUTPUTS[50] AT %QB."R2_IRB1200".Module002_Output_50;
	Cyclic#1.P2_Robot.KOM_OUT.Profinet_PLC_OUTPUTS[51] AT %QB."R2_IRB1200".Module002_Output_51;
	Cyclic#1.P2_Robot.KOM_OUT.Profinet_PLC_OUTPUTS[52] AT %QB."R2_IRB1200".Module002_Output_52;
	Cyclic#1.P2_Robot.KOM_OUT.Profinet_PLC_OUTPUTS[53] AT %QB."R2_IRB1200".Module002_Output_53;
	Cyclic#1.P2_Robot.KOM_OUT.Profinet_PLC_OUTPUTS[54] AT %QB."R2_IRB1200".Module002_Output_54;
	Cyclic#1.P2_Robot.KOM_OUT.Profinet_PLC_OUTPUTS[55] AT %QB."R2_IRB1200".Module002_Output_55;
	Cyclic#1.P2_Robot.KOM_OUT.Profinet_PLC_OUTPUTS[56] AT %QB."R2_IRB1200".Module002_Output_56;
	Cyclic#1.P2_Robot.KOM_OUT.Profinet_PLC_OUTPUTS[57] AT %QB."R2_IRB1200".Module002_Output_57;
	Cyclic#1.P2_Robot.KOM_OUT.Profinet_PLC_OUTPUTS[58] AT %QB."R2_IRB1200".Module002_Output_58;
	Cyclic#1.P2_Robot.KOM_OUT.Profinet_PLC_OUTPUTS[59] AT %QB."R2_IRB1200".Module002_Output_59;
	Cyclic#1.P2_Robot.KOM_OUT.Profinet_PLC_OUTPUTS[60] AT %QB."R2_IRB1200".Module002_Output_60;
	Cyclic#1.P2_Robot.KOM_OUT.Profinet_PLC_OUTPUTS[61] AT %QB."R2_IRB1200".Module002_Output_61;
	Cyclic#1.P2_Robot.KOM_OUT.Profinet_PLC_OUTPUTS[62] AT %QB."R2_IRB1200".Module002_Output_62;
	Cyclic#1.P2_Robot.KOM_OUT.Profinet_PLC_OUTPUTS[63] AT %QB."R2_IRB1200".Module002_Output_63;
	Cyclic#1.P1_Robot.PAR.Modul_IOLink_Inputs AT %IB."DS1_1".InputData01_1;
	Cyclic#1.P1_Vytah.PAR.Banner_IOLinkInputs AT %IO."DS1_1".InputData02;
	Cyclic#1.P1_Vytah.PAR.Banner_IOLinkOutputs AT %QO."DS1_1".OutputData02;
	Cyclic#1.P1_Vytah.PAR.SnimacPaletky_IOLinkInputs AT %IO."DS1_1".InputData03;
	Cyclic#1.P1_StoperSrobovania.PAR.SnimacPaletky_IOLinkInputs AT %IO."DS1_1".InputData04;
	Cyclic#1.P1_Pracovisko.IN.PrivodVzduchu_SnimacTlaku_S18 AT %IX."DI1.3_8DI".DigitalInput06;
	Cyclic#1.P1_Vytah.IN.VystupDopravnikaVytahu_OS12 AT %IX."DI1.3_8DI".DigitalInput03;
	Cyclic#1.P1_Vytah.IN.ZdvihVytahu_LimSnimacNEG_IS60 AT %IX."DI1.3_8DI".DigitalInput04;
	Cyclic#1.P1_Vytah.IN.ZdvihVytahu_LimSnimacPOS_IS61 AT %IX."DI1.3_8DI".DigitalInput05;
	Cyclic#1.P1_Srobovanie.IN.SkrutkM5_SnimacVakua_S28 AT %IX."DI1.4_8DI".DigitalInput08;
	Cyclic#1.P1_Vytah.OUT.Dopravnik_NAVAZANIE_M25 AT %QX."AB1.8_16xDO".DigitalOutput10;
	Cyclic#1.P1_Vytah.OUT.Dopravnik_VYVAZANIE_M25 AT %QX."AB1.8_16xDO".DigitalOutput15;
	Cyclic#1.P2_Dopravniky.OUT.HornyDoprav_ChodVPRED_M7 AT %QX."AB2.9_16xDO".DigitalOutput12;
	Cyclic#1.P2_Dopravniky.OUT.SpodnyDoprav_ChodVPRED_M8 AT %QX."AB2.9_16xDO".DigitalOutput13;
	Cyclic#1.P2_Robot.OUT.OdvzdusnenieVyvodov_YV70 AT %QX."AB2.9_16xDO".DigitalOutput16;
	Cyclic#1.P1_Srobovanie.PAR.K30_AtlasCopcoInputs[0] AT %ID."RJ5_P1_Srobovacka_K30".Module001_Input_00;
	Cyclic#1.P1_Srobovanie.PAR.K30_AllasCopcoOutputs[0] AT %QD."RJ5_P1_Srobovacka_K30".Module002_Output_00;
	Cyclic#1.P1_Srobovanie.PAR.K30_AtlasCopcoInputs[1] AT %ID."RJ5_P1_Srobovacka_K30".Module001_Input_01;
	Cyclic#1.P1_Srobovanie.PAR.K30_AllasCopcoOutputs[1] AT %QD."RJ5_P1_Srobovacka_K30".Module002_Output_01;
	Cyclic#1.P1_Srobovanie.PAR.M5_AtlasCopcoInputs[0] AT %ID."RJ6_P1_Srobovacka_M5".Module001_Input_00;
	Cyclic#1.P1_Srobovanie.PAR.M5_AllasCopcoOutputs[0] AT %QD."RJ6_P1_Srobovacka_M5".Module002_Output_00;
	Cyclic#1.P1_Srobovanie.PAR.M5_AtlasCopcoInputs[1] AT %ID."RJ6_P1_Srobovacka_M5".Module001_Input_01;
	Cyclic#1.P1_Srobovanie.PAR.M5_AllasCopcoOutputs[1] AT %QD."RJ6_P1_Srobovacka_M5".Module002_Output_01;
	Cyclic#1.P1_Srobovanie.PAR.M4_AtlasCopcoInputs[0] AT %ID."RJ7_P1_Srobovacka_M4".Module001_Input_00;
	Cyclic#1.P1_Srobovanie.PAR.M4_AllasCopcoOutputs[0] AT %QD."RJ7_P1_Srobovacka_M4".Module002_Output_00;
	Cyclic#1.P1_Srobovanie.PAR.M4_AtlasCopcoInputs[1] AT %ID."RJ7_P1_Srobovacka_M4".Module001_Input_01;
	Cyclic#1.P1_Srobovanie.PAR.M4_AllasCopcoOutputs[1] AT %QD."RJ7_P1_Srobovacka_M4".Module002_Output_01;
	Cyclic#1.P3_Pracovisko.STAV.KartaAB35_OK AT %IX."AB3.5_20xSI".ModuleOk;
	Cyclic#1.Safety.IN.P3_VyblokovanieSafety_CH1_SA1 AT %IX."AB3.5_20xSI".SafeDigitalInput01;
	Cyclic#1.Safety.IN.P3_VyblokovanieSafety_CH2_SA1 AT %IX."AB3.5_20xSI".SafeDigitalInput02;
	Cyclic#1.Safety.IN.P3_Skrina_TlacitkoCS_CH1_CS9 AT %IX."AB3.5_20xSI".SafeDigitalInput03;
	Cyclic#1.Safety.IN.P3_Skrina_TlacitkoCS_CH2_CS9 AT %IX."AB3.5_20xSI".SafeDigitalInput04;
	Cyclic#1.P3_Dopravniky.IN.HornyDoprav_TeplotaMotora_OK AT %IX."AB3.5_20xSI".SafeDigitalInput05;
	Cyclic#1.P3_Dopravniky.IN.SpodnyDoprav_TeplotaMotora_OK AT %IX."AB3.5_20xSI".SafeDigitalInput06;
	Cyclic#1.Safety.IN.P3_ZamkyBunky_CH1 AT %IX."AB3.5_20xSI".SafeDigitalInput07;
	Cyclic#1.Safety.IN.P3_ZamkyBunky_CH2 AT %IX."AB3.5_20xSI".SafeDigitalInput08;
	Cyclic#1.P3_Pracovisko.STAV.KartaAB36_OK AT %IX."AB3.6_4xSO".ModuleOk;
	Cyclic#1.P3_Pracovisko.STAV.KartaAB37_OK AT %IX."AB3.7_16xDI".ModuleOk;
	Cyclic#1.P3_Pracovisko.IN.PrepatovaOchrana_OK AT %IX."AB3.7_16xDI".DigitalInput01;
	Cyclic#1.P3_Dopravniky.IN.HornyDoprav_READY AT %IX."AB3.7_16xDI".DigitalInput07;
	Cyclic#1.P3_Dopravniky.IN.SpodnyDoprav_READY AT %IX."AB3.7_16xDI".DigitalInput08;
	Cyclic#1.P3_Srobovanie.IN.NapajanieSkrutkovackyK40_OK AT %IX."AB3.7_16xDI".DigitalInput02;
	Cyclic#1.P3_Srobovanie.IN.NapajanieSkrutkovackyM5_OK AT %IX."AB3.7_16xDI".DigitalInput03;
	Cyclic#1.P3_Srobovanie.IN.NapajanieVibroZasobnikaK40_OK AT %IX."AB3.7_16xDI".DigitalInput04;
	Cyclic#1.P3_Srobovanie.IN.NapajanieVibroZasobnikaM5_OK AT %IX."AB3.7_16xDI".DigitalInput05;
	Cyclic#1.P3_Srobovanie.IN.NapajanieVibroListyM5_OK AT %IX."AB3.7_16xDI".DigitalInput06;
	Cyclic#1.P3_LeakageTestA.IN.NapajanieTestera_OK_ATEQ1 AT %IX."AB3.7_16xDI".DigitalInput09;
	Cyclic#1.P3_LeakageTestB.IN.NapajanieTestera_OK_ATEQ2 AT %IX."AB3.7_16xDI".DigitalInput10;
	Cyclic#1.Safety.IN.P3_SV_Ventil1_ZonaBunka_B11 AT %IX."AB3.7_16xDI".DigitalInput11;
	Cyclic#1.Safety.IN.P3_SV_Ventil2_ZonaBunka_B12 AT %IX."AB3.7_16xDI".DigitalInput12;
	Cyclic#1.Safety.IN.P3_SV_ZonaCS AT %IX."AB3.7_16xDI".DigitalInput13;
	Cyclic#1.Safety.IN.P3_SV_ZonaBunka AT %IX."AB3.7_16xDI".DigitalInput14;
	Cyclic#1.P3_Pracovisko.STAV.KartaAB38_OK AT %IX."AB3.8_16xDO".ModuleOk;
	Cyclic#1.P3_Pracovisko.OUT.Majak_ZeleneSvetlo AT %QX."AB3.8_16xDO".DigitalOutput01;
	Cyclic#1.P3_Pracovisko.OUT.Majak_ZlteSvetlo AT %QX."AB3.8_16xDO".DigitalOutput02;
	Cyclic#1.P3_Pracovisko.OUT.Majak_CerveneSvetlo AT %QX."AB3.8_16xDO".DigitalOutput03;
	Cyclic#1.P3_Pracovisko.OUT.Majak_Hukacka AT %QX."AB3.8_16xDO".DigitalOutput04;
	Cyclic#1.P3_Srobovanie.OUT.ZasobSrobK40_Vibrovanie_RUN_FM15 AT %QX."AB3.8_16xDO".DigitalOutput05;
	Cyclic#1.P3_Srobovanie.OUT.ZasobSrobM5_Vibrovanie_RUN_FM16 AT %QX."AB3.8_16xDO".DigitalOutput06;
	Cyclic#1.P3_Srobovanie.OUT.VibrolistaSrobM5_Vibrov_RUN_FM17 AT %QX."AB3.8_16xDO".DigitalOutput07;
	Cyclic#1.P3_Pracovisko.OUT.OsvetlenieBunky AT %QX."AB3.8_16xDO".DigitalOutput08;
	Cyclic#1.P3_Dopravniky.OUT.HornyDoprav_ChodVPRED_M33 AT %QX."AB3.8_16xDO".DigitalOutput09;
	Cyclic#1.P3_Dopravniky.OUT.SpodnyDoprav_ChodVPRED_M34 AT %QX."AB3.8_16xDO".DigitalOutput10;
	Cyclic#1.P3_Pracovisko.OUT.Osvetlenie_CAM13 AT %QX."AB3.8_16xDO".DigitalOutput11;
	Cyclic#1.P3_Pracovisko.STAV.KartaAB39_OK AT %IX."AB3.9_X2X".ModuleOk;
	Cyclic#1.P3_Pracovisko.STAV.ModulDI31_OK AT %IX."DI3.1_16DI".ModuleOk;
	Cyclic#1.P3_StoperSrobovania.IN.Centrovanie_ZASUNUTE_MS42 AT %IX."DI3.1_16DI".DigitalInput03;
	Cyclic#1.P3_StoperSrobovania.IN.Centrovanie_VYSUNUTE_MS43 AT %IX."DI3.1_16DI".DigitalInput04;
	Cyclic#1.P3_Srobovanie.IN.HVTest_Kontakty_ZASUNUTE_MS44 AT %IX."DI3.1_16DI".DigitalInput05;
	Cyclic#1.P3_Srobovanie.IN.HVTest_Kontakty_VYSUNUTE_MS45 AT %IX."DI3.1_16DI".DigitalInput06;
	Cyclic#1.P3_AkumulacnyStoper.IN.PritomnPaletky_IS65 AT %IX."DI3.1_16DI".DigitalInput09;
	Cyclic#1.P3_SpodnyStoper.IN.PritomnPaletky_IS66 AT %IX."DI3.1_16DI".DigitalInput10;
	Cyclic#1.P3_Pracovisko.IN.PrivodVzduchu_SnimacTlaku_S25 AT %IX."DI3.1_16DI".DigitalInput11;
	Cyclic#1.P3_Pracovisko.STAV.ModulDI32_OK AT %IX."DI3.2_16DI".ModuleOk;
	Cyclic#1.P3_LeakageTestA.IN.Pritlak_ZASUNUTY_MS46 AT %IX."DI3.2_16DI".DigitalInput01;
	Cyclic#1.P3_LeakageTestA.IN.Pritlak_VYSUNUTY_MS47 AT %IX."DI3.2_16DI".DigitalInput02;
	Cyclic#1.P3_LeakageTestB.IN.Pritlak_ZASUNUTY_MS48 AT %IX."DI3.2_16DI".DigitalInput03;
	Cyclic#1.P3_LeakageTestB.IN.Pritlak_VYSUNUTY_MS49 AT %IX."DI3.2_16DI".DigitalInput04;
	Cyclic#1.P3_LeakageTestA.IN.PritomnostKopita_IS67 AT %IX."DI3.2_16DI".DigitalInput05;
	Cyclic#1.P3_LeakageTestA.IN.Kopito_ZASUNUTE_IS68 AT %IX."DI3.2_16DI".DigitalInput06;
	Cyclic#1.P3_LeakageTestB.IN.PritomnostKopita_IS69 AT %IX."DI3.2_16DI".DigitalInput07;
	Cyclic#1.P3_LeakageTestB.IN.Kopito_ZASUNUTE_IS70 AT %IX."DI3.2_16DI".DigitalInput08;
	Cyclic#1.P3_LeakageTestA.IN.Centrovanie_VYSUNUTE_IS71 AT %IX."DI3.2_16DI".DigitalInput09;
	Cyclic#1.P3_LeakageTestA.IN.Centrovanie_ZASUNUTE_IS72 AT %IX."DI3.2_16DI".DigitalInput10;
	Cyclic#1.P3_LeakageTestB.IN.Centrovanie_VYSUNUTE_IS73 AT %IX."DI3.2_16DI".DigitalInput11;
	Cyclic#1.P3_LeakageTestB.IN.Centrovanie_ZASUNUTE_IS74 AT %IX."DI3.2_16DI".DigitalInput12;
	Cyclic#1.P3_Pracovisko.STAV.ModulDI33_OK AT %IX."DI3.3_16DI".ModuleOk;
	Cyclic#1.P3_Srobovanie.IN.ZasobSrobK40_PRAZDNY_IS79 AT %IX."DI3.3_16DI".DigitalInput01;
	Cyclic#1.P3_Srobovanie.IN.ZasobSrobK40_ListaPLNA_OS15 AT %IX."DI3.3_16DI".DigitalInput02;
	Cyclic#1.P3_Srobovanie.IN.NastrelSrobK40_SrobaPresla_IS80 AT %IX."DI3.3_16DI".DigitalInput03;
	Cyclic#1.P3_Srobovanie.IN.SkrutkK40_Cist_SrobaPresla_IS82 AT %IX."DI3.3_16DI".DigitalInput04;
	Cyclic#1.P3_Srobovanie.IN.ZasobSrobM5_PRAZDNY_IS83 AT %IX."DI3.3_16DI".DigitalInput09;
	Cyclic#1.P3_Srobovanie.IN.ZasobSrobM5_ListaPLNA_OS16 AT %IX."DI3.3_16DI".DigitalInput10;
	Cyclic#1.P3_Srobovanie.IN.VibrolistaSrobM5_KONIEC_OS17 AT %IX."DI3.3_16DI".DigitalInput11;
	Cyclic#1.P3_Srobovanie.IN.VibrolistaSrobM5_ZACIATOK_OS18 AT %IX."DI3.3_16DI".DigitalInput12;
	Cyclic#1.P3_Srobovanie.IN.OddelSrobM5_SrobaNaVstupe_OS19 AT %IX."DI3.3_16DI".DigitalInput13;
	Cyclic#1.P3_Srobovanie.IN.OddelSrobM5_SrobaNaVystupe_OS20 AT %IX."DI3.3_16DI".DigitalInput14;
	Cyclic#1.P3_Pracovisko.STAV.ModulDI34_OK AT %IX."DI3.4_8DI".ModuleOk;
	Cyclic#1.P3_Srobovanie.IN.ManipulOsY_LimSnimacPOS_IS75 AT %IX."DI3.4_8DI".DigitalInput01;
	Cyclic#1.P3_Srobovanie.IN.ManipulOsY_LimSnimacNEG_IS76 AT %IX."DI3.4_8DI".DigitalInput02;
	Cyclic#1.P3_Srobovanie.IN.SkrutkM5_ZASUNUTY_MS57 AT %IX."DI3.4_8DI".DigitalInput03;
	Cyclic#1.P3_Pracovisko.STAV.ModulSI31_OK AT %IX."SI3.1".ModuleOk;
	Cyclic#1.Safety.IN.P3_VstupBunky_Bariera_CH1_BC9 AT %IX."SI3.1".SafeDigitalInput01;
	Cyclic#1.Safety.IN.P3_VstupBunky_Bariera_CH2_BC9 AT %IX."SI3.1".SafeDigitalInput02;
	Cyclic#1.Safety.IN.P3_VystupBunky_Bariera_CH1_BC10 AT %IX."SI3.1".SafeDigitalInput03;
	Cyclic#1.Safety.IN.P3_VystupBunky_Bariera_CH2_BC10 AT %IX."SI3.1".SafeDigitalInput04;
	Cyclic#1.P3_Pracovisko.STAV.ModulDM31_OK AT %IX."DM3.1".ModuleOk;
	Cyclic#1.P3_Srobovanie.IN.ZasobSrobM5_Banner_SB12 AT %IX."DM3.1".DigitalInput07;
	Cyclic#1.P3_Srobovanie.OUT.ZasobSrobM5_Banner_CervenaLED AT %QX."DM3.1".DigitalOutput08;
	Cyclic#1.P3_Srobovanie.IN.ZasobSrobK40_Banner_SB13 AT %IX."DM3.1".DigitalInput09;
	Cyclic#1.P3_Srobovanie.OUT.ZasobSrobK40_Banner_CervenaLED AT %QX."DM3.1".DigitalOutput10;
	Cyclic#1.P3_Pracovisko.STAV.ModulDS32_OK AT %IX."DS3_2".ModuleOk;
	Cyclic#1.P3_Pracovisko.STAV.ModulDS31_OK AT %IX."DS3_1".ModuleOk;
	Cyclic#1.P3_Pracovisko.STAV.ModulDS33_OK AT %IX."DS3_3".ModuleOk;
	Cyclic#1.Safety.IN.P3_SV_Ventil1_ZonaBunka_B11 AT %QX."SL1_SafetyMaster".BOOL131;
	Cyclic#1.Safety.IN.P3_SV_Ventil2_ZonaBunka_B12 AT %QX."SL1_SafetyMaster".BOOL132;
	Cyclic#1.Safety.IN.P3_SV_ZonaBunka AT %QX."SL1_SafetyMaster".BOOL133;
	Cyclic#1.Safety.IN.P3_SV_ZonaCS AT %QX."SL1_SafetyMaster".BOOL134;
	Cyclic#1.Safety.IN.P3_ReleaseKartySO_AB36 AT %QX."SL1_SafetyMaster".BOOL135;
	Cyclic#1.Safety.IN.P3_ZonaBunky_RESET AT %QX."SL1_SafetyMaster".BOOL130;
	Cyclic#1.P3_Pracovisko.IN.PrivodVzduchu_SnimacTlaku_S25 AT %QX."SL1_SafetyMaster".BOOL129;
	Cyclic#1.Safety.STAV.P3_Skrina_TlacitkoCS_AKTIVNE AT %IX."SL1_SafetyMaster".BOOL029;
	Cyclic#1.Safety.STAV.P3_VstupBunky_Bariera_AKTIVNA AT %IX."SL1_SafetyMaster".BOOL030;
	Cyclic#1.Safety.STAV.P3_VyblokovanieSafety_AKTIVNE AT %IX."SL1_SafetyMaster".BOOL031;
	Cyclic#1.Safety.STAV.P3_VystupBunky_Bariera_AKTIVNA AT %IX."SL1_SafetyMaster".BOOL032;
	Cyclic#1.Safety.STAV.P3_ZamkyBunky_AKTIVNE AT %IX."SL1_SafetyMaster".BOOL033;
	Cyclic#1.Safety.STAV.P3_ZonaBunky_AKTIVNA AT %IX."SL1_SafetyMaster".BOOL034;
	Cyclic#1.P2_Srobovanie.PAR.M6_AtlasCopcoInputs[0] AT %ID."RJ2_P2_Srobovacka_M6".Module001_Input_00;
	Cyclic#1.P2_Srobovanie.PAR.M6_AtlasCopcoInputs[1] AT %ID."RJ2_P2_Srobovacka_M6".Module001_Input_01;
	Cyclic#1.P2_Srobovanie.PAR.M6_AllasCopcoOutputs[0] AT %QD."RJ2_P2_Srobovacka_M6".Module002_Output_00;
	Cyclic#1.P2_Srobovanie.PAR.M6_AllasCopcoOutputs[1] AT %QD."RJ2_P2_Srobovacka_M6".Module002_Output_01;
	Cyclic#1.P2_Srobovanie.PAR.M5_AtlasCopcoInputs[0] AT %ID."RJ4_P2_Srobovacka_M5".Module001_Input_00;
	Cyclic#1.P2_Srobovanie.PAR.M5_AtlasCopcoInputs[1] AT %ID."RJ4_P2_Srobovacka_M5".Module001_Input_01;
	Cyclic#1.P2_Srobovanie.PAR.M5_AllasCopcoOutputs[0] AT %QD."RJ4_P2_Srobovacka_M5".Module002_Output_00;
	Cyclic#1.P2_Srobovanie.PAR.M5_AllasCopcoOutputs[1] AT %QD."RJ4_P2_Srobovacka_M5".Module002_Output_01;
	Cyclic#1.P2_Srobovanie.PAR.M4_AtlasCopcoInputs[0] AT %ID."RJ3_P2_Srobovacka_M4".Module001_Input_00;
	Cyclic#1.P2_Srobovanie.PAR.M4_AtlasCopcoInputs[1] AT %ID."RJ3_P2_Srobovacka_M4".Module001_Input_01;
	Cyclic#1.P2_Srobovanie.PAR.M4_AllasCopcoOutputs[0] AT %QD."RJ3_P2_Srobovacka_M4".Module002_Output_00;
	Cyclic#1.P2_Srobovanie.PAR.M4_AllasCopcoOutputs[1] AT %QD."RJ3_P2_Srobovacka_M4".Module002_Output_01;
	Cyclic#1.P3_Pracovisko.OUT.VT6_OUT1 AT %QB."VentilovyTerminal_VT6".OUT1_I2200_S01Out;
	Cyclic#1.P3_Pracovisko.OUT.VT6_OUT2 AT %QB."VentilovyTerminal_VT6".OUT2_I2200_S02Out;
	Cyclic#1.P3_Pracovisko.OUT.VT6_OUT3 AT %QB."VentilovyTerminal_VT6".OUT3_I2200_S03Out;
	Cyclic#1.P3_Pracovisko.OUT.VT6_OUT4 AT %QB."VentilovyTerminal_VT6".OUT4_I2200_S04Out;
	Cyclic#1.P3_Pracovisko.OUT.VT7_OUT1 AT %QB."VentilovyTerminal_VT7".OUT1_I2200_S01Out;
	Cyclic#1.P3_Pracovisko.OUT.VT7_OUT2 AT %QB."VentilovyTerminal_VT7".OUT2_I2200_S02Out;
	Cyclic#1.P3_Pracovisko.OUT.VT7_OUT3 AT %QB."VentilovyTerminal_VT7".OUT3_I2200_S03Out;
	Cyclic#1.P3_Pracovisko.OUT.VT7_OUT4 AT %QB."VentilovyTerminal_VT7".OUT4_I2200_S04Out;
	Cyclic#1.P3_Srobovanie.PAR.K40_AtlasCopcoInputs[0] AT %ID."P3_Srobovacka_K40".Module001_Input_00;
	Cyclic#1.P3_Srobovanie.PAR.K40_AtlasCopcoInputs[1] AT %ID."P3_Srobovacka_K40".Module001_Input_01;
	Cyclic#1.P3_Srobovanie.PAR.K40_AllasCopcoOutputs[0] AT %QD."P3_Srobovacka_K40".Module002_Output_00;
	Cyclic#1.P3_Srobovanie.PAR.K40_AllasCopcoOutputs[1] AT %QD."P3_Srobovacka_K40".Module002_Output_01;
	Cyclic#1.P3_Srobovanie.PAR.M5_AtlasCopcoInputs[0] AT %ID."P3_Srobovacka_M5".Module001_Input_00;
	Cyclic#1.P3_Srobovanie.PAR.M5_AtlasCopcoInputs[1] AT %ID."P3_Srobovacka_M5".Module001_Input_01;
	Cyclic#1.P3_Srobovanie.PAR.M5_AllasCopcoOutputs[0] AT %QD."P3_Srobovacka_M5".Module002_Output_00;
	Cyclic#1.P3_Srobovanie.PAR.M5_AllasCopcoOutputs[1] AT %QD."P3_Srobovacka_M5".Module002_Output_01;
	Cyclic#1.P2_SkrutkovacMatic.PAR.MaticeM4_AtlasCopcoInputs[0] AT %ID."RJ1_P2_SrobovackaMatic_M4".Module001_Input_00;
	Cyclic#1.P2_SkrutkovacMatic.PAR.MaticeM4_AtlasCopcoInputs[1] AT %ID."RJ1_P2_SrobovackaMatic_M4".Module001_Input_01;
	Cyclic#1.P2_SkrutkovacMatic.PAR.MaticeM4_AtlasCopcoOutputs[0] AT %QD."RJ1_P2_SrobovackaMatic_M4".Module002_Output_00;
	Cyclic#1.P2_SkrutkovacMatic.PAR.MaticeM4_AtlasCopcoOutputs[1] AT %QD."RJ1_P2_SrobovackaMatic_M4".Module002_Output_01;
	Cyclic#1.P3_StoperSrobovania.PAR.SnimacPaletky_IOLinkInputs AT %IO."DS3_1".InputData01;
	Cyclic#1.P3_LeakageTestA.PAR.SnimacPaletky_IOLinkInputs AT %IO."DS3_1".InputData02;
	Cyclic#1.P3_LeakageTestB.PAR.SnimacPaletky_IOLinkInputs AT %IO."DS3_1".InputData03;
	Cyclic#1.P4_Pracovisko.IN.PrivodVzduchu_SnimacTlaku_S15 AT %QX."SL1_SafetyMaster".BOOL136;
	Cyclic#1.Safety.IN.P4_ZonaBunky_RESET AT %QX."SL1_SafetyMaster".BOOL137;
	Cyclic#1.Safety.IN.P4_ZonaVytahu_RESET AT %QX."SL1_SafetyMaster".BOOL138;
	Cyclic#1.Safety.IN.P4_SV_Ventil1_ZonaBunka_B13 AT %QX."SL1_SafetyMaster".BOOL139;
	Cyclic#1.Safety.IN.P4_SV_Ventil2_ZonaBunka_B14 AT %QX."SL1_SafetyMaster".BOOL140;
	Cyclic#1.Safety.IN.P4_SV_ZonaBunka AT %QX."SL1_SafetyMaster".BOOL141;
	Cyclic#1.Safety.IN.P4_SV_ZonaCS AT %QX."SL1_SafetyMaster".BOOL142;
	Cyclic#1.Safety.IN.P4_SV_ZonaVytah AT %QX."SL1_SafetyMaster".BOOL143;
	Cyclic#1.Safety.IN.P4_ReleaseKartySO_AB45 AT %QX."SL1_SafetyMaster".BOOL144;
	Cyclic#1.Safety.IN.P4_Vytah_Zdvih_BUSY AT %QX."SL1_SafetyMaster".BOOL145;
	Cyclic#1.Safety.STAV.P4_Panel_TlacitkoCS_AKTIVNE AT %IX."SL1_SafetyMaster".BOOL035;
	Cyclic#1.Safety.STAV.P4_Skrina_TlacitkoCS_AKTIVNE AT %IX."SL1_SafetyMaster".BOOL036;
	Cyclic#1.Safety.STAV.P4_VstupBunky_Bariera_AKTIVNA AT %IX."SL1_SafetyMaster".BOOL037;
	Cyclic#1.Safety.STAV.P4_VystupBunky_Bariera_AKTIVNA AT %IX."SL1_SafetyMaster".BOOL038;
	Cyclic#1.Safety.STAV.P4_Vytah_Bariera_AKTIVNA AT %IX."SL1_SafetyMaster".BOOL039;
	Cyclic#1.Safety.STAV.P4_VyblokovanieSafety_AKTIVNE AT %IX."SL1_SafetyMaster".BOOL040;
	Cyclic#1.Safety.STAV.P4_ZamkyBunky_AKTIVNE AT %IX."SL1_SafetyMaster".BOOL041;
	Cyclic#1.Safety.STAV.P4_ZonaBunky_AKTIVNA AT %IX."SL1_SafetyMaster".BOOL042;
	Cyclic#1.Safety.STAV.P4_ZonaVytahu_AKTIVNA AT %IX."SL1_SafetyMaster".BOOL043;
	Cyclic#1.Safety.STAV.P4_SnimacVytahu_AKTIVNY AT %IX."SL1_SafetyMaster".BOOL044;
	Cyclic#1.P4_Pracovisko.OUT.VT8_OUT1 AT %QB."VentilovyTerminal_VT8".OUT1_I2200_S01Out;
	Cyclic#1.P4_Pracovisko.OUT.VT8_OUT2 AT %QB."VentilovyTerminal_VT8".OUT2_I2200_S02Out;
	Cyclic#1.P4_Pracovisko.OUT.VT8_OUT3 AT %QB."VentilovyTerminal_VT8".OUT3_I2200_S03Out;
	Cyclic#1.P4_Pracovisko.OUT.VT8_OUT4 AT %QB."VentilovyTerminal_VT8".OUT4_I2200_S04Out;
	Cyclic#1.P4_Pracovisko.STAV.KartaAB44_OK AT %IX."AB4.4_20xSI".ModuleOk;
	Cyclic#1.Safety.IN.P4_Skrina_TlacitkoCS_CH1_CS7 AT %IX."AB4.4_20xSI".SafeDigitalInput01;
	Cyclic#1.Safety.IN.P4_Skrina_TlacitkoCS_CH2_CS7 AT %IX."AB4.4_20xSI".SafeDigitalInput02;
	Cyclic#1.Safety.IN.P4_Panel_TlacitkoCS_CH1_CS6 AT %IX."AB4.4_20xSI".SafeDigitalInput03;
	Cyclic#1.Safety.IN.P4_Panel_TlacitkoCS_CH2_CS6 AT %IX."AB4.4_20xSI".SafeDigitalInput04;
	Cyclic#1.Safety.IN.P4_VyblokovanieSafety_CH1_SA1 AT %IX."AB4.4_20xSI".SafeDigitalInput05;
	Cyclic#1.Safety.IN.P4_VyblokovanieSafety_CH2_SA1 AT %IX."AB4.4_20xSI".SafeDigitalInput06;
	Cyclic#1.Safety.IN.P4_Vytah_SnimHornaPoz_CH1_B7 AT %IX."AB4.4_20xSI".SafeDigitalInput07;
	Cyclic#1.Safety.IN.P4_Vytah_SnimHornaPoz_CH2_B7 AT %IX."AB4.4_20xSI".SafeDigitalInput08;
	Cyclic#1.P4_Dopravniky.IN.HornyDoprav_TeplotaMotora_OK AT %IX."AB4.4_20xSI".SafeDigitalInput09;
	Cyclic#1.P4_Vytah.IN.Dopravnik_TeplotaMotora_OK AT %IX."AB4.4_20xSI".SafeDigitalInput10;
	Cyclic#1.P4_Dopravniky.IN.SpodnyDoprav_TeplotaMotora_OK AT %IX."AB4.4_20xSI".SafeDigitalInput11;
	Cyclic#1.P4_Pracovisko.STAV.ModulSI42_OK AT %IX."SI4.2".ModuleOk;
	Cyclic#1.Safety.IN.P4_VstupBunky_Bariera_CH1_BC4 AT %IX."SI4.2".SafeDigitalInput01;
	Cyclic#1.Safety.IN.P4_VstupBunky_Bariera_CH2_BC4 AT %IX."SI4.2".SafeDigitalInput02;
	Cyclic#1.Safety.IN.P4_VystupBunky_Bariera_CH1_BC5 AT %IX."SI4.2".SafeDigitalInput03;
	Cyclic#1.Safety.IN.P4_VystupBunky_Bariera_CH2_BC5 AT %IX."SI4.2".SafeDigitalInput04;
	Cyclic#1.P4_Pracovisko.STAV.ModulSI41_OK AT %IX."SI4.1".ModuleOk;
	Cyclic#1.Safety.IN.P4_ZamkyBunky_CH1 AT %IX."SI4.1".SafeDigitalInput01;
	Cyclic#1.Safety.IN.P4_ZamkyBunky_CH2 AT %IX."SI4.1".SafeDigitalInput02;
	Cyclic#1.Safety.IN.P4_Vytah_Bariera_CH1_BC3 AT %IX."SI4.1".SafeDigitalInput03;
	Cyclic#1.Safety.IN.P4_Vytah_Bariera_CH2_BC3 AT %IX."SI4.1".SafeDigitalInput04;
	Cyclic#1.P4_Pracovisko.STAV.KartaAB45_OK AT %IX."AB4.5_4xSO".ModuleOk;
	Cyclic#1.P4_Pracovisko.STAV.KartaAB48_OK AT %IX."AB4.8_X2X".ModuleOk;
	Cyclic#1.P4_Pracovisko.STAV.ModulDI42_OK AT %IX."DI4.2_16DI".ModuleOk;
	Cyclic#1.P4_Pracovisko.STAV.ModulDM41_OK AT %IX."DM4.1".ModuleOk;
	Cyclic#1.P4_Pracovisko.STAV.ModulDS41_OK AT %IX."DS4_1".ModuleOk;
	Cyclic#1.P4_Pracovisko.STAV.ModulDI41_OK AT %IX."DI4.1_8DI".ModuleOk;
	Cyclic#1.P4_Pracovisko.STAV.ModulDS42_OK AT %IX."DS4_2".ModuleOk;
	Cyclic#1.P4_Pracovisko.IN.PrepatovaOchrana_OK AT %IX."AB4.6_16xDI".DigitalInput01;
	Cyclic#1.P4_Etiketovacka.IN.NapajanieTlaciarne_OK AT %IX."AB4.6_16xDI".DigitalInput02;
	Cyclic#1.P4_Dopravniky.IN.HornyDoprav_READY AT %IX."AB4.6_16xDI".DigitalInput03;
	Cyclic#1.P4_Vytah.IN.Dopravnik_READY AT %IX."AB4.6_16xDI".DigitalInput04;
	Cyclic#1.P4_Dopravniky.IN.SpodnyDoprav_READY AT %IX."AB4.6_16xDI".DigitalInput05;
	Cyclic#1.Safety.IN.P4_SV_Ventil1_ZonaBunka_B13 AT %IX."AB4.6_16xDI".DigitalInput06;
	Cyclic#1.Safety.IN.P4_SV_Ventil2_ZonaBunka_B14 AT %IX."AB4.6_16xDI".DigitalInput07;
	Cyclic#1.Safety.IN.P4_SV_ZonaCS AT %IX."AB4.6_16xDI".DigitalInput08;
	Cyclic#1.Safety.IN.P4_SV_ZonaBunka AT %IX."AB4.6_16xDI".DigitalInput09;
	Cyclic#1.Safety.IN.P4_SV_ZonaVytah AT %IX."AB4.6_16xDI".DigitalInput10;
	Cyclic#1.P4_Pracovisko.OUT.Majak_ZeleneSvetlo AT %QX."AB4.7_16xDO".DigitalOutput01;
	Cyclic#1.P4_Pracovisko.OUT.Majak_ZlteSvetlo AT %QX."AB4.7_16xDO".DigitalOutput02;
	Cyclic#1.P4_Pracovisko.OUT.Majak_CerveneSvetlo AT %QX."AB4.7_16xDO".DigitalOutput03;
	Cyclic#1.P4_Pracovisko.OUT.Majak_Hukacka AT %QX."AB4.7_16xDO".DigitalOutput04;
	Cyclic#1.P4_Dopravniky.OUT.HornyDoprav_ChodVPRED_M24 AT %QX."AB4.7_16xDO".DigitalOutput05;
	Cyclic#1.P4_Dopravniky.OUT.SpodnyDoprav_ChodVPRED_M27 AT %QX."AB4.7_16xDO".DigitalOutput07;
	Cyclic#1.P4_Pracovisko.OUT.Osvetlenie_CAM16 AT %QX."AB4.7_16xDO".DigitalOutput08;
	Cyclic#1.P4_Pracovisko.OUT.OsvetlenieBunky AT %QX."AB4.7_16xDO".DigitalOutput11;
	Cyclic#1.P4_Pracovisko.OUT.Osvetlenie_CAM15 AT %QX."AB4.7_16xDO".DigitalOutput12;
	Cyclic#1.P4_Pracovisko.STAV.KartaAB47_OK AT %IX."AB4.7_16xDO".ModuleOk;
	Cyclic#1.P4_Pracovisko.STAV.KartaAB46_OK AT %IX."AB4.6_16xDI".ModuleOk;
	Cyclic#1.P4_FunkcnyTestB.IN.HorneKontakty_ZASUNUTE_MS24 AT %IX."DI4.2_16DI".DigitalInput09;
	Cyclic#1.P4_FunkcnyTestB.IN.HorneKontakty_VYSUNUTE_MS26 AT %IX."DI4.2_16DI".DigitalInput10;
	Cyclic#1.P4_FunkcnyTestB.IN.Centrovanie_ZASUNUTE_MS28 AT %IX."DI4.2_16DI".DigitalInput11;
	Cyclic#1.P4_FunkcnyTestB.IN.Centrovanie_VYSUNUTE_MS30 AT %IX."DI4.2_16DI".DigitalInput12;
	Cyclic#1.P4_FunkcnyTestB.IN.SpodneKontakty_ZASUNUTE_MS32 AT %IX."DI4.2_16DI".DigitalInput13;
	Cyclic#1.P4_FunkcnyTestB.IN.SpodneKontakty_VYSUNUTE_MS34 AT %IX."DI4.2_16DI".DigitalInput14;
	Cyclic#1.P4_Vytah.IN.VystupDopravnikaVytahu_OS11 AT %IX."DI4.2_16DI".DigitalInput15;
	Cyclic#1.P4_Pracovisko.IN.PrivodVzduchu_SnimacTlaku_S15 AT %IX."DI4.2_16DI".DigitalInput16;
	Cyclic#1.P4_Etiketovacka.IN.ZdvihEtiketovania_RefSnimac_IS59 AT %IX."DI4.1_8DI".DigitalInput01;
	Cyclic#1.P4_Etiketovacka.IN.Aplikator_ZASUNUTY_MS35 AT %IX."DI4.1_8DI".DigitalInput02;
	Cyclic#1.P4_Etiketovacka.IN.Aplikator_VYSUNUTY_MS36 AT %IX."DI4.1_8DI".DigitalInput03;
	Cyclic#1.P4_Etiketovacka.IN.Centrovanie_VYSUNUTE_IS54 AT %IX."DI4.1_8DI".DigitalInput04;
	Cyclic#1.P4_Etiketovacka.IN.Centrovanie_ZASUNUTE_IS55 AT %IX."DI4.1_8DI".DigitalInput05;
	Cyclic#1.P4_Dopravniky.IN.SnimacZaplneniaSpodnejTrate_IS58 AT %IX."DI4.1_8DI".DigitalInput06;
	Cyclic#1.P4_Etiketovacka.IN.SnimacVakuaPrisavaniaEtikety_S32 AT %IX."DI4.1_8DI".DigitalInput07;
	Cyclic#1.P4_FunkcnyTestA.IN.HorneKontakty_ZASUNUTE_MS23 AT %IX."DI4.2_16DI".DigitalInput01;
	Cyclic#1.P4_FunkcnyTestA.IN.HorneKontakty_VYSUNUTE_MS25 AT %IX."DI4.2_16DI".DigitalInput02;
	Cyclic#1.P4_FunkcnyTestA.IN.Centrovanie_ZASUNUTE_MS27 AT %IX."DI4.2_16DI".DigitalInput03;
	Cyclic#1.P4_FunkcnyTestA.IN.Centrovanie_VYSUNUTE_MS29 AT %IX."DI4.2_16DI".DigitalInput04;
	Cyclic#1.P4_FunkcnyTestA.IN.SpodneKontakty_ZASUNUTE_MS31 AT %IX."DI4.2_16DI".DigitalInput05;
	Cyclic#1.P4_FunkcnyTestA.IN.SpodneKontakty_VYSUNUTE_MS33 AT %IX."DI4.2_16DI".DigitalInput06;
	Cyclic#1.P4_Vytah.IN.ZdvihVytahu_LimSnimacNEG_IS56 AT %IX."DI4.2_16DI".DigitalInput07;
	Cyclic#1.P4_Vytah.IN.ZdvihVytahu_LimSnimacPOS_IS57 AT %IX."DI4.2_16DI".DigitalInput08;
	Cyclic#1.P4_FunkcnyTestA.PAR.SnimacPaletky_IOLinkInputs AT %IO."DS4_1".InputData01;
	Cyclic#1.P4_FunkcnyTestB.PAR.SnimacPaletky_IOLinkInputs AT %IO."DS4_1".InputData02;
	Cyclic#1.P4_Etiketovacka.PAR.SnimacPaletky_IOLinkInputs AT %IO."DS4_1".InputData03;
	Cyclic#1.P4_Vytah.OUT.Dopravnik_NAVAZANIE_M5 AT %QX."AB4.7_16xDO".DigitalOutput06;
	Cyclic#1.P4_Vytah.OUT.Dopravnik_VYVAZANIE_M5 AT %QX."AB4.7_16xDO".DigitalOutput13;
	Cyclic#1.P4_Vytah.PAR.SnimacPaletky_IOLinkInputs AT %IO."DS4_2".InputData02;
	Cyclic#1.P4_Vytah.PAR.Banner_IOLinkInputs AT %IO."DS4_2".InputData01;
	Cyclic#1.P4_Vytah.PAR.Banner_IOLinkOutputs AT %QO."DS4_2".OutputData01;
	Cyclic#1.P3_Srobovanie.IN.HVTest_ZASUNUTY_MS51 AT %IX."DI3.4_8DI".DigitalInput07;
	Cyclic#1.P3_Srobovanie.IN.HVTest_VYSUNUTY_MS50 AT %IX."DI3.4_8DI".DigitalInput06;
	Cyclic#1.P3_Srobovanie.IN.SkrutkK40_Cist_BrzdaOtvor_MS53 AT %IX."DI3.3_16DI".DigitalInput05;
	Cyclic#1.P3_Srobovanie.IN.SkrutkK40_Cist_BrzdaZatvor_MS54 AT %IX."DI3.3_16DI".DigitalInput06;
	Cyclic#1.P3_Srobovanie.IN.OddelSrobM5_OtocenyVZAD_MS55 AT %IX."DI3.3_16DI".DigitalInput15;
	Cyclic#1.P3_Srobovanie.IN.OddelSrobM5_OtocenyVPRED_MS56 AT %IX."DI3.3_16DI".DigitalInput16;
	Cyclic#1.P3_Srobovanie.IN.SkrutkK40_ZASUNUTY_MS52 AT %IX."DI3.4_8DI".DigitalInput04;
	Cyclic#1.P3_Srobovanie.IN.SkrutkM5_SnimacVakua_S29 AT %IX."DI3.4_8DI".DigitalInput05;
	Cyclic#1.P3_Srobovanie.IN.SkrutkK40_SrobaPresla_IS81 AT %IX."DI3.4_8DI".DigitalInput08;
	Cyclic#1.P3_LeakageTestA.PAR.SnimacTlaku_IOLinkInputs AT %IO."DS3_2".InputData01;
	Cyclic#1.P3_LeakageTestB.PAR.SnimacTlaku_IOLinkInputs AT %IO."DS3_2".InputData02;
	Cyclic#1.AteqLeakageTester_A.Profinet_PLC_INPUTS[1] AT %IB."LeakageTester_A".Module001_Inputs001;
	Cyclic#1.AteqLeakageTester_A.Profinet_PLC_INPUTS[2] AT %IB."LeakageTester_A".Module001_Inputs002;
	Cyclic#1.AteqLeakageTester_A.Profinet_PLC_INPUTS[3] AT %IB."LeakageTester_A".Module001_Inputs003;
	Cyclic#1.AteqLeakageTester_A.Profinet_PLC_INPUTS[4] AT %IB."LeakageTester_A".Module001_Inputs004;
	Cyclic#1.AteqLeakageTester_A.Profinet_PLC_INPUTS[5] AT %IB."LeakageTester_A".Module001_Inputs005;
	Cyclic#1.AteqLeakageTester_A.Profinet_PLC_INPUTS[6] AT %IB."LeakageTester_A".Module001_Inputs006;
	Cyclic#1.AteqLeakageTester_A.Profinet_PLC_INPUTS[7] AT %IB."LeakageTester_A".Module001_Inputs007;
	Cyclic#1.AteqLeakageTester_A.Profinet_PLC_INPUTS[8] AT %IB."LeakageTester_A".Module001_Inputs008;
	Cyclic#1.AteqLeakageTester_A.Profinet_PLC_INPUTS[9] AT %IB."LeakageTester_A".Module001_Inputs009;
	Cyclic#1.AteqLeakageTester_A.Profinet_PLC_INPUTS[10] AT %IB."LeakageTester_A".Module001_Inputs010;
	Cyclic#1.AteqLeakageTester_A.Profinet_PLC_INPUTS[11] AT %IB."LeakageTester_A".Module001_Inputs011;
	Cyclic#1.AteqLeakageTester_A.Profinet_PLC_INPUTS[12] AT %IB."LeakageTester_A".Module001_Inputs012;
	Cyclic#1.AteqLeakageTester_A.Profinet_PLC_INPUTS[13] AT %IB."LeakageTester_A".Module001_Inputs013;
	Cyclic#1.AteqLeakageTester_A.Profinet_PLC_OUTPUTS[1] AT %QB."LeakageTester_A".Module002_Outputs001;
	Cyclic#1.AteqLeakageTester_A.Profinet_PLC_OUTPUTS[2] AT %QB."LeakageTester_A".Module002_Outputs002;
	Cyclic#1.AteqLeakageTester_A.Profinet_PLC_OUTPUTS[3] AT %QB."LeakageTester_A".Module002_Outputs003;
	Cyclic#1.AteqLeakageTester_A.Profinet_PLC_OUTPUTS[4] AT %QB."LeakageTester_A".Module002_Outputs004;
	Cyclic#1.AteqLeakageTester_A.Profinet_PLC_OUTPUTS[5] AT %QB."LeakageTester_A".Module002_Outputs005;
	Cyclic#1.AteqLeakageTester_A.Profinet_PLC_OUTPUTS[6] AT %QB."LeakageTester_A".Module002_Outputs006;
	Cyclic#1.AteqLeakageTester_A.Profinet_PLC_OUTPUTS[7] AT %QB."LeakageTester_A".Module002_Outputs007;
	Cyclic#1.AteqLeakageTester_A.Profinet_PLC_OUTPUTS[8] AT %QB."LeakageTester_A".Module002_Outputs008;
	Cyclic#1.AteqLeakageTester_A.Profinet_PLC_OUTPUTS[9] AT %QB."LeakageTester_A".Module002_Outputs009;
	Cyclic#1.AteqLeakageTester_A.Profinet_PLC_OUTPUTS[10] AT %QB."LeakageTester_A".Module002_Outputs010;
	Cyclic#1.AteqLeakageTester_A.Profinet_PLC_OUTPUTS[11] AT %QB."LeakageTester_A".Module002_Outputs011;
	Cyclic#1.AteqLeakageTester_A.Profinet_PLC_OUTPUTS[12] AT %QB."LeakageTester_A".Module002_Outputs012;
	Cyclic#1.AteqLeakageTester_A.Profinet_PLC_OUTPUTS[13] AT %QB."LeakageTester_A".Module002_Outputs013;
	Cyclic#1.AteqLeakageTester_A.Profinet_PLC_OUTPUTS[14] AT %QB."LeakageTester_A".Module002_Outputs014;
	Cyclic#1.AteqLeakageTester_A.Profinet_PLC_OUTPUTS[15] AT %QB."LeakageTester_A".Module002_Outputs015;
	Cyclic#1.AteqLeakageTester_A.Profinet_PLC_OUTPUTS[16] AT %QB."LeakageTester_A".Module002_Outputs016;
	Cyclic#1.AteqLeakageTester_B.Profinet_PLC_INPUTS[1] AT %IB."LeakageTester_B".Module001_Inputs001;
	Cyclic#1.AteqLeakageTester_B.Profinet_PLC_OUTPUTS[1] AT %QB."LeakageTester_B".Module002_Outputs001;
	Cyclic#1.AteqLeakageTester_B.Profinet_PLC_INPUTS[2] AT %IB."LeakageTester_B".Module001_Inputs002;
	Cyclic#1.AteqLeakageTester_B.Profinet_PLC_INPUTS[3] AT %IB."LeakageTester_B".Module001_Inputs003;
	Cyclic#1.AteqLeakageTester_B.Profinet_PLC_INPUTS[4] AT %IB."LeakageTester_B".Module001_Inputs004;
	Cyclic#1.AteqLeakageTester_B.Profinet_PLC_INPUTS[5] AT %IB."LeakageTester_B".Module001_Inputs005;
	Cyclic#1.AteqLeakageTester_B.Profinet_PLC_INPUTS[6] AT %IB."LeakageTester_B".Module001_Inputs006;
	Cyclic#1.AteqLeakageTester_B.Profinet_PLC_INPUTS[7] AT %IB."LeakageTester_B".Module001_Inputs007;
	Cyclic#1.AteqLeakageTester_B.Profinet_PLC_INPUTS[8] AT %IB."LeakageTester_B".Module001_Inputs008;
	Cyclic#1.AteqLeakageTester_B.Profinet_PLC_INPUTS[9] AT %IB."LeakageTester_B".Module001_Inputs009;
	Cyclic#1.AteqLeakageTester_B.Profinet_PLC_INPUTS[10] AT %IB."LeakageTester_B".Module001_Inputs010;
	Cyclic#1.AteqLeakageTester_B.Profinet_PLC_INPUTS[11] AT %IB."LeakageTester_B".Module001_Inputs011;
	Cyclic#1.AteqLeakageTester_B.Profinet_PLC_INPUTS[12] AT %IB."LeakageTester_B".Module001_Inputs012;
	Cyclic#1.AteqLeakageTester_B.Profinet_PLC_INPUTS[13] AT %IB."LeakageTester_B".Module001_Inputs013;
	Cyclic#1.AteqLeakageTester_B.Profinet_PLC_OUTPUTS[2] AT %QB."LeakageTester_B".Module002_Outputs002;
	Cyclic#1.AteqLeakageTester_B.Profinet_PLC_OUTPUTS[3] AT %QB."LeakageTester_B".Module002_Outputs003;
	Cyclic#1.AteqLeakageTester_B.Profinet_PLC_OUTPUTS[4] AT %QB."LeakageTester_B".Module002_Outputs004;
	Cyclic#1.AteqLeakageTester_B.Profinet_PLC_OUTPUTS[5] AT %QB."LeakageTester_B".Module002_Outputs005;
	Cyclic#1.AteqLeakageTester_B.Profinet_PLC_OUTPUTS[6] AT %QB."LeakageTester_B".Module002_Outputs006;
	Cyclic#1.AteqLeakageTester_B.Profinet_PLC_OUTPUTS[7] AT %QB."LeakageTester_B".Module002_Outputs007;
	Cyclic#1.AteqLeakageTester_B.Profinet_PLC_OUTPUTS[8] AT %QB."LeakageTester_B".Module002_Outputs008;
	Cyclic#1.AteqLeakageTester_B.Profinet_PLC_OUTPUTS[9] AT %QB."LeakageTester_B".Module002_Outputs009;
	Cyclic#1.AteqLeakageTester_B.Profinet_PLC_OUTPUTS[10] AT %QB."LeakageTester_B".Module002_Outputs010;
	Cyclic#1.AteqLeakageTester_B.Profinet_PLC_OUTPUTS[11] AT %QB."LeakageTester_B".Module002_Outputs011;
	Cyclic#1.AteqLeakageTester_B.Profinet_PLC_OUTPUTS[12] AT %QB."LeakageTester_B".Module002_Outputs012;
	Cyclic#1.AteqLeakageTester_B.Profinet_PLC_OUTPUTS[13] AT %QB."LeakageTester_B".Module002_Outputs013;
	Cyclic#1.AteqLeakageTester_B.Profinet_PLC_OUTPUTS[14] AT %QB."LeakageTester_B".Module002_Outputs014;
	Cyclic#1.AteqLeakageTester_B.Profinet_PLC_OUTPUTS[15] AT %QB."LeakageTester_B".Module002_Outputs015;
	Cyclic#1.AteqLeakageTester_B.Profinet_PLC_OUTPUTS[16] AT %QB."LeakageTester_B".Module002_Outputs016;
	Cyclic#1.P4_Etiketovacka.IN.Tlaciaren_ERROR AT %IX."AB4.6_16xDI".DigitalInput14;
	Cyclic#1.P4_Etiketovacka.IN.Tlaciaren_READY AT %IX."AB4.6_16xDI".DigitalInput15;
	Cyclic#1.P4_Etiketovacka.IN.Tlaciaren_DochadzaPaska AT %IX."AB4.6_16xDI".DigitalInput16;
	Cyclic#1.P4_Etiketovacka.OUT.Tlaciaren_START_Tlace AT %QX."AB4.7_16xDO".DigitalOutput15;
	Cyclic#1.P4_Etiketovacka.OUT.Tlaciaren_RESET_Poruchy AT %QX."AB4.7_16xDO".DigitalOutput16;
	Cyclic#1.P4_FunkcnyTestA.IN.TypSpodnychKontaktov_4F AT %IX."DM4.1".DigitalInput04;
	Cyclic#1.P4_FunkcnyTestB.IN.TypSpodnychKontaktov_4F AT %IX."DM4.1".DigitalInput06;
	Cyclic#1.P4_FunkcnyTestB.IN.TypSpodnychKontaktov_5F_5H AT %IX."DM4.1".DigitalInput05;
	Cyclic#1.Safety.OUT.P4_ZamkniZamok_PredneDvere AT %QX."DM4.1".DigitalOutput01;
	Cyclic#1.Safety.IN.P4_PredneDvere_PritomPetlice AT %IX."DM4.1".DigitalInput02;
	Cyclic#1.P4_FunkcnyTestA.IN.TypSpodnychKontaktov_5F_5H AT %IX."DM4.1".DigitalInput03;
	Cyclic#1.P3_LeakageTestA.PAR.SnimacTlaku_IOLinkInputs AT %IW."DS3_2".InputData01_1;
	Cyclic#1.P3_LeakageTestB.PAR.SnimacTlaku_IOLinkInputs AT %IW."DS3_2".InputData02_1;
	Cyclic#1.ControlUnit.Profinet_PLC_INPUTS[0] AT %IB."KAM_ControlUNit".Module001_Inputs001;
	Cyclic#1.ControlUnit.Profinet_PLC_INPUTS[1] AT %IB."KAM_ControlUNit".Module001_Inputs002;
	Cyclic#1.CAM2.Profinet_PLC_INPUTS[0] AT %IB."KAM_ControlUNit".Module002_Inputs001;
	Cyclic#1.CAM2.Profinet_PLC_INPUTS[1] AT %IB."KAM_ControlUNit".Module002_Inputs002;
	Cyclic#1.CAM2.Profinet_PLC_INPUTS[2] AT %IB."KAM_ControlUNit".Module002_Inputs003;
	Cyclic#1.CAM4.Profinet_PLC_INPUTS[0] AT %IB."KAM_ControlUNit".Module004_Inputs001;
	Cyclic#1.CAM4.Profinet_PLC_INPUTS[1] AT %IB."KAM_ControlUNit".Module004_Inputs002;
	Cyclic#1.CAM6.Profinet_PLC_INPUTS[0] AT %IB."KAM_ControlUNit".Module006_Inputs001;
	Cyclic#1.CAM6.Profinet_PLC_INPUTS[1] AT %IB."KAM_ControlUNit".Module006_Inputs002;
	Cyclic#1.CAM6.Profinet_PLC_INPUTS[2] AT %IB."KAM_ControlUNit".Module006_Inputs003;
	Cyclic#1.CAM6.Profinet_PLC_INPUTS[3] AT %IB."KAM_ControlUNit".Module006_Inputs004;
	Cyclic#1.CAM2.Profinet_PLC_OUTPUTS[0] AT %QB."KAM_ControlUNit".Module026_Outputs001;
	Cyclic#1.CAM4.Profinet_PLC_OUTPUTS[0] AT %QB."KAM_ControlUNit".Module027_Outputs001;
	Cyclic#1.CAM6.Profinet_PLC_OUTPUTS[0] AT %QB."KAM_ControlUNit".Module028_Outputs001;
	Cyclic#1.CAM1.Profinet_PLC_OUTPUTS[0] AT %QB."KAM_ControlUNit".Module029_Outputs001;
	Cyclic#1.CAM7.Profinet_PLC_OUTPUTS[0] AT %QB."KAM_ControlUNit".Module030_Outputs001;
	Cyclic#1.CAM17.Profinet_PLC_OUTPUTS[0] AT %QB."KAM_ControlUNit".Module031_Outputs001;
	Cyclic#1.CAM10.Profinet_PLC_OUTPUTS[0] AT %QB."KAM_ControlUNit".Module032_Outputs001;
	Cyclic#1.CAM11.Profinet_PLC_OUTPUTS[0] AT %QB."KAM_ControlUNit".Module033_Outputs001;
	Cyclic#1.CAM12.Profinet_PLC_OUTPUTS[0] AT %QB."KAM_ControlUNit".Module034_Outputs001;
	Cyclic#1.CAM13.Profinet_PLC_OUTPUTS[0] AT %QB."KAM_ControlUNit".Module035_Outputs001;
	Cyclic#1.CAM15.Profinet_PLC_OUTPUTS[0] AT %QB."KAM_ControlUNit".Module036_Outputs001;
	Cyclic#1.CAM16.Profinet_PLC_OUTPUTS[0] AT %QB."KAM_ControlUNit".Module037_Outputs001;
	Cyclic#1.CAM2.Profinet_PLC_INPUTS[3] AT %IB."KAM_ControlUNit".Module002_Inputs004;
	Cyclic#1.CAM4.Profinet_PLC_INPUTS[2] AT %IB."KAM_ControlUNit".Module004_Inputs003;
	Cyclic#1.CAM4.Profinet_PLC_INPUTS[3] AT %IB."KAM_ControlUNit".Module004_Inputs004;
	Cyclic#1.CAM6.Profinet_PLC_INPUTS[4] AT %IB."KAM_ControlUNit".Module006_Inputs005;
	Cyclic#1.CAM6.Profinet_PLC_INPUTS[5] AT %IB."KAM_ControlUNit".Module006_Inputs006;
	Cyclic#1.Safety.OUT.P3_ZamkniZamok_PredneDvereLS AT %QX."DM3.1".DigitalOutput01;
	Cyclic#1.Safety.OUT.P3_ZamkniZamok_PredneDverePS AT %QX."DM3.1".DigitalOutput03;
	Cyclic#1.Safety.OUT.P3_ZamkniZamok_ZadneDvere AT %QX."DM3.1".DigitalOutput05;
	Cyclic#1.Safety.IN.P3_PredneDvereLS_PritomPetlice AT %IX."DM3.1".DigitalInput02;
	Cyclic#1.Safety.IN.P3_PredneDverePS_PritomPetlice AT %IX."DM3.1".DigitalInput04;
	Cyclic#1.Safety.IN.P3_ZadneDvere_PritomPetlice AT %IX."DM3.1".DigitalInput06;
	Cyclic#1.P3_Srobovanie.OUT.ZasobSrobM5_Banner_CervenaLED AT %QX."DM3.1".DigitalOutput07;
	Cyclic#1.P3_Srobovanie.OUT.ZasobSrobK40_Banner_CervenaLED AT %QX."DM3.1".DigitalOutput09;
	Cyclic#1.P3_Srobovanie.IN.ZasobSrobM5_Banner_SB12 AT %IX."DM3.1".DigitalInput08;
	Cyclic#1.P3_Srobovanie.IN.ZasobSrobK40_Banner_SB13 AT %IX."DM3.1".DigitalInput10;
	Cyclic#1.CAM3.Profinet_QRkod_Znaky[0] AT %IB."P1_KAM3".Module004_Input_64_Byte001;
	Cyclic#1.CAM3.Profinet_QRkod_Znaky[1] AT %IB."P1_KAM3".Module004_Input_64_Byte002;
	Cyclic#1.CAM3.Profinet_QRkod_Znaky[2] AT %IB."P1_KAM3".Module004_Input_64_Byte003;
	Cyclic#1.CAM3.Profinet_QRkod_Znaky[3] AT %IB."P1_KAM3".Module004_Input_64_Byte004;
	Cyclic#1.CAM3.Profinet_QRkod_Znaky[4] AT %IB."P1_KAM3".Module004_Input_64_Byte005;
	Cyclic#1.CAM3.Profinet_QRkod_Znaky[5] AT %IB."P1_KAM3".Module004_Input_64_Byte006;
	Cyclic#1.CAM3.Profinet_QRkod_Znaky[6] AT %IB."P1_KAM3".Module004_Input_64_Byte007;
	Cyclic#1.CAM3.Profinet_QRkod_Znaky[7] AT %IB."P1_KAM3".Module004_Input_64_Byte008;
	Cyclic#1.CAM3.Profinet_QRkod_Znaky[8] AT %IB."P1_KAM3".Module004_Input_64_Byte009;
	Cyclic#1.CAM3.Profinet_QRkod_Znaky[9] AT %IB."P1_KAM3".Module004_Input_64_Byte010;
	Cyclic#1.CAM3.Profinet_QRkod_Znaky[10] AT %IB."P1_KAM3".Module004_Input_64_Byte011;
	Cyclic#1.CAM3.Profinet_QRkod_Znaky[11] AT %IB."P1_KAM3".Module004_Input_64_Byte012;
	Cyclic#1.CAM3.Profinet_QRkod_Znaky[12] AT %IB."P1_KAM3".Module004_Input_64_Byte013;
	Cyclic#1.CAM3.Profinet_QRkod_Znaky[13] AT %IB."P1_KAM3".Module004_Input_64_Byte014;
	Cyclic#1.CAM3.Profinet_QRkod_Znaky[14] AT %IB."P1_KAM3".Module004_Input_64_Byte015;
	Cyclic#1.CAM3.Profinet_QRkod_Znaky[15] AT %IB."P1_KAM3".Module004_Input_64_Byte016;
	Cyclic#1.CAM3.Profinet_QRkod_Znaky[16] AT %IB."P1_KAM3".Module004_Input_64_Byte017;
	Cyclic#1.CAM3.Profinet_QRkod_Znaky[17] AT %IB."P1_KAM3".Module004_Input_64_Byte018;
	Cyclic#1.CAM3.Profinet_QRkod_Znaky[18] AT %IB."P1_KAM3".Module004_Input_64_Byte019;
	Cyclic#1.CAM3.Profinet_QRkod_Znaky[19] AT %IB."P1_KAM3".Module004_Input_64_Byte020;
	Cyclic#1.CAM3.Profinet_QRkod_Znaky[20] AT %IB."P1_KAM3".Module004_Input_64_Byte021;
	Cyclic#1.CAM3.Profinet_QRkod_Znaky[21] AT %IB."P1_KAM3".Module004_Input_64_Byte022;
	Cyclic#1.CAM3.Profinet_QRkod_Znaky[22] AT %IB."P1_KAM3".Module004_Input_64_Byte023;
	Cyclic#1.CAM3.Profinet_QRkod_Znaky[23] AT %IB."P1_KAM3".Module004_Input_64_Byte024;
	Cyclic#1.CAM3.Profinet_QRkod_Znaky[24] AT %IB."P1_KAM3".Module004_Input_64_Byte025;
	Cyclic#1.CAM3.Profinet_QRkod_Znaky[25] AT %IB."P1_KAM3".Module004_Input_64_Byte026;
	Cyclic#1.CAM3.Profinet_QRkod_Znaky[26] AT %IB."P1_KAM3".Module004_Input_64_Byte027;
	Cyclic#1.CAM3.Profinet_QRkod_Znaky[27] AT %IB."P1_KAM3".Module004_Input_64_Byte028;
	Cyclic#1.CAM3.Profinet_QRkod_Znaky[28] AT %IB."P1_KAM3".Module004_Input_64_Byte029;
	Cyclic#1.CAM3.Profinet_QRkod_Znaky[29] AT %IB."P1_KAM3".Module004_Input_64_Byte030;
	Cyclic#1.CAM3.Profinet_QRkod_Znaky[30] AT %IB."P1_KAM3".Module004_Input_64_Byte031;
	Cyclic#1.CAM3.Profinet_QRkod_Znaky[31] AT %IB."P1_KAM3".Module004_Input_64_Byte032;
	Cyclic#1.CAM3.STAV.READY AT %IX."P1_KAM3".ModuleOk;
	Cyclic#1.CAM3.Profinet_PLC_INPUTS[10] AT %IB."P1_KAM3".Module006_Input_16_Byte012;
	Cyclic#1.CAM3.Profinet_PLC_INPUTS[0] AT %IB."P1_KAM3".Module005_Input_1_Byte;
	Cyclic#1.CAM3.Profinet_PLC_OUTPUTS[0] AT %QB."P1_KAM3".Module003_Output_1_Byte;
	Cyclic#1.CAM5.STAV.READY AT %IX."P1_KAM5".ModuleOk;
	Cyclic#1.CAM5.Profinet_PLC_OUTPUTS[0] AT %QB."P1_KAM5".Module003_Output_1_Byte;
	Cyclic#1.CAM5.Profinet_QRkod_Znaky[0] AT %IB."P1_KAM5".Module004_Input_64_Byte001;
	Cyclic#1.CAM5.Profinet_QRkod_Znaky[1] AT %IB."P1_KAM5".Module004_Input_64_Byte002;
	Cyclic#1.CAM5.Profinet_QRkod_Znaky[2] AT %IB."P1_KAM5".Module004_Input_64_Byte003;
	Cyclic#1.CAM5.Profinet_QRkod_Znaky[3] AT %IB."P1_KAM5".Module004_Input_64_Byte004;
	Cyclic#1.CAM5.Profinet_QRkod_Znaky[4] AT %IB."P1_KAM5".Module004_Input_64_Byte005;
	Cyclic#1.CAM5.Profinet_QRkod_Znaky[5] AT %IB."P1_KAM5".Module004_Input_64_Byte006;
	Cyclic#1.CAM5.Profinet_QRkod_Znaky[6] AT %IB."P1_KAM5".Module004_Input_64_Byte007;
	Cyclic#1.CAM5.Profinet_QRkod_Znaky[7] AT %IB."P1_KAM5".Module004_Input_64_Byte008;
	Cyclic#1.CAM5.Profinet_QRkod_Znaky[8] AT %IB."P1_KAM5".Module004_Input_64_Byte009;
	Cyclic#1.CAM5.Profinet_QRkod_Znaky[9] AT %IB."P1_KAM5".Module004_Input_64_Byte010;
	Cyclic#1.CAM5.Profinet_QRkod_Znaky[10] AT %IB."P1_KAM5".Module004_Input_64_Byte011;
	Cyclic#1.CAM5.Profinet_QRkod_Znaky[11] AT %IB."P1_KAM5".Module004_Input_64_Byte012;
	Cyclic#1.CAM5.Profinet_QRkod_Znaky[12] AT %IB."P1_KAM5".Module004_Input_64_Byte013;
	Cyclic#1.CAM5.Profinet_QRkod_Znaky[13] AT %IB."P1_KAM5".Module004_Input_64_Byte014;
	Cyclic#1.CAM5.Profinet_QRkod_Znaky[14] AT %IB."P1_KAM5".Module004_Input_64_Byte015;
	Cyclic#1.CAM5.Profinet_QRkod_Znaky[15] AT %IB."P1_KAM5".Module004_Input_64_Byte016;
	Cyclic#1.CAM5.Profinet_QRkod_Znaky[16] AT %IB."P1_KAM5".Module004_Input_64_Byte017;
	Cyclic#1.CAM5.Profinet_QRkod_Znaky[17] AT %IB."P1_KAM5".Module004_Input_64_Byte018;
	Cyclic#1.CAM5.Profinet_QRkod_Znaky[18] AT %IB."P1_KAM5".Module004_Input_64_Byte019;
	Cyclic#1.CAM5.Profinet_QRkod_Znaky[19] AT %IB."P1_KAM5".Module004_Input_64_Byte020;
	Cyclic#1.CAM5.Profinet_QRkod_Znaky[20] AT %IB."P1_KAM5".Module004_Input_64_Byte021;
	Cyclic#1.CAM5.Profinet_QRkod_Znaky[21] AT %IB."P1_KAM5".Module004_Input_64_Byte022;
	Cyclic#1.CAM5.Profinet_QRkod_Znaky[22] AT %IB."P1_KAM5".Module004_Input_64_Byte023;
	Cyclic#1.CAM5.Profinet_QRkod_Znaky[23] AT %IB."P1_KAM5".Module004_Input_64_Byte024;
	Cyclic#1.CAM5.Profinet_QRkod_Znaky[24] AT %IB."P1_KAM5".Module004_Input_64_Byte025;
	Cyclic#1.CAM5.Profinet_QRkod_Znaky[25] AT %IB."P1_KAM5".Module004_Input_64_Byte026;
	Cyclic#1.CAM5.Profinet_QRkod_Znaky[26] AT %IB."P1_KAM5".Module004_Input_64_Byte027;
	Cyclic#1.CAM5.Profinet_QRkod_Znaky[27] AT %IB."P1_KAM5".Module004_Input_64_Byte028;
	Cyclic#1.CAM5.Profinet_QRkod_Znaky[28] AT %IB."P1_KAM5".Module004_Input_64_Byte029;
	Cyclic#1.CAM5.Profinet_QRkod_Znaky[29] AT %IB."P1_KAM5".Module004_Input_64_Byte030;
	Cyclic#1.CAM5.Profinet_QRkod_Znaky[30] AT %IB."P1_KAM5".Module004_Input_64_Byte031;
	Cyclic#1.CAM5.Profinet_QRkod_Znaky[31] AT %IB."P1_KAM5".Module004_Input_64_Byte032;
	Cyclic#1.CAM5.Profinet_PLC_INPUTS[0] AT %IB."P1_KAM5".Module005_Input_1_Byte;
	Cyclic#1.CAM5.Profinet_PLC_INPUTS[10] AT %IB."P1_KAM5".Module006_Input_16_Byte012;
	Cyclic#1.CAM8.STAV.READY AT %IX."P2_KAM8".ModuleOk;
	Cyclic#1.CAM8.Profinet_PLC_OUTPUTS[0] AT %QB."P2_KAM8".Module003_Output_1_Byte;
	Cyclic#1.CAM8.Profinet_QRkod_Znaky[0] AT %IB."P2_KAM8".Module004_Input_64_Byte001;
	Cyclic#1.CAM8.Profinet_QRkod_Znaky[1] AT %IB."P2_KAM8".Module004_Input_64_Byte002;
	Cyclic#1.CAM8.Profinet_QRkod_Znaky[2] AT %IB."P2_KAM8".Module004_Input_64_Byte003;
	Cyclic#1.CAM8.Profinet_QRkod_Znaky[3] AT %IB."P2_KAM8".Module004_Input_64_Byte004;
	Cyclic#1.CAM8.Profinet_QRkod_Znaky[4] AT %IB."P2_KAM8".Module004_Input_64_Byte005;
	Cyclic#1.CAM8.Profinet_QRkod_Znaky[5] AT %IB."P2_KAM8".Module004_Input_64_Byte006;
	Cyclic#1.CAM8.Profinet_QRkod_Znaky[6] AT %IB."P2_KAM8".Module004_Input_64_Byte007;
	Cyclic#1.CAM8.Profinet_QRkod_Znaky[7] AT %IB."P2_KAM8".Module004_Input_64_Byte008;
	Cyclic#1.CAM8.Profinet_QRkod_Znaky[8] AT %IB."P2_KAM8".Module004_Input_64_Byte009;
	Cyclic#1.CAM8.Profinet_QRkod_Znaky[9] AT %IB."P2_KAM8".Module004_Input_64_Byte010;
	Cyclic#1.CAM8.Profinet_QRkod_Znaky[10] AT %IB."P2_KAM8".Module004_Input_64_Byte011;
	Cyclic#1.CAM8.Profinet_QRkod_Znaky[11] AT %IB."P2_KAM8".Module004_Input_64_Byte012;
	Cyclic#1.CAM8.Profinet_QRkod_Znaky[12] AT %IB."P2_KAM8".Module004_Input_64_Byte013;
	Cyclic#1.CAM8.Profinet_QRkod_Znaky[13] AT %IB."P2_KAM8".Module004_Input_64_Byte014;
	Cyclic#1.CAM8.Profinet_QRkod_Znaky[14] AT %IB."P2_KAM8".Module004_Input_64_Byte015;
	Cyclic#1.CAM8.Profinet_QRkod_Znaky[15] AT %IB."P2_KAM8".Module004_Input_64_Byte016;
	Cyclic#1.CAM8.Profinet_QRkod_Znaky[16] AT %IB."P2_KAM8".Module004_Input_64_Byte017;
	Cyclic#1.CAM8.Profinet_QRkod_Znaky[17] AT %IB."P2_KAM8".Module004_Input_64_Byte018;
	Cyclic#1.CAM8.Profinet_QRkod_Znaky[18] AT %IB."P2_KAM8".Module004_Input_64_Byte019;
	Cyclic#1.CAM8.Profinet_QRkod_Znaky[19] AT %IB."P2_KAM8".Module004_Input_64_Byte020;
	Cyclic#1.CAM8.Profinet_QRkod_Znaky[20] AT %IB."P2_KAM8".Module004_Input_64_Byte021;
	Cyclic#1.CAM8.Profinet_QRkod_Znaky[21] AT %IB."P2_KAM8".Module004_Input_64_Byte022;
	Cyclic#1.CAM8.Profinet_QRkod_Znaky[22] AT %IB."P2_KAM8".Module004_Input_64_Byte023;
	Cyclic#1.CAM8.Profinet_QRkod_Znaky[23] AT %IB."P2_KAM8".Module004_Input_64_Byte024;
	Cyclic#1.CAM8.Profinet_QRkod_Znaky[24] AT %IB."P2_KAM8".Module004_Input_64_Byte025;
	Cyclic#1.CAM8.Profinet_QRkod_Znaky[25] AT %IB."P2_KAM8".Module004_Input_64_Byte026;
	Cyclic#1.CAM8.Profinet_QRkod_Znaky[26] AT %IB."P2_KAM8".Module004_Input_64_Byte027;
	Cyclic#1.CAM8.Profinet_QRkod_Znaky[27] AT %IB."P2_KAM8".Module004_Input_64_Byte028;
	Cyclic#1.CAM8.Profinet_QRkod_Znaky[28] AT %IB."P2_KAM8".Module004_Input_64_Byte029;
	Cyclic#1.CAM8.Profinet_QRkod_Znaky[29] AT %IB."P2_KAM8".Module004_Input_64_Byte030;
	Cyclic#1.CAM8.Profinet_QRkod_Znaky[30] AT %IB."P2_KAM8".Module004_Input_64_Byte031;
	Cyclic#1.CAM8.Profinet_QRkod_Znaky[31] AT %IB."P2_KAM8".Module004_Input_64_Byte032;
	Cyclic#1.CAM8.Profinet_PLC_INPUTS[0] AT %IB."P2_KAM8".Module005_Input_1_Byte;
	Cyclic#1.CAM8.Profinet_PLC_INPUTS[10] AT %IB."P2_KAM8".Module006_Input_16_Byte012;
	Cyclic#1.CAM14.STAV.READY AT %IX."P4_KAM14".ModuleOk;
	Cyclic#1.CAM14.Profinet_PLC_OUTPUTS[0] AT %QB."P4_KAM14".Module003_Output_1_Byte;
	Cyclic#1.CAM14.Profinet_QRkod_Znaky[0] AT %IB."P4_KAM14".Module004_Input_64_Byte001;
	Cyclic#1.CAM14.Profinet_QRkod_Znaky[1] AT %IB."P4_KAM14".Module004_Input_64_Byte002;
	Cyclic#1.CAM14.Profinet_QRkod_Znaky[2] AT %IB."P4_KAM14".Module004_Input_64_Byte003;
	Cyclic#1.CAM14.Profinet_QRkod_Znaky[3] AT %IB."P4_KAM14".Module004_Input_64_Byte004;
	Cyclic#1.CAM14.Profinet_QRkod_Znaky[4] AT %IB."P4_KAM14".Module004_Input_64_Byte005;
	Cyclic#1.CAM14.Profinet_QRkod_Znaky[5] AT %IB."P4_KAM14".Module004_Input_64_Byte006;
	Cyclic#1.CAM14.Profinet_QRkod_Znaky[6] AT %IB."P4_KAM14".Module004_Input_64_Byte007;
	Cyclic#1.CAM14.Profinet_QRkod_Znaky[7] AT %IB."P4_KAM14".Module004_Input_64_Byte008;
	Cyclic#1.CAM14.Profinet_QRkod_Znaky[8] AT %IB."P4_KAM14".Module004_Input_64_Byte009;
	Cyclic#1.CAM14.Profinet_QRkod_Znaky[9] AT %IB."P4_KAM14".Module004_Input_64_Byte010;
	Cyclic#1.CAM14.Profinet_QRkod_Znaky[10] AT %IB."P4_KAM14".Module004_Input_64_Byte011;
	Cyclic#1.CAM14.Profinet_QRkod_Znaky[11] AT %IB."P4_KAM14".Module004_Input_64_Byte012;
	Cyclic#1.CAM14.Profinet_QRkod_Znaky[12] AT %IB."P4_KAM14".Module004_Input_64_Byte013;
	Cyclic#1.CAM14.Profinet_QRkod_Znaky[13] AT %IB."P4_KAM14".Module004_Input_64_Byte014;
	Cyclic#1.CAM14.Profinet_QRkod_Znaky[14] AT %IB."P4_KAM14".Module004_Input_64_Byte015;
	Cyclic#1.CAM14.Profinet_QRkod_Znaky[15] AT %IB."P4_KAM14".Module004_Input_64_Byte016;
	Cyclic#1.CAM14.Profinet_QRkod_Znaky[16] AT %IB."P4_KAM14".Module004_Input_64_Byte017;
	Cyclic#1.CAM14.Profinet_QRkod_Znaky[17] AT %IB."P4_KAM14".Module004_Input_64_Byte018;
	Cyclic#1.CAM14.Profinet_QRkod_Znaky[18] AT %IB."P4_KAM14".Module004_Input_64_Byte019;
	Cyclic#1.CAM14.Profinet_QRkod_Znaky[19] AT %IB."P4_KAM14".Module004_Input_64_Byte020;
	Cyclic#1.CAM14.Profinet_QRkod_Znaky[20] AT %IB."P4_KAM14".Module004_Input_64_Byte021;
	Cyclic#1.CAM14.Profinet_QRkod_Znaky[21] AT %IB."P4_KAM14".Module004_Input_64_Byte022;
	Cyclic#1.CAM14.Profinet_QRkod_Znaky[22] AT %IB."P4_KAM14".Module004_Input_64_Byte023;
	Cyclic#1.CAM14.Profinet_QRkod_Znaky[23] AT %IB."P4_KAM14".Module004_Input_64_Byte024;
	Cyclic#1.CAM14.Profinet_QRkod_Znaky[24] AT %IB."P4_KAM14".Module004_Input_64_Byte025;
	Cyclic#1.CAM14.Profinet_QRkod_Znaky[25] AT %IB."P4_KAM14".Module004_Input_64_Byte026;
	Cyclic#1.CAM14.Profinet_QRkod_Znaky[26] AT %IB."P4_KAM14".Module004_Input_64_Byte027;
	Cyclic#1.CAM14.Profinet_QRkod_Znaky[27] AT %IB."P4_KAM14".Module004_Input_64_Byte028;
	Cyclic#1.CAM14.Profinet_QRkod_Znaky[28] AT %IB."P4_KAM14".Module004_Input_64_Byte029;
	Cyclic#1.CAM14.Profinet_QRkod_Znaky[29] AT %IB."P4_KAM14".Module004_Input_64_Byte030;
	Cyclic#1.CAM14.Profinet_QRkod_Znaky[30] AT %IB."P4_KAM14".Module004_Input_64_Byte031;
	Cyclic#1.CAM14.Profinet_QRkod_Znaky[31] AT %IB."P4_KAM14".Module004_Input_64_Byte032;
	Cyclic#1.CAM14.Profinet_PLC_INPUTS[0] AT %IB."P4_KAM14".Module005_Input_1_Byte;
	Cyclic#1.CAM14.Profinet_PLC_INPUTS[10] AT %IB."P4_KAM14".Module006_Input_16_Byte012;
	Cyclic#1.CAM9.STAV.READY AT %IX."P2_KAM9".ModuleOk;
	Cyclic#1.CAM9.Profinet_PLC_OUTPUTS[0] AT %QB."P2_KAM9".Module003_Output_1_Byte;
	Cyclic#1.CAM9.Profinet_PLC_INPUTS[0] AT %IB."P2_KAM9".Module005_Input_1_Byte;
	Cyclic#1.CAM9.Profinet_PLC_INPUTS[10] AT %IB."P2_KAM9".Module006_Input_16_Byte012;
	Cyclic#1.P3_Pracovisko.STAV.LeakageTestA_OK AT %IX."LeakageTester_A".ModuleOk;
	Cyclic#1.P3_Pracovisko.STAV.LeakageTestB_OK AT %IX."LeakageTester_B".ModuleOk;
	Cyclic#1.P3_Pracovisko.STAV.VentilovyTerminal_VT6_OK AT %IX."VentilovyTerminal_VT6".ModuleOk;
	Cyclic#1.P3_Pracovisko.STAV.VentilovyTerminal_VT7_OK AT %IX."VentilovyTerminal_VT7".ModuleOk;
	Cyclic#1.P2_Pracovisko.STAV.VentilovyTerminal_VT1_OK AT %IX."VentilovyTerminal_VT1".ModuleOk;
	Cyclic#1.P2_Pracovisko.STAV.VentilovyTerminal_VT2_OK AT %IX."VentilovyTerminal_VT2".ModuleOk;
	Cyclic#1.P2_Pracovisko.STAV.VentilovyTerminal_VT3_OK AT %IX."VentilovyTerminal_VT3".ModuleOk;
	Cyclic#1.P2_Pracovisko.STAV.KOM_Robot_OK AT %IX."R2_IRB1200".ModuleOk;
	Cyclic#1.P2_Pracovisko.STAV.Skrutkovacka_M6_OK AT %IX."RJ2_P2_Srobovacka_M6".ModuleOk;
	Cyclic#1.P2_Pracovisko.STAV.Skrutkovacka_M5_OK AT %IX."RJ4_P2_Srobovacka_M5".ModuleOk;
	Cyclic#1.P2_Pracovisko.STAV.Skrutkovacka_M4_OK AT %IX."RJ3_P2_Srobovacka_M4".ModuleOk;
	Cyclic#1.P2_Pracovisko.STAV.Maticovacka_M4_OK AT %IX."RJ1_P2_SrobovackaMatic_M4".ModuleOk;
	Cyclic#1.P3_Pracovisko.STAV.Skrutkovacka_K40_OK AT %IX."P3_Srobovacka_K40".ModuleOk;
	Cyclic#1.P3_Pracovisko.STAV.Skrutkovacka_M5_OK AT %IX."P3_Srobovacka_M5".ModuleOk;
	Cyclic#1.P4_Pracovisko.STAV.VentilovyTerminal_VT8_OK AT %IX."VentilovyTerminal_VT8".ModuleOk;
	Cyclic#1.P1_Pracovisko.STAV.Skrutkovacka_K30_OK AT %IX."RJ5_P1_Srobovacka_K30".ModuleOk;
	Cyclic#1.P1_Pracovisko.STAV.Skrutkovacka_M5_OK AT %IX."RJ6_P1_Srobovacka_M5".ModuleOk;
	Cyclic#1.P1_Pracovisko.STAV.Skrutkovacka_M4_OK AT %IX."RJ7_P1_Srobovacka_M4".ModuleOk;
	Cyclic#1.P1_Pracovisko.STAV.KartaAB110_OK AT %IX."AB1.10_X2X".ModuleOk;
	Cyclic#1.P4_Etiketovacka.IN.PritlakPaskyOdisteny_IS84 AT %IX."DI4.1_8DI".DigitalInput08;
	Cyclic#1.CAM1.Profinet_PLC_INPUTS[0] AT %IB."KAM_ControlUNit".Module008_Inputs001;
	Cyclic#1.CAM1.Profinet_PLC_INPUTS[1] AT %IB."KAM_ControlUNit".Module008_Inputs002;
	Cyclic#1.CAM1.Profinet_PLC_INPUTS[2] AT %IB."KAM_ControlUNit".Module008_Inputs003;
	Cyclic#1.CAM7.Profinet_PLC_INPUTS[0] AT %IB."KAM_ControlUNit".Module010_Inputs001;
	Cyclic#1.CAM7.Profinet_PLC_INPUTS[1] AT %IB."KAM_ControlUNit".Module010_Inputs002;
	Cyclic#1.CAM7.Profinet_PLC_INPUTS[2] AT %IB."KAM_ControlUNit".Module010_Inputs003;
	Cyclic#1.CAM7.Profinet_PLC_INPUTS[3] AT %IB."KAM_ControlUNit".Module010_Inputs004;
	Cyclic#1.CAM1.Profinet_PLC_INPUTS[3] AT %IB."KAM_ControlUNit".Module008_Inputs004;
	Cyclic#1.CAM17.Profinet_PLC_INPUTS[0] AT %IB."KAM_ControlUNit".Module012_Inputs001;
	Cyclic#1.CAM17.Profinet_PLC_INPUTS[1] AT %IB."KAM_ControlUNit".Module012_Inputs002;
	Cyclic#1.CAM17.Profinet_PLC_INPUTS[2] AT %IB."KAM_ControlUNit".Module012_Inputs003;
	Cyclic#1.CAM17.Profinet_PLC_INPUTS[3] AT %IB."KAM_ControlUNit".Module012_Inputs004;
	Cyclic#1.CAM7.Profinet_QRkod_Znaky[0] AT %IB."KAM_ControlUNit".Module011_Inputs001;
	Cyclic#1.CAM7.Profinet_QRkod_Znaky[1] AT %IB."KAM_ControlUNit".Module011_Inputs002;
	Cyclic#1.CAM7.Profinet_QRkod_Znaky[2] AT %IB."KAM_ControlUNit".Module011_Inputs003;
	Cyclic#1.CAM7.Profinet_QRkod_Znaky[3] AT %IB."KAM_ControlUNit".Module011_Inputs004;
	Cyclic#1.CAM7.Profinet_QRkod_Znaky[4] AT %IB."KAM_ControlUNit".Module011_Inputs005;
	Cyclic#1.CAM7.Profinet_QRkod_Znaky[5] AT %IB."KAM_ControlUNit".Module011_Inputs006;
	Cyclic#1.CAM7.Profinet_QRkod_Znaky[6] AT %IB."KAM_ControlUNit".Module011_Inputs007;
	Cyclic#1.CAM7.Profinet_QRkod_Znaky[7] AT %IB."KAM_ControlUNit".Module011_Inputs008;
	Cyclic#1.CAM7.Profinet_QRkod_Znaky[8] AT %IB."KAM_ControlUNit".Module011_Inputs009;
	Cyclic#1.CAM7.Profinet_QRkod_Znaky[9] AT %IB."KAM_ControlUNit".Module011_Inputs010;
	Cyclic#1.CAM7.Profinet_QRkod_Znaky[10] AT %IB."KAM_ControlUNit".Module011_Inputs011;
	Cyclic#1.CAM7.Profinet_QRkod_Znaky[11] AT %IB."KAM_ControlUNit".Module011_Inputs012;
	Cyclic#1.CAM7.Profinet_QRkod_Znaky[12] AT %IB."KAM_ControlUNit".Module011_Inputs013;
	Cyclic#1.CAM7.Profinet_QRkod_Znaky[13] AT %IB."KAM_ControlUNit".Module011_Inputs014;
	Cyclic#1.CAM7.Profinet_QRkod_Znaky[14] AT %IB."KAM_ControlUNit".Module011_Inputs015;
	Cyclic#1.CAM7.Profinet_QRkod_Znaky[15] AT %IB."KAM_ControlUNit".Module011_Inputs016;
	Cyclic#1.CAM7.Profinet_QRkod_Znaky[16] AT %IB."KAM_ControlUNit".Module011_Inputs017;
	Cyclic#1.CAM7.Profinet_QRkod_Znaky[17] AT %IB."KAM_ControlUNit".Module011_Inputs018;
	Cyclic#1.CAM7.Profinet_QRkod_Znaky[18] AT %IB."KAM_ControlUNit".Module011_Inputs019;
	Cyclic#1.CAM7.Profinet_QRkod_Znaky[19] AT %IB."KAM_ControlUNit".Module011_Inputs020;
	Cyclic#1.CAM7.Profinet_QRkod_Znaky[20] AT %IB."KAM_ControlUNit".Module011_Inputs021;
	Cyclic#1.CAM7.Profinet_QRkod_Znaky[21] AT %IB."KAM_ControlUNit".Module011_Inputs022;
	Cyclic#1.CAM7.Profinet_QRkod_Znaky[22] AT %IB."KAM_ControlUNit".Module011_Inputs023;
	Cyclic#1.CAM7.Profinet_QRkod_Znaky[23] AT %IB."KAM_ControlUNit".Module011_Inputs024;
	Cyclic#1.CAM7.Profinet_QRkod_Znaky[24] AT %IB."KAM_ControlUNit".Module011_Inputs025;
	Cyclic#1.CAM7.Profinet_QRkod_Znaky[25] AT %IB."KAM_ControlUNit".Module011_Inputs026;
	Cyclic#1.CAM7.Profinet_QRkod_Znaky[26] AT %IB."KAM_ControlUNit".Module011_Inputs027;
	Cyclic#1.CAM7.Profinet_QRkod_Znaky[27] AT %IB."KAM_ControlUNit".Module011_Inputs028;
	Cyclic#1.CAM7.Profinet_QRkod_Znaky[28] AT %IB."KAM_ControlUNit".Module011_Inputs029;
	Cyclic#1.CAM7.Profinet_QRkod_Znaky[29] AT %IB."KAM_ControlUNit".Module011_Inputs030;
	Cyclic#1.CAM7.Profinet_QRkod_Znaky[30] AT %IB."KAM_ControlUNit".Module011_Inputs031;
	Cyclic#1.CAM7.Profinet_QRkod_Znaky[31] AT %IB."KAM_ControlUNit".Module011_Inputs032;
	Cyclic#1.CAM10.Profinet_PLC_INPUTS[0] AT %IB."KAM_ControlUNit".Module015_Inputs001;
	Cyclic#1.CAM10.Profinet_PLC_INPUTS[1] AT %IB."KAM_ControlUNit".Module015_Inputs002;
	Cyclic#1.CAM10.Profinet_PLC_INPUTS[2] AT %IB."KAM_ControlUNit".Module015_Inputs003;
	Cyclic#1.CAM10.Profinet_PLC_INPUTS[3] AT %IB."KAM_ControlUNit".Module015_Inputs004;
	Cyclic#1.CAM11.Profinet_PLC_INPUTS[0] AT %IB."KAM_ControlUNit".Module017_Inputs001;
	Cyclic#1.CAM11.Profinet_PLC_INPUTS[1] AT %IB."KAM_ControlUNit".Module017_Inputs002;
	Cyclic#1.CAM11.Profinet_PLC_INPUTS[2] AT %IB."KAM_ControlUNit".Module017_Inputs003;
	Cyclic#1.CAM11.Profinet_PLC_INPUTS[3] AT %IB."KAM_ControlUNit".Module017_Inputs004;
	Cyclic#1.CAM12.Profinet_PLC_INPUTS[0] AT %IB."KAM_ControlUNit".Module019_Inputs001;
	Cyclic#1.CAM12.Profinet_PLC_INPUTS[1] AT %IB."KAM_ControlUNit".Module019_Inputs002;
	Cyclic#1.CAM12.Profinet_PLC_INPUTS[2] AT %IB."KAM_ControlUNit".Module019_Inputs003;
	Cyclic#1.CAM12.Profinet_PLC_INPUTS[3] AT %IB."KAM_ControlUNit".Module019_Inputs004;
	Cyclic#1.CAM13.Profinet_PLC_INPUTS[0] AT %IB."KAM_ControlUNit".Module021_Inputs001;
	Cyclic#1.CAM13.Profinet_PLC_INPUTS[1] AT %IB."KAM_ControlUNit".Module021_Inputs002;
	Cyclic#1.CAM13.Profinet_PLC_INPUTS[2] AT %IB."KAM_ControlUNit".Module021_Inputs003;
	Cyclic#1.CAM13.Profinet_PLC_INPUTS[3] AT %IB."KAM_ControlUNit".Module021_Inputs004;
	Cyclic#1.CAM15.Profinet_PLC_INPUTS[0] AT %IB."KAM_ControlUNit".Module023_Inputs001;
	Cyclic#1.CAM15.Profinet_PLC_INPUTS[1] AT %IB."KAM_ControlUNit".Module023_Inputs002;
	Cyclic#1.CAM15.Profinet_PLC_INPUTS[2] AT %IB."KAM_ControlUNit".Module023_Inputs003;
	Cyclic#1.CAM15.Profinet_PLC_INPUTS[3] AT %IB."KAM_ControlUNit".Module023_Inputs004;
	Cyclic#1.CAM16.Profinet_PLC_INPUTS[0] AT %IB."KAM_ControlUNit".Module025_Inputs001;
	Cyclic#1.CAM16.Profinet_PLC_INPUTS[1] AT %IB."KAM_ControlUNit".Module025_Inputs002;
	Cyclic#1.CAM16.Profinet_PLC_INPUTS[2] AT %IB."KAM_ControlUNit".Module025_Inputs003;
	Cyclic#1.CAM16.Profinet_PLC_INPUTS[3] AT %IB."KAM_ControlUNit".Module025_Inputs004;
	Cyclic#1.CAM14.Profinet_PLC_INPUTS[4] AT %IB."P4_KAM14".Module006_Input_16_Byte004;
	Cyclic#1.CAM15.Profinet_QRkod_Znaky[0] AT %IB."KAM_ControlUNit".Module023_Inputs033;
	Cyclic#1.CAM15.Profinet_QRkod_Znaky[1] AT %IB."KAM_ControlUNit".Module023_Inputs034;
	Cyclic#1.CAM15.Profinet_QRkod_Znaky[2] AT %IB."KAM_ControlUNit".Module023_Inputs035;
	Cyclic#1.CAM15.Profinet_QRkod_Znaky[3] AT %IB."KAM_ControlUNit".Module023_Inputs036;
	Cyclic#1.CAM15.Profinet_QRkod_Znaky[4] AT %IB."KAM_ControlUNit".Module023_Inputs037;
	Cyclic#1.CAM15.Profinet_QRkod_Znaky[5] AT %IB."KAM_ControlUNit".Module023_Inputs038;
	Cyclic#1.CAM15.Profinet_QRkod_Znaky[6] AT %IB."KAM_ControlUNit".Module023_Inputs039;
	Cyclic#1.CAM15.Profinet_QRkod_Znaky[7] AT %IB."KAM_ControlUNit".Module023_Inputs040;
	Cyclic#1.CAM15.Profinet_QRkod_Znaky[8] AT %IB."KAM_ControlUNit".Module023_Inputs041;
	Cyclic#1.CAM15.Profinet_QRkod_Znaky[9] AT %IB."KAM_ControlUNit".Module023_Inputs042;
	Cyclic#1.CAM15.Profinet_QRkod_Znaky[10] AT %IB."KAM_ControlUNit".Module023_Inputs043;
	Cyclic#1.CAM15.Profinet_QRkod_Znaky[11] AT %IB."KAM_ControlUNit".Module023_Inputs044;
	Cyclic#1.CAM15.Profinet_QRkod_Znaky[12] AT %IB."KAM_ControlUNit".Module023_Inputs045;
	Cyclic#1.CAM15.Profinet_QRkod_Znaky[13] AT %IB."KAM_ControlUNit".Module023_Inputs046;
	Cyclic#1.CAM15.Profinet_QRkod_Znaky[14] AT %IB."KAM_ControlUNit".Module023_Inputs047;
	Cyclic#1.CAM15.Profinet_QRkod_Znaky[15] AT %IB."KAM_ControlUNit".Module023_Inputs048;
	Cyclic#1.CAM15.Profinet_QRkod_Znaky[16] AT %IB."KAM_ControlUNit".Module023_Inputs049;
	Cyclic#1.CAM15.Profinet_QRkod_Znaky[17] AT %IB."KAM_ControlUNit".Module023_Inputs050;
	Cyclic#1.CAM15.Profinet_QRkod_Znaky[18] AT %IB."KAM_ControlUNit".Module023_Inputs051;
	Cyclic#1.CAM15.Profinet_QRkod_Znaky[19] AT %IB."KAM_ControlUNit".Module023_Inputs052;
	Cyclic#1.CAM15.Profinet_QRkod_Znaky[20] AT %IB."KAM_ControlUNit".Module023_Inputs053;
	Cyclic#1.CAM15.Profinet_QRkod_Znaky[21] AT %IB."KAM_ControlUNit".Module023_Inputs054;
	Cyclic#1.CAM15.Profinet_QRkod_Znaky[22] AT %IB."KAM_ControlUNit".Module023_Inputs055;
	Cyclic#1.CAM15.Profinet_QRkod_Znaky[23] AT %IB."KAM_ControlUNit".Module023_Inputs056;
	Cyclic#1.CAM15.Profinet_QRkod_Znaky[24] AT %IB."KAM_ControlUNit".Module023_Inputs057;
	Cyclic#1.CAM15.Profinet_QRkod_Znaky[25] AT %IB."KAM_ControlUNit".Module023_Inputs058;
	Cyclic#1.CAM15.Profinet_QRkod_Znaky[26] AT %IB."KAM_ControlUNit".Module023_Inputs059;
	Cyclic#1.CAM15.Profinet_QRkod_Znaky[27] AT %IB."KAM_ControlUNit".Module023_Inputs060;
	Cyclic#1.CAM15.Profinet_QRkod_Znaky[28] AT %IB."KAM_ControlUNit".Module023_Inputs061;
	Cyclic#1.CAM15.Profinet_QRkod_Znaky[29] AT %IB."KAM_ControlUNit".Module023_Inputs062;
	Cyclic#1.CAM15.Profinet_QRkod_Znaky[30] AT %IB."KAM_ControlUNit".Module023_Inputs063;
	Cyclic#1.CAM15.Profinet_QRkod_Znaky[31] AT %IB."KAM_ControlUNit".Module023_Inputs064;
	Cyclic#1.CAM15.Profinet_OCR_Znaky[0] AT %IB."KAM_ControlUNit".Module024_Inputs001;
	Cyclic#1.CAM15.Profinet_OCR_Znaky[1] AT %IB."KAM_ControlUNit".Module024_Inputs002;
	Cyclic#1.CAM15.Profinet_OCR_Znaky[2] AT %IB."KAM_ControlUNit".Module024_Inputs003;
	Cyclic#1.CAM15.Profinet_OCR_Znaky[3] AT %IB."KAM_ControlUNit".Module024_Inputs004;
	Cyclic#1.CAM15.Profinet_OCR_Znaky[4] AT %IB."KAM_ControlUNit".Module024_Inputs005;
	Cyclic#1.CAM15.Profinet_OCR_Znaky[5] AT %IB."KAM_ControlUNit".Module024_Inputs006;
	Cyclic#1.CAM15.Profinet_OCR_Znaky[6] AT %IB."KAM_ControlUNit".Module024_Inputs007;
	Cyclic#1.CAM15.Profinet_OCR_Znaky[7] AT %IB."KAM_ControlUNit".Module024_Inputs008;
	Cyclic#1.CAM15.Profinet_OCR_Znaky[8] AT %IB."KAM_ControlUNit".Module024_Inputs009;
	Cyclic#1.CAM15.Profinet_OCR_Znaky[9] AT %IB."KAM_ControlUNit".Module024_Inputs010;
	Cyclic#1.CAM15.Profinet_OCR_Znaky[10] AT %IB."KAM_ControlUNit".Module024_Inputs011;
	Cyclic#1.CAM15.Profinet_OCR_Znaky[11] AT %IB."KAM_ControlUNit".Module024_Inputs012;
	Cyclic#1.CAM15.Profinet_OCR_Znaky[12] AT %IB."KAM_ControlUNit".Module024_Inputs013;
	Cyclic#1.CAM15.Profinet_OCR_Znaky[13] AT %IB."KAM_ControlUNit".Module024_Inputs014;
	Cyclic#1.CAM15.Profinet_OCR_Znaky[14] AT %IB."KAM_ControlUNit".Module024_Inputs015;
	Cyclic#1.CAM15.Profinet_OCR_Znaky[15] AT %IB."KAM_ControlUNit".Module024_Inputs016;
	Cyclic#1.CAM15.Profinet_OCR_Znaky[16] AT %IB."KAM_ControlUNit".Module024_Inputs017;
	Cyclic#1.CAM15.Profinet_OCR_Znaky[17] AT %IB."KAM_ControlUNit".Module024_Inputs018;
	Cyclic#1.CAM15.Profinet_OCR_Znaky[18] AT %IB."KAM_ControlUNit".Module024_Inputs019;
	Cyclic#1.CAM15.Profinet_OCR_Znaky[19] AT %IB."KAM_ControlUNit".Module024_Inputs020;
	Cyclic#1.CAM15.Profinet_OCR_Znaky[20] AT %IB."KAM_ControlUNit".Module024_Inputs021;
	Cyclic#1.CAM15.Profinet_OCR_Znaky[21] AT %IB."KAM_ControlUNit".Module024_Inputs022;
	Cyclic#1.CAM15.Profinet_OCR_Znaky[22] AT %IB."KAM_ControlUNit".Module024_Inputs023;
	Cyclic#1.CAM15.Profinet_OCR_Znaky[23] AT %IB."KAM_ControlUNit".Module024_Inputs024;
	Cyclic#1.CAM15.Profinet_OCR_Znaky[24] AT %IB."KAM_ControlUNit".Module024_Inputs025;
	Cyclic#1.CAM15.Profinet_OCR_Znaky[25] AT %IB."KAM_ControlUNit".Module024_Inputs026;
	Cyclic#1.CAM15.Profinet_OCR_Znaky[26] AT %IB."KAM_ControlUNit".Module024_Inputs027;
	Cyclic#1.CAM15.Profinet_OCR_Znaky[27] AT %IB."KAM_ControlUNit".Module024_Inputs028;
	Cyclic#1.CAM15.Profinet_OCR_Znaky[28] AT %IB."KAM_ControlUNit".Module024_Inputs029;
	Cyclic#1.CAM15.Profinet_OCR_Znaky[29] AT %IB."KAM_ControlUNit".Module024_Inputs030;
	Cyclic#1.CAM15.Profinet_OCR_Znaky[30] AT %IB."KAM_ControlUNit".Module024_Inputs031;
	Cyclic#1.CAM15.Profinet_OCR_Znaky[31] AT %IB."KAM_ControlUNit".Module024_Inputs032;
	Cyclic#1.P3_LeakageTestA.IN.Tester_TypKonektoru_5F_5H AT %IX."DI3.2_16DI".DigitalInput13;
	Cyclic#1.P3_LeakageTestA.IN.Tester_TypKonektoru_4F AT %IX."DI3.2_16DI".DigitalInput14;
	Cyclic#1.P3_LeakageTestB.IN.Tester_TypKonektoru_5F_5H AT %IX."DI3.2_16DI".DigitalInput15;
	Cyclic#1.P3_LeakageTestB.IN.Tester_TypKonektoru_4F AT %IX."DI3.2_16DI".DigitalInput16;
	Cyclic#1.P3_Srobovanie.IN.HVTest_TypKonektoru_5F_5H AT %IX."DI3.1_16DI".DigitalInput07;
	Cyclic#1.P3_Srobovanie.IN.HVTest_TypKonektoru_4F AT %IX."DI3.1_16DI".DigitalInput08;
	Cyclic#1.P1_Srobovanie.PAR.M5_AtlasCopcoInputs[2] AT %ID."RJ6_P1_Srobovacka_M5".Module002_Input_I_00;
	Cyclic#1.P1_Srobovanie.PAR.M5_AtlasCopcoInputs[3] AT %ID."RJ6_P1_Srobovacka_M5".Module002_Input_I_01;
	Cyclic#1.P1_Srobovanie.PAR.M5_AllasCopcoOutputs[0] AT %QD."RJ6_P1_Srobovacka_M5".Module003_Output_O_00;
	Cyclic#1.P1_Srobovanie.PAR.M5_AllasCopcoOutputs[1] AT %QD."RJ6_P1_Srobovacka_M5".Module003_Output_O_01;
	Cyclic#1.P1_Srobovanie.PAR.M5_AllasCopcoOutputs[2] AT %QD."RJ6_P1_Srobovacka_M5".Module004_Output_O_00;
	Cyclic#1.P1_Srobovanie.PAR.M5_AllasCopcoOutputs[3] AT %QD."RJ6_P1_Srobovacka_M5".Module004_Output_O_01;
	Cyclic#1.Safety.OUT.P2_ZamkniZamok_ZadneDvereLS AT %QX."DM2.1_16DI/DO".DigitalOutput05;
	Cyclic#1.Safety.OUT.P2_ZamkniZamok_ZadneDverePS AT %QX."DM2.1_16DI/DO".DigitalOutput07;
	Cyclic#1.Safety.IN.P2_ZadneDvereLS_PritomPetlice AT %IX."DM2.1_16DI/DO".DigitalInput06;
	Cyclic#1.Safety.IN.P2_ZadneDverePS_PritomPetlice AT %IX."DM2.1_16DI/DO".DigitalInput08;
	Cyclic#1.P1_Srobovanie.PAR.K30_AtlasCopcoInputs[2] AT %ID."RJ5_P1_Srobovacka_K30".Module002_Input_I_00;
	Cyclic#1.P1_Srobovanie.PAR.K30_AtlasCopcoInputs[3] AT %ID."RJ5_P1_Srobovacka_K30".Module002_Input_I_01;
	Cyclic#1.P1_Srobovanie.PAR.K30_AllasCopcoOutputs[0] AT %QD."RJ5_P1_Srobovacka_K30".Module003_Output_O_00;
	Cyclic#1.P1_Srobovanie.PAR.K30_AllasCopcoOutputs[1] AT %QD."RJ5_P1_Srobovacka_K30".Module003_Output_O_01;
	Cyclic#1.P1_Srobovanie.PAR.K30_AllasCopcoOutputs[2] AT %QD."RJ5_P1_Srobovacka_K30".Module004_Output_O_00;
	Cyclic#1.P1_Srobovanie.PAR.K30_AllasCopcoOutputs[3] AT %QD."RJ5_P1_Srobovacka_K30".Module004_Output_O_01;
	Cyclic#1.P1_Srobovanie.PAR.K30_AllasCopcoOutputs[0] AT %QD."RJ5_P1_Srobovacka_K30".Module005_Output_O_00;
	Cyclic#1.P1_Srobovanie.PAR.K30_AllasCopcoOutputs[1] AT %QD."RJ5_P1_Srobovacka_K30".Module005_Output_O_01;
	Cyclic#1.P1_Srobovanie.PAR.K30_AllasCopcoOutputs[2] AT %QD."RJ5_P1_Srobovacka_K30".Module006_Output_O_00;
	Cyclic#1.P1_Srobovanie.PAR.K30_AllasCopcoOutputs[3] AT %QD."RJ5_P1_Srobovacka_K30".Module006_Output_O_01;
	Cyclic#1.P1_Srobovanie.PAR.M5_AllasCopcoOutputs[0] AT %QD."RJ6_P1_Srobovacka_M5".Module005_Output_O_00;
	Cyclic#1.P1_Srobovanie.PAR.M5_AllasCopcoOutputs[1] AT %QD."RJ6_P1_Srobovacka_M5".Module005_Output_O_01;
	Cyclic#1.P1_Srobovanie.PAR.M5_AllasCopcoOutputs[2] AT %QD."RJ6_P1_Srobovacka_M5".Module006_Output_O_00;
	Cyclic#1.P1_Srobovanie.PAR.M5_AllasCopcoOutputs[3] AT %QD."RJ6_P1_Srobovacka_M5".Module006_Output_O_01;
	Cyclic#1.P1_Srobovanie.PAR.M4_AtlasCopcoInputs[2] AT %ID."RJ7_P1_Srobovacka_M4".Module002_Input_I_00;
	Cyclic#1.P1_Srobovanie.PAR.M4_AtlasCopcoInputs[3] AT %ID."RJ7_P1_Srobovacka_M4".Module002_Input_I_01;
	Cyclic#1.P1_Srobovanie.PAR.M4_AllasCopcoOutputs[0] AT %QD."RJ7_P1_Srobovacka_M4".Module005_Output_O_00;
	Cyclic#1.P1_Srobovanie.PAR.M4_AllasCopcoOutputs[1] AT %QD."RJ7_P1_Srobovacka_M4".Module005_Output_O_01;
	Cyclic#1.P1_Srobovanie.PAR.M4_AllasCopcoOutputs[2] AT %QD."RJ7_P1_Srobovacka_M4".Module006_Output_O_00;
	Cyclic#1.P1_Srobovanie.PAR.M4_AllasCopcoOutputs[3] AT %QD."RJ7_P1_Srobovacka_M4".Module006_Output_O_01;
	Cyclic#1.P2_Srobovanie.PAR.M6_AtlasCopcoInputs[2] AT %ID."RJ2_P2_Srobovacka_M6".Module002_Input_I_00;
	Cyclic#1.P2_Srobovanie.PAR.M6_AtlasCopcoInputs[3] AT %ID."RJ2_P2_Srobovacka_M6".Module002_Input_I_01;
	Cyclic#1.P2_Srobovanie.PAR.M6_AllasCopcoOutputs[0] AT %QD."RJ2_P2_Srobovacka_M6".Module005_Output_O_00;
	Cyclic#1.P2_Srobovanie.PAR.M6_AllasCopcoOutputs[1] AT %QD."RJ2_P2_Srobovacka_M6".Module005_Output_O_01;
	Cyclic#1.P2_Srobovanie.PAR.M6_AllasCopcoOutputs[2] AT %QD."RJ2_P2_Srobovacka_M6".Module006_Output_O_00;
	Cyclic#1.P2_Srobovanie.PAR.M6_AllasCopcoOutputs[3] AT %QD."RJ2_P2_Srobovacka_M6".Module006_Output_O_01;
	Cyclic#1.P2_Srobovanie.PAR.M5_AtlasCopcoInputs[2] AT %ID."RJ4_P2_Srobovacka_M5".Module002_Input_I_00;
	Cyclic#1.P2_Srobovanie.PAR.M5_AtlasCopcoInputs[3] AT %ID."RJ4_P2_Srobovacka_M5".Module002_Input_I_01;
	Cyclic#1.P2_Srobovanie.PAR.M5_AllasCopcoOutputs[0] AT %QD."RJ4_P2_Srobovacka_M5".Module005_Output_O_00;
	Cyclic#1.P2_Srobovanie.PAR.M5_AllasCopcoOutputs[1] AT %QD."RJ4_P2_Srobovacka_M5".Module005_Output_O_01;
	Cyclic#1.P2_Srobovanie.PAR.M5_AllasCopcoOutputs[2] AT %QD."RJ4_P2_Srobovacka_M5".Module006_Output_O_00;
	Cyclic#1.P2_Srobovanie.PAR.M5_AllasCopcoOutputs[3] AT %QD."RJ4_P2_Srobovacka_M5".Module006_Output_O_01;
	Cyclic#1.P2_Srobovanie.PAR.M4_AtlasCopcoInputs[2] AT %ID."RJ3_P2_Srobovacka_M4".Module002_Input_I_00;
	Cyclic#1.P2_Srobovanie.PAR.M4_AtlasCopcoInputs[3] AT %ID."RJ3_P2_Srobovacka_M4".Module002_Input_I_01;
	Cyclic#1.P2_Srobovanie.PAR.M4_AllasCopcoOutputs[0] AT %QD."RJ3_P2_Srobovacka_M4".Module005_Output_O_00;
	Cyclic#1.P2_Srobovanie.PAR.M4_AllasCopcoOutputs[1] AT %QD."RJ3_P2_Srobovacka_M4".Module005_Output_O_01;
	Cyclic#1.P2_Srobovanie.PAR.M4_AllasCopcoOutputs[2] AT %QD."RJ3_P2_Srobovacka_M4".Module006_Output_O_00;
	Cyclic#1.P2_Srobovanie.PAR.M4_AllasCopcoOutputs[3] AT %QD."RJ3_P2_Srobovacka_M4".Module006_Output_O_01;
	Cyclic#1.P2_SkrutkovacMatic.PAR.MaticeM4_AtlasCopcoInputs[2] AT %ID."RJ1_P2_SrobovackaMatic_M4".Module002_Input_I_00;
	Cyclic#1.P2_SkrutkovacMatic.PAR.MaticeM4_AtlasCopcoInputs[3] AT %ID."RJ1_P2_SrobovackaMatic_M4".Module002_Input_I_01;
	Cyclic#1.P2_SkrutkovacMatic.PAR.MaticeM4_AtlasCopcoOutputs[0] AT %QD."RJ1_P2_SrobovackaMatic_M4".Module005_Output_O_00;
	Cyclic#1.P2_SkrutkovacMatic.PAR.MaticeM4_AtlasCopcoOutputs[1] AT %QD."RJ1_P2_SrobovackaMatic_M4".Module005_Output_O_01;
	Cyclic#1.P2_SkrutkovacMatic.PAR.MaticeM4_AtlasCopcoOutputs[2] AT %QD."RJ1_P2_SrobovackaMatic_M4".Module006_Output_O_00;
	Cyclic#1.P2_SkrutkovacMatic.PAR.MaticeM4_AtlasCopcoOutputs[3] AT %QD."RJ1_P2_SrobovackaMatic_M4".Module006_Output_O_01;
	Cyclic#1.P3_Srobovanie.PAR.K40_AtlasCopcoInputs[2] AT %ID."P3_Srobovacka_K40".Module002_Input_I_00;
	Cyclic#1.P3_Srobovanie.PAR.K40_AtlasCopcoInputs[3] AT %ID."P3_Srobovacka_K40".Module002_Input_I_01;
	Cyclic#1.P3_Srobovanie.PAR.K40_AllasCopcoOutputs[0] AT %QD."P3_Srobovacka_K40".Module005_Output_O_00;
	Cyclic#1.P3_Srobovanie.PAR.K40_AllasCopcoOutputs[1] AT %QD."P3_Srobovacka_K40".Module005_Output_O_01;
	Cyclic#1.P3_Srobovanie.PAR.K40_AllasCopcoOutputs[2] AT %QD."P3_Srobovacka_K40".Module006_Output_O_00;
	Cyclic#1.P3_Srobovanie.PAR.K40_AllasCopcoOutputs[3] AT %QD."P3_Srobovacka_K40".Module006_Output_O_01;
	Cyclic#1.P3_Srobovanie.PAR.M5_AtlasCopcoInputs[2] AT %ID."P3_Srobovacka_M5".Module002_Input_I_00;
	Cyclic#1.P3_Srobovanie.PAR.M5_AtlasCopcoInputs[3] AT %ID."P3_Srobovacka_M5".Module002_Input_I_01;
	Cyclic#1.P3_Srobovanie.PAR.M5_AllasCopcoOutputs[0] AT %QD."P3_Srobovacka_M5".Module005_Output_O_00;
	Cyclic#1.P3_Srobovanie.PAR.M5_AllasCopcoOutputs[1] AT %QD."P3_Srobovacka_M5".Module005_Output_O_01;
	Cyclic#1.P3_Srobovanie.PAR.M5_AllasCopcoOutputs[2] AT %QD."P3_Srobovacka_M5".Module006_Output_O_00;
	Cyclic#1.P3_Srobovanie.PAR.M5_AllasCopcoOutputs[3] AT %QD."P3_Srobovacka_M5".Module006_Output_O_01;
	Cyclic#1.P1_Srobovanie.PAR.K30_AtlasCopcoInputs[4] AT %ID."RJ5_P1_Srobovacka_K30".Module003_Input_I_00;
	Cyclic#1.P1_Srobovanie.PAR.K30_AtlasCopcoInputs[5] AT %ID."RJ5_P1_Srobovacka_K30".Module003_Input_I_01;
	Cyclic#1.P1_Srobovanie.PAR.K30_AllasCopcoOutputs[4] AT %QD."RJ5_P1_Srobovacka_K30".Module007_Output_O_00;
	Cyclic#1.P1_Srobovanie.PAR.K30_AllasCopcoOutputs[5] AT %QD."RJ5_P1_Srobovacka_K30".Module007_Output_O_01;
	Cyclic#1.P1_Srobovanie.PAR.K30_AtlasCopcoInputs[6] AT %ID."RJ5_P1_Srobovacka_K30".Module004_Input_I_00;
	Cyclic#1.P1_Srobovanie.PAR.K30_AtlasCopcoInputs[7] AT %ID."RJ5_P1_Srobovacka_K30".Module004_Input_I_01;
	Cyclic#1.P1_Srobovanie.PAR.K30_AllasCopcoOutputs[6] AT %QD."RJ5_P1_Srobovacka_K30".Module008_Output_O_00;
	Cyclic#1.P1_Srobovanie.PAR.K30_AllasCopcoOutputs[7] AT %QD."RJ5_P1_Srobovacka_K30".Module008_Output_O_01;
	Cyclic#1.P1_Srobovanie.PAR.M5_AtlasCopcoInputs[4] AT %ID."RJ6_P1_Srobovacka_M5".Module003_Input_I_00;
	Cyclic#1.P1_Srobovanie.PAR.M5_AtlasCopcoInputs[5] AT %ID."RJ6_P1_Srobovacka_M5".Module003_Input_I_01;
	Cyclic#1.P1_Srobovanie.PAR.M5_AtlasCopcoInputs[6] AT %ID."RJ6_P1_Srobovacka_M5".Module004_Input_I_00;
	Cyclic#1.P1_Srobovanie.PAR.M5_AtlasCopcoInputs[7] AT %ID."RJ6_P1_Srobovacka_M5".Module004_Input_I_01;
	Cyclic#1.P1_Srobovanie.PAR.M5_AllasCopcoOutputs[4] AT %QD."RJ6_P1_Srobovacka_M5".Module007_Output_O_00;
	Cyclic#1.P1_Srobovanie.PAR.M5_AllasCopcoOutputs[5] AT %QD."RJ6_P1_Srobovacka_M5".Module007_Output_O_01;
	Cyclic#1.P1_Srobovanie.PAR.M5_AllasCopcoOutputs[6] AT %QD."RJ6_P1_Srobovacka_M5".Module008_Output_O_00;
	Cyclic#1.P1_Srobovanie.PAR.M5_AllasCopcoOutputs[7] AT %QD."RJ6_P1_Srobovacka_M5".Module008_Output_O_01;
	Cyclic#1.P1_Srobovanie.PAR.M4_AtlasCopcoInputs[4] AT %ID."RJ7_P1_Srobovacka_M4".Module003_Input_I_00;
	Cyclic#1.P1_Srobovanie.PAR.M4_AtlasCopcoInputs[5] AT %ID."RJ7_P1_Srobovacka_M4".Module003_Input_I_01;
	Cyclic#1.P1_Srobovanie.PAR.M4_AtlasCopcoInputs[6] AT %ID."RJ7_P1_Srobovacka_M4".Module004_Input_I_00;
	Cyclic#1.P1_Srobovanie.PAR.M4_AtlasCopcoInputs[7] AT %ID."RJ7_P1_Srobovacka_M4".Module004_Input_I_01;
	Cyclic#1.P1_Srobovanie.PAR.M4_AllasCopcoOutputs[4] AT %QD."RJ7_P1_Srobovacka_M4".Module007_Output_O_00;
	Cyclic#1.P1_Srobovanie.PAR.M4_AllasCopcoOutputs[5] AT %QD."RJ7_P1_Srobovacka_M4".Module007_Output_O_01;
	Cyclic#1.P1_Srobovanie.PAR.M4_AllasCopcoOutputs[6] AT %QD."RJ7_P1_Srobovacka_M4".Module008_Output_O_00;
	Cyclic#1.P1_Srobovanie.PAR.M4_AllasCopcoOutputs[7] AT %QD."RJ7_P1_Srobovacka_M4".Module008_Output_O_01;
	Cyclic#1.P2_Srobovanie.PAR.M6_AtlasCopcoInputs[4] AT %ID."RJ2_P2_Srobovacka_M6".Module003_Input_I_00;
	Cyclic#1.P2_Srobovanie.PAR.M6_AtlasCopcoInputs[5] AT %ID."RJ2_P2_Srobovacka_M6".Module003_Input_I_01;
	Cyclic#1.P2_Srobovanie.PAR.M6_AtlasCopcoInputs[6] AT %ID."RJ2_P2_Srobovacka_M6".Module004_Input_I_00;
	Cyclic#1.P2_Srobovanie.PAR.M6_AtlasCopcoInputs[7] AT %ID."RJ2_P2_Srobovacka_M6".Module004_Input_I_01;
	Cyclic#1.P2_Srobovanie.PAR.M6_AllasCopcoOutputs[4] AT %QD."RJ2_P2_Srobovacka_M6".Module007_Output_O_00;
	Cyclic#1.P2_Srobovanie.PAR.M6_AllasCopcoOutputs[5] AT %QD."RJ2_P2_Srobovacka_M6".Module007_Output_O_01;
	Cyclic#1.P2_Srobovanie.PAR.M6_AllasCopcoOutputs[6] AT %QD."RJ2_P2_Srobovacka_M6".Module008_Output_O_00;
	Cyclic#1.P2_Srobovanie.PAR.M6_AllasCopcoOutputs[7] AT %QD."RJ2_P2_Srobovacka_M6".Module008_Output_O_01;
	Cyclic#1.P2_Srobovanie.PAR.M5_AtlasCopcoInputs[4] AT %ID."RJ4_P2_Srobovacka_M5".Module003_Input_I_00;
	Cyclic#1.P2_Srobovanie.PAR.M5_AtlasCopcoInputs[5] AT %ID."RJ4_P2_Srobovacka_M5".Module003_Input_I_01;
	Cyclic#1.P2_Srobovanie.PAR.M5_AtlasCopcoInputs[6] AT %ID."RJ4_P2_Srobovacka_M5".Module004_Input_I_00;
	Cyclic#1.P2_Srobovanie.PAR.M5_AtlasCopcoInputs[7] AT %ID."RJ4_P2_Srobovacka_M5".Module004_Input_I_01;
	Cyclic#1.P2_Srobovanie.PAR.M5_AllasCopcoOutputs[4] AT %QD."RJ4_P2_Srobovacka_M5".Module007_Output_O_00;
	Cyclic#1.P2_Srobovanie.PAR.M5_AllasCopcoOutputs[5] AT %QD."RJ4_P2_Srobovacka_M5".Module007_Output_O_01;
	Cyclic#1.P2_Srobovanie.PAR.M5_AllasCopcoOutputs[6] AT %QD."RJ4_P2_Srobovacka_M5".Module008_Output_O_00;
	Cyclic#1.P2_Srobovanie.PAR.M5_AllasCopcoOutputs[7] AT %QD."RJ4_P2_Srobovacka_M5".Module008_Output_O_01;
	Cyclic#1.P2_Srobovanie.PAR.M4_AtlasCopcoInputs[4] AT %ID."RJ3_P2_Srobovacka_M4".Module003_Input_I_00;
	Cyclic#1.P2_Srobovanie.PAR.M4_AtlasCopcoInputs[5] AT %ID."RJ3_P2_Srobovacka_M4".Module003_Input_I_01;
	Cyclic#1.P2_Srobovanie.PAR.M4_AtlasCopcoInputs[6] AT %ID."RJ3_P2_Srobovacka_M4".Module004_Input_I_00;
	Cyclic#1.P2_Srobovanie.PAR.M4_AtlasCopcoInputs[7] AT %ID."RJ3_P2_Srobovacka_M4".Module004_Input_I_01;
	Cyclic#1.P2_Srobovanie.PAR.M4_AllasCopcoOutputs[4] AT %QD."RJ3_P2_Srobovacka_M4".Module007_Output_O_00;
	Cyclic#1.P2_Srobovanie.PAR.M4_AllasCopcoOutputs[5] AT %QD."RJ3_P2_Srobovacka_M4".Module007_Output_O_01;
	Cyclic#1.P2_Srobovanie.PAR.M4_AllasCopcoOutputs[6] AT %QD."RJ3_P2_Srobovacka_M4".Module008_Output_O_00;
	Cyclic#1.P2_Srobovanie.PAR.M4_AllasCopcoOutputs[7] AT %QD."RJ3_P2_Srobovacka_M4".Module008_Output_O_01;
	Cyclic#1.P2_SkrutkovacMatic.PAR.MaticeM4_AtlasCopcoInputs[4] AT %ID."RJ1_P2_SrobovackaMatic_M4".Module003_Input_I_00;
	Cyclic#1.P2_SkrutkovacMatic.PAR.MaticeM4_AtlasCopcoInputs[5] AT %ID."RJ1_P2_SrobovackaMatic_M4".Module003_Input_I_01;
	Cyclic#1.P2_SkrutkovacMatic.PAR.MaticeM4_AtlasCopcoInputs[6] AT %ID."RJ1_P2_SrobovackaMatic_M4".Module004_Input_I_00;
	Cyclic#1.P2_SkrutkovacMatic.PAR.MaticeM4_AtlasCopcoInputs[7] AT %ID."RJ1_P2_SrobovackaMatic_M4".Module004_Input_I_01;
	Cyclic#1.P2_SkrutkovacMatic.PAR.MaticeM4_AtlasCopcoOutputs[4] AT %QD."RJ1_P2_SrobovackaMatic_M4".Module007_Output_O_00;
	Cyclic#1.P2_SkrutkovacMatic.PAR.MaticeM4_AtlasCopcoOutputs[5] AT %QD."RJ1_P2_SrobovackaMatic_M4".Module007_Output_O_01;
	Cyclic#1.P2_SkrutkovacMatic.PAR.MaticeM4_AtlasCopcoOutputs[6] AT %QD."RJ1_P2_SrobovackaMatic_M4".Module008_Output_O_00;
	Cyclic#1.P2_SkrutkovacMatic.PAR.MaticeM4_AtlasCopcoOutputs[7] AT %QD."RJ1_P2_SrobovackaMatic_M4".Module008_Output_O_01;
	Cyclic#1.P3_Srobovanie.PAR.K40_AtlasCopcoInputs[4] AT %ID."P3_Srobovacka_K40".Module003_Input_I_00;
	Cyclic#1.P3_Srobovanie.PAR.K40_AtlasCopcoInputs[5] AT %ID."P3_Srobovacka_K40".Module003_Input_I_01;
	Cyclic#1.P3_Srobovanie.PAR.K40_AtlasCopcoInputs[6] AT %ID."P3_Srobovacka_K40".Module004_Input_I_00;
	Cyclic#1.P3_Srobovanie.PAR.K40_AtlasCopcoInputs[7] AT %ID."P3_Srobovacka_K40".Module004_Input_I_01;
	Cyclic#1.P3_Srobovanie.PAR.K40_AllasCopcoOutputs[4] AT %QD."P3_Srobovacka_K40".Module007_Output_O_00;
	Cyclic#1.P3_Srobovanie.PAR.K40_AllasCopcoOutputs[5] AT %QD."P3_Srobovacka_K40".Module007_Output_O_01;
	Cyclic#1.P3_Srobovanie.PAR.K40_AllasCopcoOutputs[6] AT %QD."P3_Srobovacka_K40".Module008_Output_O_00;
	Cyclic#1.P3_Srobovanie.PAR.K40_AllasCopcoOutputs[7] AT %QD."P3_Srobovacka_K40".Module008_Output_O_01;
	Cyclic#1.P3_Srobovanie.PAR.M5_AtlasCopcoInputs[4] AT %ID."P3_Srobovacka_M5".Module003_Input_I_00;
	Cyclic#1.P3_Srobovanie.PAR.M5_AtlasCopcoInputs[5] AT %ID."P3_Srobovacka_M5".Module003_Input_I_01;
	Cyclic#1.P3_Srobovanie.PAR.M5_AtlasCopcoInputs[6] AT %ID."P3_Srobovacka_M5".Module004_Input_I_00;
	Cyclic#1.P3_Srobovanie.PAR.M5_AtlasCopcoInputs[7] AT %ID."P3_Srobovacka_M5".Module004_Input_I_01;
	Cyclic#1.P3_Srobovanie.PAR.M5_AllasCopcoOutputs[4] AT %QD."P3_Srobovacka_M5".Module007_Output_O_00;
	Cyclic#1.P3_Srobovanie.PAR.M5_AllasCopcoOutputs[5] AT %QD."P3_Srobovacka_M5".Module007_Output_O_01;
	Cyclic#1.P3_Srobovanie.PAR.M5_AllasCopcoOutputs[6] AT %QD."P3_Srobovacka_M5".Module008_Output_O_00;
	Cyclic#1.P3_Srobovanie.PAR.M5_AllasCopcoOutputs[7] AT %QD."P3_Srobovacka_M5".Module008_Output_O_01;
	Cyclic#1.AteqLeakageTester_A.Profinet_PLC_INPUTS[24] AT %IB."LeakageTester_A".Module001_Inputs024;
	Cyclic#1.AteqLeakageTester_A.Profinet_PLC_INPUTS[25] AT %IB."LeakageTester_A".Module001_Inputs025;
	Cyclic#1.AteqLeakageTester_A.Profinet_PLC_INPUTS[26] AT %IB."LeakageTester_A".Module001_Inputs026;
	Cyclic#1.AteqLeakageTester_A.Profinet_PLC_INPUTS[27] AT %IB."LeakageTester_A".Module001_Inputs027;
	Cyclic#1.AteqLeakageTester_A.Profinet_PLC_INPUTS[35] AT %IB."LeakageTester_A".Module001_Inputs035;
	Cyclic#1.AteqLeakageTester_A.Profinet_PLC_INPUTS[36] AT %IB."LeakageTester_A".Module001_Inputs036;
	Cyclic#1.AteqLeakageTester_A.Profinet_PLC_INPUTS[41] AT %IB."LeakageTester_A".Module001_Inputs041;
	Cyclic#1.AteqLeakageTester_A.Profinet_PLC_INPUTS[42] AT %IB."LeakageTester_A".Module001_Inputs042;
	Cyclic#1.AteqLeakageTester_A.Profinet_PLC_INPUTS[47] AT %IB."LeakageTester_A".Module001_Inputs047;
	Cyclic#1.AteqLeakageTester_A.Profinet_PLC_INPUTS[48] AT %IB."LeakageTester_A".Module001_Inputs048;
	Cyclic#1.AteqLeakageTester_A.Profinet_PLC_INPUTS[53] AT %IB."LeakageTester_A".Module001_Inputs053;
	Cyclic#1.AteqLeakageTester_A.Profinet_PLC_INPUTS[54] AT %IB."LeakageTester_A".Module001_Inputs054;
	Cyclic#1.AteqLeakageTester_A.Profinet_PLC_OUTPUTS[1] AT %QB."LeakageTester_A".Module005_Outputs001;
	Cyclic#1.AteqLeakageTester_A.Profinet_PLC_OUTPUTS[7] AT %QB."LeakageTester_A".Module005_Outputs007;
	Cyclic#1.AteqLeakageTester_A.Profinet_PLC_OUTPUTS[8] AT %QB."LeakageTester_A".Module005_Outputs008;
	Cyclic#1.AteqLeakageTester_A.PocetCitanychParametrov AT %QB."LeakageTester_A".Module005_Outputs033;
	Cyclic#1.AteqLeakageTester_A.IdentifikaciaParametra_1 AT %QB."LeakageTester_A".Module005_Outputs035;
	Cyclic#1.AteqLeakageTester_A.IdentifikaciaParametra_2 AT %QB."LeakageTester_A".Module005_Outputs037;
	Cyclic#1.AteqLeakageTester_A.IdentifikaciaParametra_3 AT %QB."LeakageTester_A".Module005_Outputs039;
	Cyclic#1.AteqLeakageTester_A.IdentifikaciaParametra_4 AT %QB."LeakageTester_A".Module005_Outputs041;
	Cyclic#1.AteqLeakageTester_B.Profinet_PLC_INPUTS[24] AT %IB."LeakageTester_B".Module001_Inputs024;
	Cyclic#1.AteqLeakageTester_B.Profinet_PLC_INPUTS[25] AT %IB."LeakageTester_B".Module001_Inputs025;
	Cyclic#1.AteqLeakageTester_B.Profinet_PLC_INPUTS[26] AT %IB."LeakageTester_B".Module001_Inputs026;
	Cyclic#1.AteqLeakageTester_B.Profinet_PLC_INPUTS[27] AT %IB."LeakageTester_B".Module001_Inputs027;
	Cyclic#1.AteqLeakageTester_B.Profinet_PLC_INPUTS[35] AT %IB."LeakageTester_B".Module001_Inputs035;
	Cyclic#1.AteqLeakageTester_B.Profinet_PLC_INPUTS[36] AT %IB."LeakageTester_B".Module001_Inputs036;
	Cyclic#1.AteqLeakageTester_B.Profinet_PLC_INPUTS[41] AT %IB."LeakageTester_B".Module001_Inputs041;
	Cyclic#1.AteqLeakageTester_B.Profinet_PLC_INPUTS[42] AT %IB."LeakageTester_B".Module001_Inputs042;
	Cyclic#1.AteqLeakageTester_B.Profinet_PLC_INPUTS[47] AT %IB."LeakageTester_B".Module001_Inputs047;
	Cyclic#1.AteqLeakageTester_B.Profinet_PLC_INPUTS[48] AT %IB."LeakageTester_B".Module001_Inputs048;
	Cyclic#1.AteqLeakageTester_B.Profinet_PLC_INPUTS[53] AT %IB."LeakageTester_B".Module001_Inputs053;
	Cyclic#1.AteqLeakageTester_B.Profinet_PLC_INPUTS[54] AT %IB."LeakageTester_B".Module001_Inputs054;
	Cyclic#1.AteqLeakageTester_B.Profinet_PLC_OUTPUTS[1] AT %QB."LeakageTester_B".Module005_Outputs001;
	Cyclic#1.AteqLeakageTester_B.Profinet_PLC_OUTPUTS[7] AT %QB."LeakageTester_B".Module005_Outputs007;
	Cyclic#1.AteqLeakageTester_B.Profinet_PLC_OUTPUTS[8] AT %QB."LeakageTester_B".Module005_Outputs008;
	Cyclic#1.AteqLeakageTester_B.PocetCitanychParametrov AT %QB."LeakageTester_B".Module005_Outputs033;
	Cyclic#1.AteqLeakageTester_B.IdentifikaciaParametra_1 AT %QB."LeakageTester_B".Module005_Outputs035;
	Cyclic#1.AteqLeakageTester_B.IdentifikaciaParametra_2 AT %QB."LeakageTester_B".Module005_Outputs037;
	Cyclic#1.AteqLeakageTester_B.IdentifikaciaParametra_3 AT %QB."LeakageTester_B".Module005_Outputs039;
	Cyclic#1.AteqLeakageTester_B.IdentifikaciaParametra_4 AT %QB."LeakageTester_B".Module005_Outputs041;
	Cyclic#1.P1_Pracovisko.STAV.VentilovyTerminal_VT4_OK AT %IX."VentilovyTerminal_VT4".ModuleOk;
	Cyclic#1.P1_Pracovisko.STAV.VentilovyTerminal_VT5_OK AT %IX."VentilovyTerminal_VT5".ModuleOk;
	Cyclic#1.CAM2.Profinet_PLC_INPUTS[4] AT %IB."KAM_ControlUNit".Module002_Inputs005;
	Cyclic#1.Linka.STAV.WenglorControlUnit_OK AT %IX."KAM_ControlUNit".ModuleOk;
	Cyclic#1.P3_VstupnyStoper.IN.PritomnPaletky_IS85 AT %IX."DI3.1_16DI".DigitalInput13;
	Cyclic#1.Safety.OUT.P4_ResetBarieryVytahu AT %QX."SI4.1".DigitalOutput02;
	Cyclic#1.Safety.OUT.P1_ResetBarieryVytahu AT %QX."SI1.1".DigitalOutput02;
	Cyclic#1.P2_Pracovisko.STAV.KartaAB21_OK AT %IX."AB2_1_Profinet".ModuleOk;
	Cyclic#1.P1_Srobovanie.IN.SkrutkM4_VysunutieHrotu_IOlink AT %IO."DS1_2".InputData02;
	Cyclic#1.P1_Srobovanie.IN.SkrutkM5_VysunutieHrotu_IOlink AT %IO."DS1_2".InputData03;
	Cyclic#1.P2_Srobovanie.IN.SkrutkM6_VysunutieHrotu_IOlink AT %IO."DS2_3".InputData01;
	Cyclic#1.P2_Srobovanie.IN.SkrutkM4_VysunutieHrotu_IOlink AT %IO."DS2_3".InputData02;
	Cyclic#1.P2_Srobovanie.IN.SkrutkM5_VysunutieHrotu_IOlink AT %IO."DS2_3".InputData03;
	Cyclic#1.P3_Srobovanie.IN.SkrutkK40_VysunutieHrotu_IOlink AT %IO."DS3_3".InputData01;
	Cyclic#1.P3_Srobovanie.IN.SkrutkM5_VysunutieHrotu_IOlink AT %IO."DS3_3".InputData02;
	Cyclic#1.P1_Srobovanie.IN.SkrutkM5_VysunutieHrotu_IOlink AT %IW."DS1_2".InputData03_1;
	Cyclic#1.P2_SkrutkovacMatic.IN.SkrutkMatic_VysunutHrotu_IOlink AT %IW."DS2_1".InputData03_1;
	Cyclic#1.P2_Srobovanie.IN.SkrutkM6_VysunutieHrotu_IOlink AT %IW."DS2_3".InputData01_1;
	Cyclic#1.P2_Srobovanie.IN.SkrutkM4_VysunutieHrotu_IOlink AT %IW."DS2_3".InputData02_1;
	Cyclic#1.P2_Srobovanie.IN.SkrutkM5_VysunutieHrotu_IOlink AT %IW."DS2_3".InputData03_1;
	Cyclic#1.P3_Srobovanie.IN.SkrutkK40_VysunutieHrotu_IOlink AT %IW."DS3_3".InputData01_1;
	Cyclic#1.P3_Srobovanie.IN.SkrutkM5_VysunutieHrotu_IOlink AT %IW."DS3_3".InputData02_1;
END_VAR
```
